(* CODESYS project HiSimulK_NF.project
   Title: BWTS
   Version: 2.0.0.1
   Company: Hyundaiwelding

Project tree, tasks and I/O mapping:
  Device : X2 control 15 - Powerfail, Beijer Electronics Products AB, order no. 
      , version 3.5.13.30
    application Application
      libraries: Util, * (System); Toolbibliothek WM, 1.0.0.6 (Weidmüller Interface GmbH & Co.KG); Standard, * (System); BWTS, 1.4.3.4 (Hyundaiwelding)
      task MainTask (cyclic, interval t#20ms, priority 1) calls MODE, MASTER_SEQUENCE_BALLASTING, MASTER_SEQUENCE_DEBALLASTING, MASTER_SEQUENCE_STRIPPING, SEQ_BAL_SP_P, SEQ_BAL_SP_S, SEQ_BAL_ST_P, SEQ_BAL_ST_S, SEQ_DEBAL_SP_P, SEQ_DEBAL_SP_S, SEQ_DEBAL_ST_P, SEQ_DEBAL_ST_S, SEQ_STRIP_SP, SEQ_STRIP_ST, MASTER_SEQUENCE_DIAGNOSIS, SEQ_DIAG_DEVICE, SEQ_DIAG_INSTRUMENT
      task Alarm (cyclic, interval 20 ms, priority 1) calls ALARM_BUZZER_1, ALARM_BUZZER_2, ALARM_COMMON, ALARM_DEVICE, ALARM_INTERLOCK_A, ALARM_INTERLOCK_D_1, ALARM_INTERLOCK_D_2, ALARM_RECTIFIER, ALARM_TRO
      task ETC (cyclic, interval 50 ms, priority 1) calls AUTO_MODE, BLOWER_TIMER, LINE_UP, MAINTENANCE_AND_DISABLE, RF_CC, SELECTION, TRC_SETTING, UTILITY, RUNNING_HOURS
      task Device (cyclic, interval t#20ms, priority 1) calls DEVICE_AIT151, DEVICE_AIT251, DEVICE_B117A, DEVICE_B117B, DEVICE_FCV1131, DEVICE_FCV2131, DEVICE_FCV1211, DEVICE_FCV2211, DEVICE_GSP01, DEVICE_GSP02, DEVICE_P132, DEVICE_P232, DEVICE_P171A, DEVICE_P171B, DEVICE_RFA, DEVICE_RFB, DEVICE_RFC, DEVICE_WBP01, DEVICE_WBP02, DEVICE_XV1151, DEVICE_XV1171A, DEVICE_XV1171B, DEVICE_XV1172A, DEVICE_XV1321, DEVICE_XV2321, DEVICE_XV1511, DEVICE_XV1512, DEVICE_XV2511, DEVICE_XV2512, DEVICE_XV1731, DEVICE_XV1732, DEVICE_XV1901, DEVICE_XV1541, DEVICE_BA35, DEVICE_BA36, DEVICE_BA37, DEVICE_BA38
      task Shutdown (cyclic, interval t#20ms, priority 1) calls ESD101, PSD10X, PSD11X, PSD12X, PSD20X, PSD21X, PSD22X, PSD30X, PSD31X, USD41X, USD42X, USD43X
      task SIMULATION (cyclic, interval t#20ms, priority 1) calls SCENARIO, SIMULATION_CAL, VIRTUAL_1, VIRTUAL_2, VIRTUAL_3, AMS
      global variables GVL_Alarm_Device
      global variables GVL_IO_DO
      global variables GVL_IO_AO
      global variables GVL_IO_AI
      Logic/
        3.SD/
          program PSD10X [CFC]
          program USD41X [CFC]
          program ESD101 [CFC]
          program PSD20X [CFC]
          program PSD21X [CFC]
          program PSD11X [CFC]
          program USD42X [CFC]
          program PSD12X [CFC]
          program PSD22X [CFC]
          program PSD30X [CFC]
          program PSD31X [CFC]
          program USD43X [CFC]
        1.Mode/
          program MODE [CFC]
        0.ETC/
          program SELECTION [CFC]
          program TRC_SETTING [CFC]
          program MAINTENANCE_AND_DISABLE [CFC]
          program RF_CC [CFC]
          program UTILITY [CFC]
          program BLOWER_TIMER [CFC]
          program AUTO_MODE [CFC]
          program LINE_UP [CFC]
          program RUNNING_HOURS [ST]
        2.Sequence/
          program SEQ_BAL_ST_S [CFC]
          program SEQ_DEBAL_SP_S [CFC]
          program SEQ_DEBAL_ST_S [CFC]
          program MASTER_SEQUENCE_BALLASTING [CFC]
          program MASTER_SEQUENCE_DEBALLASTING [CFC]
          program SEQ_BAL_SP_S [CFC]
          program MASTER_SEQUENCE_STRIPPING [CFC]
          program SEQ_BAL_ST_P [CFC]
          program SEQ_BAL_SP_P [CFC]
          program SEQ_DEBAL_ST_P [CFC]
          program SEQ_DEBAL_SP_P [CFC]
          program SEQ_STRIP_ST [CFC]
          program SEQ_STRIP_SP [CFC]
          program MASTER_SEQUENCE_DIAGNOSIS [CFC]
          program SEQ_DIAG_DEVICE [ST]
          program SEQ_DIAG_INSTRUMENT [ST]
        0.ALARM/
          program ALARM_INTERLOCK_D_1 [CFC]
          program ALARM_BUZZER_1 [ST]
          program ALARM_RECTIFIER [ST]
          program ALARM_INTERLOCK_A [CFC]
          program ALARM_TRO [CFC]
          program ALARM_DEVICE [ST]
          program ALARM_INTERLOCK_D_2 [CFC]
          program ALARM_COMMON [ST]
          program ALARM_BUZZER_2 [ST]
        4.Device/
          program DEVICE_FCV1211 [CFC]
          program DEVICE_P171A [CFC]
          program DEVICE_WBP01 [CFC]
          program DEVICE_XV1731 [CFC]
          program DEVICE_XV1171B [CFC]
          program DEVICE_AIT151 [CFC]
          program DEVICE_XV1732 [CFC]
          program DEVICE_B117B [CFC]
          program DEVICE_XV1511 [CFC]
          program DEVICE_FCV1131 [CFC]
          program DEVICE_RFA [CFC]
          program DEVICE_XV1151 [CFC]
          program DEVICE_B117A [CFC]
          program DEVICE_XV1512 [CFC]
          program DEVICE_P132 [CFC]
          program DEVICE_XV1171A [CFC]
          program DEVICE_XV1172A [CFC]
          program DEVICE_P171B [CFC]
          program DEVICE_P232 [CFC]
          program DEVICE_RFB [CFC]
          program DEVICE_WBP02 [CFC]
          program DEVICE_XV1321 [CFC]
          program DEVICE_XV1541 [CFC]
          program DEVICE_XV2321 [CFC]
          program DEVICE_XV1901 [CFC]
          program DEVICE_GSP01 [CFC]
          program DEVICE_GSP02 [CFC]
          program DEVICE_AIT251 [CFC]
          program DEVICE_XV2511 [CFC]
          program DEVICE_XV2512 [CFC]
          program DEVICE_FCV2211 [CFC]
          program DEVICE_FCV2131 [CFC]
          program DEVICE_RFC [CFC]
          program DEVICE_BA35 [CFC]
          program DEVICE_BA36 [CFC]
          program DEVICE_BA37 [CFC]
          program DEVICE_BA38 [CFC]
        0.SIMULATION/
          program AMS [CFC]
          program SCENARIO [CFC]
          program VIRTUAL_1 [CFC]
          program SIMULATION_CAL [CFC]
          program VIRTUAL_2 [CFC]
          program VIRTUAL_3 [ST]
        0.SIMULATION FBD/
          function block SM_RF_TRO1 [CFC]
          function SM_CELL_VOLT [ST]
          function SM_NA_TRO [ST]
          function SM_H2_CONC [ST]
          function SM_HEAT [ST]
          function block SM_FU_DP [ST]
          function block SM_FOT [CFC]
          function block SM_RF_TRO [ST]
      Symbols
      global variables GVL_Event_Operation
      global variables GVL_SEQ_LIB
      global variables GVL_Event_Device
      global variables GVL_Alarm_Interlock
      global variables GVL_Event_Optrack
      global variables GVL_IO_DI
      global variables GVL_Alarm_System
      global variables GVL_IO_RECTIFIER
      global variables PersistentVars
      global variables GVL_UTILITY
      global variables GVL_SIMULATION
      global variables GVL_IO_TRO
*)

// Device/Application/GVL_Alarm_Device
//{attribute 'qualified_only'}
VAR_GLOBAL
	/////////////////////////////////////// Tags that registered as an Alarm ///////////////////////////////////////
	
	//BLOWER
	B117A_STF : BOOL;
	B117A_SPF : BOOL;
	B117B_STF : BOOL;
	B117B_SPF : BOOL;
	
	XV1171A_OPF : BOOL;
	XV1171A_CLF : BOOL;
	XV1171B_OPF : BOOL;
	XV1171B_CLF : BOOL;
	
	//Sea Water Feeding Unit
	P171A_STF : BOOL;
	P171A_SPF : BOOL;
	P171B_STF : BOOL;
	P171B_SPF : BOOL;
	
	//Injection Flow Control Valves
	FCV1131_CF : BOOL;	// FCV-1131 CONTROL FAIL
	FCV2131_CF : BOOL;	// FCV-2131 CONTROL FAIL
	
	//Main Flow Control Valves
	FCV1211_CF : BOOL;	// FCV-1211 CONTROL FAIL
	FCV2211_CF : BOOL;	// FCV-2211 CONTROL FAIL

	//N.U UNIT
	P132_STF : BOOL;
	P132_SPF : BOOL;
	P232_STF : BOOL;
	P232_SPF : BOOL;
		
	//RECTIFIER
	RF142A_STF : BOOL;
	RF142A_SPF : BOOL;
	RF142B_STF : BOOL;
	RF142B_SPF : BOOL;
	RF142C_STF : BOOL;
	RF142C_SPF : BOOL;

	//W.B PUMP
	WBP01_STF : BOOL;
	WBP01_SPF : BOOL;
	WBP02_STF : BOOL;
	WBP02_SPF : BOOL;

	GSP01_STF : BOOL;
	GSP01_SPF : BOOL;
	GSP02_STF : BOOL;
	GSP02_SPF : BOOL;
	
	/////////////////////////////////////// END : Tags that registered as an Alarm ///////////////////////////////////////
	
	// BALLAST VALVES
	BA35_OPF : BOOL;
	BA35_CLF : BOOL;
	BA36_OPF : BOOL;
	BA36_CLF : BOOL;
	BA37_OPF : BOOL;
	BA37_CLF : BOOL;
	BA38_OPF : BOOL;
	BA38_CLF : BOOL;
END_VAR

// Device/Application/GVL_IO_DO
//{attribute 'qualified_only'}
VAR_GLOBAL
	// Digital Output with DC 24V
	BWTS_003 : BOOL; //Shutdown alarm Lamp
	BWTS_004 : BOOL; //Common alarm Lamp
	BWTS_007 : BOOL; //Alarm buzzer
	
	XV_1151_CMD : BOOL;
	XV_1172A_CMD : BOOL;
	XV_1731_CMD : BOOL;
	XV_1732_CMD : BOOL;
	XV_1171A_CMD : BOOL;
	XV_1171B_CMD : BOOL;
	XV_1901_CMD : BOOL; 

	XV_1321_CMD : BOOL;
	XV_2321_CMD : BOOL;
	AIT_151_ST : BOOL;
	AIT_251_ST : BOOL;

	XV_1511_CMD : BOOL;
	XV_1512_CMD : BOOL;
	XV_2511_CMD : BOOL;
	XV_2512_CMD : BOOL;

	XV_1541_CMD : BOOL;
	
	// Digital Output with free voltage
	
	BWTS_005 : BOOL;		// BWTS COMMON ALARM TO AMS	
	BWTS_006 : BOOL;		// BWTS SHUTDOWN ALARM TO AMS
	BWTS_009 : BOOL;		// BWTS RUNNING TO AMS
	B_117A_ST : BOOL;
	B_117B_ST : BOOL;
	P_171A_ST : BOOL;
	P_171B_ST : BOOL;
	
	P_132_ST : BOOL;
	P_232_ST : BOOL;
	
	RF_142A_ST : BOOL;
	RF_142A_SP : BOOL;
	RF_142B_ST : BOOL;
	RF_142B_SP : BOOL;
	RF_142C_ST : BOOL;
	RF_142C_SP : BOOL;

	GSP_01_SP : BOOL;
	GSP_02_SP : BOOL;
END_VAR

// Device/Application/GVL_IO_AO
//{attribute 'qualified_only'}
VAR_GLOBAL
	// Analog Output
	FCV_1211_CMD : REAL;
	FCV_2211_CMD : REAL;
	
	FCV_1131_CMD : REAL;
	FCV_2131_CMD : REAL;

	P_132_CMD : REAL;
	P_232_CMD : REAL;

END_VAR

// Device/Application/GVL_IO_AI
//{attribute 'qualified_only'}
VAR_GLOBAL
	// Analog Input
	CT_1111 : REAL;
	TE_1111 : REAL;
	AIT_1121 : REAL;
	AIT_1122 : REAL;
	AIT_1123 : REAL;
	PT_1121 : REAL;
	PT_1721 : REAL;
	PT_1722 : REAL;
	LIT_1311 : REAL;
	AP_LVL_01 : REAL;

	P_132_FD : REAL;
	P_232_FD : REAL;

	FCV_1211_FD : REAL;
	FCV_2211_FD : REAL;

	FIT_1211 : REAL;
	FIT_2211 : REAL;

	FCV_1131_FD : REAL;
	FCV_2131_FD : REAL;

	FIT_1131 : REAL;
	FIT_2131 : REAL;

	AIT_151 : REAL;
	AIT_251 : REAL;
	
	/////////////////////////////////////////////////////////// ANALOGUE RANGE ///////////////////////////////////////////////////////////
	
	RL_CT_1111 : REAL := 0;	
	RH_CT_1111 : REAL := 100;
	
	RL_TE_1111 : REAL := 0;
	RH_TE_1111 : REAL := 55;
	
	RL_PT_1121 : REAL := -70;
	RH_PT_1121 : REAL := 70;
	
	RL_PT_1721 : REAL := 0;
	RH_PT_1721 : REAL := 10;
	RL_PT_1722 : REAL := 0;
	RH_PT_1722 : REAL := 10;
	
	RL_AP_LVL_01 : REAL := 0;
	RH_AP_LVL_01 : REAL := 800;	
	
	RL_FIT_1211 : REAL := 0;
	RH_FIT_1211 : REAL := 10163;
	
	RL_FIT_2211 : REAL := 0;
	RH_FIT_2211 : REAL := 10163;
	
	RL_FIT_1131 : REAL := 0;
	RH_FIT_1131 : REAL := 120;
	
	RL_FIT_2131 : REAL := 0;
	RH_FIT_2131 : REAL := 120;
	
	RL_AIT_151 : REAL := 0;
	RH_AIT_151 : REAL := 16;
	
	RL_AIT_251 : REAL := 0;
	RH_AIT_251 : REAL := 16;
	
END_VAR

// Device/Application/GVL_Event_Operation
//{attribute 'qualified_only'}
VAR_GLOBAL
	//OPERATION STATUS
	BAL_ST_S, BAL_IN_STBD, BAL_SP_S, BAL_S_RDY : BOOL;			// STBD BALLASTING
	BAL_ST_P, BAL_IN_PORT, BAL_SP_P, BAL_P_RDY : BOOL;			// PORT BALLASTING  	
		    	
	DEBAL_ST_S, DEBAL_IN_STBD, DEBAL_SP_S, DEBAL_S_RDY : BOOL;				// STBD DEBALLASTING
	DEBAL_ST_P, DEBAL_IN_PORT, DEBAL_SP_P, DEBAL_P_RDY : BOOL;				// PORT DEBALLASTING
		
	STR_ST_S, STR_IN_STBD, STR_SP_S, STR_S_RDY : BOOL;						// STBD STRIPPING
		
	WBP01_ST_REQ: BOOL;
	WBP01_SP_REQ: BOOL;
	WBP02_ST_REQ: BOOL;
	WBP02_SP_REQ: BOOL;
	
	GSP01_ST_REQ: BOOL;
	GSP01_SP_REQ: BOOL;
	GSP02_ST_REQ: BOOL;
	GSP02_SP_REQ: BOOL;	
	
	DIAG_ST, DIAG_IN_SELF : BOOL;	// SELF-DIAGNOSIS --------------- ADDED BY VER.1
END_VAR

// Device/Application/GVL_SEQ_LIB
//{attribute 'qualified_only'}
VAR_GLOBAL
	MST_BST_S, MST_BST_P : BWTS.SEQ;
	MST_BSP_S, MST_BSP_P : BWTS.SEQ;
	
	BST_S_01, BST_P_01 : BWTS.SEQ;	// Blower Start
	
	BST_S_03, BST_P_03 : BWTS.SEQ;	// TRC Valve Init. Open
	BST_S_04, BST_P_04 : BWTS.SEQ;	// Inj. Valve Init. Open
	BST_S_05, BST_P_05 : BWTS.SEQ;	// H/E Valve Init. Open
	BST_S_06, BST_P_06 : BWTS.SEQ;	// S.W.F.P Start
	BST_S_07, BST_P_07 : BWTS.SEQ;	// E/U Level Check
	BST_S_08, BST_P_08 : BWTS.SEQ;	// WBP Start Request
	
	BST_S_10, BST_P_10 : BWTS.SEQ;	// Salinity Check
	
	BST_S_12, BST_P_12 : BWTS.SEQ;	// Main flow Control
	BST_S_13, BST_P_13 : BWTS.SEQ;	// Inj. Flow Control
	BST_S_14, BST_P_14 : BWTS.SEQ;	// Rectifier Start
	BST_S_15, BST_P_15 : BWTS.SEQ;	// TRO Valve Open
	BST_S_16, BST_P_16 : BWTS.SEQ;	// TRO Sensing Start
	
	BST_S_18, BST_P_18 : BWTS.SEQ;	// Ballast Valves ACtion
	                                 	
	BSP_S_01, BSP_P_01 : BWTS.SEQ;	// Rectifier Stop
	
	BSP_S_03, BSP_P_03 : BWTS.SEQ;	// WBP Stop Request
	BSP_S_04, BSP_P_04 : BWTS.SEQ;	// TRO Unit Stop
	BSP_S_05, BSP_P_05 : BWTS.SEQ;	// S.W.F.P Stop
	
	BSP_S_07, BSP_P_07 : BWTS.SEQ;	// H/E Valve Close
	BSP_S_08, BSP_P_08 : BWTS.SEQ;	// Inj. Valve Close
	BSP_S_09, BSP_P_09 : BWTS.SEQ;	// TRC Valve Close
	BSP_S_10, BSP_P_10 : BWTS.SEQ;	// Blower Stop
	
	BSP_S_12, BSP_P_12 : BWTS.SEQ;	// Ballast Valve Act.

	MST_DST_S, MST_DST_P : BWTS.SEQ;
	MST_DSP_S, MST_DSP_P : BWTS.SEQ;
	
	          
	DST_S_02, DST_P_02 : BWTS.SEQ;	// TRC Valve Init. Open        
	DST_S_03, DST_P_03 : BWTS.SEQ;	// N/U Start
	DST_S_04, DST_P_04 : BWTS.SEQ;	// WBP Start Request            
	DST_S_05, DST_P_05 : BWTS.SEQ;	// TRO Valve Open         
	DST_S_06, DST_P_06 : BWTS.SEQ;	// Main Flow Control
	DST_S_07, DST_P_07 : BWTS.SEQ;	// TRO Sensing Start          
	DST_S_08, DST_P_08 : BWTS.SEQ;	// Recirculation Mode       
	DST_S_09, DST_P_09 : BWTS.SEQ;	// Discharge Mode
		                  
	DSP_S_01, DSP_P_01 : BWTS.SEQ;	// WBP Stop Request
	DSP_S_02, DSP_P_02 : BWTS.SEQ;	// N/U Pump Stop
	DSP_S_03, DSP_P_03 : BWTS.SEQ;	// TRO Unit Stop
	
	DSP_S_05, DSP_P_05 : BWTS.SEQ;	// TRC Valve Close
	DSP_S_06, DSP_P_06 : BWTS.SEQ;	// N/U Inj. Valve Close
	DSP_S_07, DSP_P_07 : BWTS.SEQ;	// Ballast Valve Act.

	MST_SST_S, MST_SST_P : BWTS.SEQ;
	MST_SSP_S, MST_SSP_P : BWTS.SEQ;
	
	SST_S_01 : BWTS.SEQ;	// N/U Start          
	SST_S_02 : BWTS.SEQ;	// WBP Start Request       
	SST_S_03 : BWTS.SEQ;	// TRO Valve Open
	SST_S_04 : BWTS.SEQ;	// TRO Sensing Start           
	   
	SST_S_06 : BWTS.SEQ;	// TRC Valve Open         
	SST_S_07 : BWTS.SEQ;	// Ballast Valves Action          
	SST_S_08 : BWTS.SEQ;	// Eductor Valve Open       
	SST_S_09 : BWTS.SEQ;	// TRO Booster Unit Start
	        
	SSP_S_01 : BWTS.SEQ;	// WBP Stop Request
	SSP_S_02 : BWTS.SEQ;	// N/U Pump Stop 
	SSP_S_03 : BWTS.SEQ;	// TRO Unit Stop
	SSP_S_04 : BWTS.SEQ;	// N/U Inj. Valve Close
	
	SSP_S_06 : BWTS.SEQ;	// TRC Valve Close
	SSP_S_07 : BWTS.SEQ;	// Eductor Valve Close
	
	// PSD
	PSD101, PSD102, PSD103, PSD10 : BWTS.PSD;									// Ballasting Common Process Shutdown
	PSD111, PSD113, PSD114, PSD115, PSD11 : BWTS.PSD;					// Ballast STBD Process Shutdown
	PSD121, PSD123, PSD124, PSD125, PSD12 : BWTS.PSD;					// Ballast PORT Process Shutdown
		
	PSD201, PSD20: BWTS.PSD;													// Deballasting Common Process Shutdown
	PSD211, PSD212, PSD213, PSD21 : BWTS.PSD;									// Deballasting STBD Process Shutdown
	PSD221, PSD222, PSD223, PSD22 : BWTS.PSD;									// Deballasting PORT Process Shutdown
		
	PSD301, PSD30 : BWTS.PSD;													// Stripping Common Process Shutdown
	PSD311, PSD312, PSD313, PSD31 : BWTS.PSD;									// Stripping STBD Process Shutdown
		
	SEQ112, SEQ122, SEQ212, SEQ222, SEQ312 : BWTS.PSD;			// Sequence Fail
	
	PSD41, PSD42, PSD43 : BWTS.PSD;
	ESD01 : BWTS.PSD;										// Emergency Shutdown
	
		// SELF-DIAGNOSIS ---------- ADDED BY VER 1
	MST_DIAG : BWTS.SEQ;
	
	DIAG_B117A_1 : BWTS.SEQ;
	DIAG_B117A_2 : BWTS.SEQ;
	DIAG_B117A_3 : BWTS.SEQ;
	
	DIAG_B117B_1 : BWTS.SEQ;
	DIAG_B117B_2 : BWTS.SEQ;
	DIAG_B117B_3 : BWTS.SEQ;
	
	DIAG_XV1171A_1 : BWTS.SEQ;
	DIAG_XV1171A_2 : BWTS.SEQ;
	DIAG_XV1171A_3 : BWTS.SEQ;
	
	DIAG_XV1171B_1 : BWTS.SEQ;
	DIAG_XV1171B_2 : BWTS.SEQ;
	DIAG_XV1171B_3 : BWTS.SEQ;
	
	DIAG_P132_1 : BWTS.SEQ;
	DIAG_P132_2 : BWTS.SEQ;
	DIAG_P132_3 : BWTS.SEQ;
	
	DIAG_P232_1 : BWTS.SEQ;
	DIAG_P232_2 : BWTS.SEQ;
	DIAG_P232_3 : BWTS.SEQ;
	
	DIAG_FCV1211_1 : BWTS.SEQ;
	DIAG_FCV1211_2 : BWTS.SEQ;
	DIAG_FCV1211_3 : BWTS.SEQ;
	DIAG_FCV1211_4 : BWTS.SEQ;
	
	DIAG_FCV2211_1 : BWTS.SEQ;
	DIAG_FCV2211_2 : BWTS.SEQ;
	DIAG_FCV2211_3 : BWTS.SEQ;
	DIAG_FCV2211_4 : BWTS.SEQ;
	
	DIAG_FCV1131_1 : BWTS.SEQ;
	DIAG_FCV1131_2 : BWTS.SEQ;
	DIAG_FCV1131_3 : BWTS.SEQ;
	DIAG_FCV1131_4 : BWTS.SEQ;
	
	DIAG_FCV2131_1 : BWTS.SEQ;
	DIAG_FCV2131_2 : BWTS.SEQ;
	DIAG_FCV2131_3 : BWTS.SEQ;
	DIAG_FCV2131_4 : BWTS.SEQ;
		
	DIAG_BA35_1 : BWTS.SEQ;
	DIAG_BA35_2 : BWTS.SEQ;
	DIAG_BA35_3 : BWTS.SEQ;
	DIAG_BA36_1 : BWTS.SEQ;
	DIAG_BA36_2 : BWTS.SEQ;
	DIAG_BA36_3 : BWTS.SEQ;
	DIAG_BA37_1 : BWTS.SEQ;
	DIAG_BA37_2 : BWTS.SEQ;
	DIAG_BA37_3 : BWTS.SEQ;
	DIAG_BA38_1 : BWTS.SEQ;
	DIAG_BA38_2 : BWTS.SEQ;
	DIAG_BA38_3 : BWTS.SEQ;
END_VAR

// Device/Application/GVL_Event_Device
//{attribute 'qualified_only'}
VAR_GLOBAL
	
	FULL_AUTO : BOOL;
	MAINTENANCE : BOOL;	//Maintenance
	
	// BLOWER UNIT
	B117A_A : BOOL;
	B117A_M : BOOL;
	B117A_RUN : BOOL;
	B117A_SPD : BOOL;
	B117B_A : BOOL;
	B117B_M : BOOL;
	B117B_RUN : BOOL;
	B117B_SPD : BOOL;
	
	XV1171A_A : BOOL; 
	XV1171A_M : BOOL;
	XV1171A_OPD : BOOL;
	XV1171A_CLD : BOOL;
	XV1171B_A : BOOL; 
	XV1171B_M : BOOL;
	XV1171B_OPD : BOOL;
	XV1171B_CLD : BOOL;
		
	// TRC CONTROL VAVLE
	FCV1211_A : BOOL;
	FCV1211_M : BOOL;
	FCV1211_OPD : BOOL;
	FCV1211_CLD : BOOL;
	FCV1211_ON : BOOL;
	
	FCV2211_A : BOOL;
	FCV2211_M : BOOL;
	FCV2211_OPD : BOOL;
	FCV2211_CLD : BOOL;
	FCV2211_ON : BOOL;

	// INJECTION CONTROL VAVLE
	FCV1131_A : BOOL;
	FCV1131_M : BOOL;
	FCV1131_OPD : BOOL;
	FCV1131_CLD : BOOL;
	FCV1131_ON : BOOL;
	
	FCV2131_A : BOOL;
	FCV2131_M : BOOL;
	FCV2131_OPD : BOOL;
	FCV2131_CLD : BOOL;
	FCV2131_ON : BOOL;
	
	// HEATER INLET/BYPASS VAVLE
	XV1731_A : BOOL;
	XV1731_M : BOOL;
	XV1731_OPD : BOOL;
	XV1731_CLD : BOOL;
	XV1732_A : BOOL;
	XV1732_M : BOOL;
	XV1732_OPD : BOOL;
	XV1732_CLD : BOOL;
		
	// SEA WATER FEED PUMP
	P171A_RUN : BOOL;
	P171A_SPD : BOOL;
	P171A_A : BOOL;
	P171A_M : BOOL;
	P171B_RUN : BOOL;
	P171B_SPD : BOOL;
	P171B_A : BOOL;
	P171B_M : BOOL;
	
	// TRO INLET VALVE	
	XV1511_A : BOOL;
	XV1511_M : BOOL;
	XV1511_OPD : BOOL;
	XV1511_CLD : BOOL;
	
	XV1512_A : BOOL;
	XV1512_M : BOOL;
	XV1512_OPD : BOOL;
	XV1512_CLD : BOOL;
			
	XV2511_A : BOOL;
	XV2511_M : BOOL;
	XV2511_OPD : BOOL;
	XV2511_CLD : BOOL;

	XV2512_A : BOOL;
	XV2512_M : BOOL;
	XV2512_OPD : BOOL;
	XV2512_CLD : BOOL;

	XV1541_A, XV1541_M : BOOL;
	XV1541_OPD, XV1541_CLD : BOOL;
 
	// TRO SENSORS
	AIT151_A : BOOL;
	AIT151_M : BOOL;
	AIT151_RUN : BOOL;
	AIT151_SPD : BOOL;
	
	AIT251_A : BOOL;
	AIT251_M : BOOL;
	AIT251_RUN : BOOL;
	AIT251_SPD : BOOL;

	// CLOSED TANK VALVE
	XV1151_A : BOOL;
	XV1151_M : BOOL;
	XV1151_OPD : BOOL;
	XV1151_CLD : BOOL;
	
	// RECTIFIER
	RFA_A : BOOL;
	RFA_M : BOOL;
	RFA_RUN : BOOL;
	RFA_SPD : BOOL;
	
	RFB_A : BOOL;
	RFB_M : BOOL;
	RFB_RUN : BOOL;
	RFB_SPD : BOOL;
	
	RFC_A : BOOL;
	RFC_M : BOOL;
	RFC_RUN : BOOL;
	RFC_SPD : BOOL;
		
	// MAIN PUMP
	WBP01_RUN : BOOL;
	WBP01_SPD : BOOL;	
	WBP02_RUN : BOOL;
	WBP02_SPD : BOOL;
	
	GSP01_RUN : BOOL;
	GSP01_SPD : BOOL;
	GSP02_RUN : BOOL;
	GSP02_SPD : BOOL;
	
	// N.A UNIT
	P132_A : BOOL;
	P132_M : BOOL;
	P132_RUN : BOOL;
	P132_SPD : BOOL;
	
	P232_A : BOOL;
	P232_M : BOOL;
	P232_RUN : BOOL;
	P232_SPD : BOOL;
	
	XV1321_A : BOOL;
	XV1321_M : BOOL;
	XV1321_OPD : BOOL;
	XV1321_CLD : BOOL;
	
	XV2321_A : BOOL;
	XV2321_M : BOOL;
	XV2321_OPD : BOOL;
	XV2321_CLD : BOOL;

	// DRAIN UNIT
	XV1901_A : BOOL;
	XV1901_M : BOOL;
	XV1901_OPD : BOOL;
	XV1901_CLD : BOOL;		

	////////////////////////////////////////////////// SELECTION //////////////////////////////////////////////////
	B117A_SEL : BOOL;
	B117B_SEL : BOOL;
	
	P171A_SEL : BOOL;
	P171B_SEL : BOOL;
	
	TRO01_SEL: BOOL;
	TRO02_SEL : BOOL;
	TRO_CROSS : BOOL;
	
	P132_SEL : BOOL;
	P232_SEL : BOOL;
	NU_CROSS : BOOL;
	
	RFA_DISABLE : BOOL;
	RFB_DISABLE : BOOL;
	RFC_DISABLE : BOOL;
	
	GSP01_SEL : BOOL;
	GSP02_SEL : BOOL;
		
	SEA_ENABLE : BOOL;
	
	SEA_ENABLE_S : BOOL;
	SEA_ENABLE_P : BOOL;
	
	CIR_ENABLE_S : BOOL;
	CIR_ENABLE_P : BOOL;
	
	//BALLAST VALVES
	BA35_A : BOOL;
	BA35_M : BOOL;
	BA36_A : BOOL;
	BA36_M : BOOL;
	BA37_A : BOOL;
	BA37_M : BOOL;
	BA38_A : BOOL;
	BA38_M : BOOL;
END_VAR

// Device/Application/GVL_Alarm_Interlock
//{attribute 'qualified_only'}
VAR_GLOBAL
	/////////////////////////////////////// Tags that registered as an Alarm ///////////////////////////////////////
	//Feeding Sea Water salinity
	CT_1111_LO : BOOL;
	CT_1111_LL : BOOL;
	
	//Feeding Sea Water Temperature
	TE_1111_HI : BOOL;
	TE_1111_LO : BOOL;
	TE_1111_LL : BOOL;
	
	//H2 Gas Detector
	AIT_1121_HH : BOOL;
	AIT_1121_HI : BOOL;
	AIT_1122_HH : BOOL;
	AIT_1122_HI : BOOL;
	AIT_1123_HH : BOOL;
	AIT_1123_HI : BOOL;
	
	//APT Level Too Level
	AP_LVL_LO, AP_LVL_LL : BOOL;
	
	//Blower Unit
	PT_1121_HI : BOOL;
	PT_1121_LO : BOOL;
	PT_1121_LL : BOOL;
	B_117A_F : BOOL;
	B_117B_F : BOOL;
	B_117A_OFF : BOOL;
	B_117B_OFF : BOOL;
	BLR_BOTH_F : BOOL;
	
	//SEA WATER FEEDING UNIT
	PT_1721_HI : BOOL;
	PT_1721_LO : BOOL;
	PT_1721_LL : BOOL;
	PT_1722_HH : BOOL;
	PT_1722_HI : BOOL;
	PT_1722_LO : BOOL;
	
	SWFU_DP_HH : BOOL;
	SWFU_DP_HI : BOOL;
	
	P_171A_F : BOOL;
	P_171A_OFF : BOOL;
	P_171B_F : BOOL;
	P_171B_OFF : BOOL;
	
	SWFP_BOTH_F : BOOL;
	
	// LINE-UP FAIL ALARM
	BAL_VV_AL_S : BOOL;
	BAL_VV_AL_P : BOOL;
		
	DEBAL_VV_AL_S : BOOL;
	DEBAL_VV_AL_P : BOOL;
	
	STR_VV_AL_S : BOOL;
	
	//Main Flow rate
	FIT_1211_HH : BOOL;
	FIT_1211_HI : BOOL;
	FIT_1211_LO : BOOL;
	FIT_2211_HH : BOOL;
	FIT_2211_HI : BOOL;
	FIT_2211_LO : BOOL;
	
	//Injection Flow rate
	FIT_1131_LO, FIT_1131_LL : BOOL;
	FIT_2131_LO, FIT_2131_LL : BOOL;

	RFS_1131 : BOOL;
	RFS_2131 : BOOL;
	
	//TRO Sensor
	BTRO_HH_S : BOOL;
	BTRO_HI_S : BOOL;
	BTRO_LO_S : BOOL;
	BTRO_LL_S : BOOL;
	DTRO_HH_S : BOOL;
	DTRO_HI_S : BOOL;
	
	BTRO_HH_P : BOOL;
	BTRO_HI_P : BOOL;
	BTRO_LO_P : BOOL;
	BTRO_LL_P : BOOL;
	DTRO_HH_P : BOOL;
	DTRO_HI_P : BOOL;
	
	STRO_HH : BOOL;
	STRO_HI : BOOL;
	
	AIT_151_E : BOOL;
	AIT_151_F : BOOL;
	AIT_151_L : BOOL; // FOR HiQ-TRO
	AIT_151_BYPASS : BOOL; // FOR HiQ-TRO (* 2023.06.01, JSY - Change from event to alarm*) 
	AIT_151_PF : BOOL; // FOR HiQ-TRO (* 2023.06.01, JSY - Power source supply statue Purge Controller to the TRO sensor*) 
	
	AIT_251_E : BOOL;
	AIT_251_F : BOOL;
	AIT_251_L : BOOL; // FOR HiQ-TRO
	AIT_251_BYPASS : BOOL; // FOR HiQ-TRO (* 2023.06.01, JSY - Change from event to alarm*)
	AIT_251_PF : BOOL; // FOR HiQ-TRO (* 2023.06.01, JSY - Power source supply statue Purge Controller to the TRO sensor*)

	//TRO DRAIN UNIT
	LS_1901_HH : BOOL;
	
	//E.U Level Switch
	LS_1111_LL : BOOL;
	LS_1141_HI : BOOL;
	
	//N.A UNIT
	LIT_1311_HI : BOOL;
	LIT_1311_LO : BOOL;
	LIT_1311_LL : BOOL;
	
	P_132_TRIP : BOOL;
	P_232_TRIP : BOOL;
	
	DPS_1321 : BOOL;
	DPS_2321 : BOOL;
	
	//RECTIFIER
	//ALARM
	REC1001, REC2001, REC3001 : BOOL;	// RECTIFIER ERROR
	REC1002, REC2002, REC3002 : BOOL;	// RECTIFIER E-STOP BY INTERNAL SAFETY INTERLOCK
	REC1003, REC2003, REC3003 : BOOL;	// RECTIFIER MODULE1 INPUT OVER CURRENT
	REC1004, REC2004, REC3004 : BOOL;	// RECTIFIER MODULE2 INPUT OVER CURRENT
	REC1005, REC2005, REC3005 : BOOL;	// RECTIFIER MODULE3 INPUT OVER CURRENT
	REC1006, REC2006, REC3006 : BOOL;	// RECTIFIER MODULE1 OUTPUT OVER CURRENT
	REC1007, REC2007, REC3007 : BOOL;	// RECTIFIER MODULE2 OUTPUT OVER CURRENT
	REC1008, REC2008, REC3008 : BOOL;	// RECTIFIER MODULE3 OUTPUT OVER CURRENT
	REC1009, REC2009, REC3009 : BOOL;	// RECTIFIER OUTPUT OVER VOLTAGE
	REC1010, REC2010, REC3010 : BOOL;	// RECTIFIER MODULE1 OVER TEMPERATURE
	REC1011, REC2011, REC3011 : BOOL;	// RECTIFIER MODULE2 OVER TEMPERATURE
	REC1012, REC2012, REC3012 : BOOL;	// RECTIFIER MODULE3 OVER TEMPERATURE
	REC1013, REC2013, REC3013 : BOOL;	// RECTIFIER UNBALANCE CURRENT
	REC1014, REC2014, REC3014 : BOOL;	// RECTIFIER LOCAL MODE
	REC1015, REC2015, REC3015 : BOOL;	// RECTIFIER LOCAL-REMOTE MODE
	REC1022, REC2022, REC3022 : BOOL;	// RECTIFIER MODULE1 FUSE ALARM
	REC1023, REC2023, REC3023 : BOOL; 	// RECTIFIER MODULE2 FUSE ALARM
	REC1024, REC2024, REC3024 : BOOL;	// RECTIFIER MODULE3 FUSE ALARM
	REC1025, REC2025, REC3025 : BOOL; 	// RECTIFIER EMERGENCY OPERATION
	REC1026, REC2026, REC3026 : BOOL; 	// RECTIFIER FAN ALARM
	REC1032, REC2032, REC3032 : BOOL; 	// RECTIFIER E-STOP BY EXTERNAL COMMAND
	REC1033, REC2033, REC3033 : BOOL; 	// RECTIFIER INTERNAL OVER TEMPERATURE
	
	REC1017_HH, REC1017_HI, REC1018_HH, REC1018_HI, REC1019_HH, REC1019_HI, REC1020_HH,	REC1020_HI,	REC1021_HH,	REC1021_HI,	REC1027_HH,	REC1027_HI : BOOL;
	RF_142A_E : BOOL;
	
	REC2017_HH,	REC2017_HI, REC2018_HH, REC2018_HI, REC2019_HH, REC2019_HI,	REC2020_HH,	REC2020_HI, REC2021_HH, REC2021_HI, REC2027_HH,	REC2027_HI : BOOL;
	RF_142B_E : BOOL;
	
	REC3017_HH,	REC3017_HI, REC3018_HH, REC3018_HI, REC3019_HH, REC3019_HI,	REC3020_HH,	REC3020_HI, REC3021_HH, REC3021_HI, REC3027_HH,	REC3027_HI : BOOL;
	RF_142C_E : BOOL;
	
	RF_ALL_SPD : BOOL;
	
	//FAN Alarm
	PR_FAN_OFF : BOOL;
	ER_FAN_OFF : BOOL;
	
	// MCC-100 BREAKER OFF
	MCC_100_OFF : BOOL;
	
	//E.U Outlet Alarm
	ZS_1112A_CL : BOOL;
	ZS_1112A_OP : BOOL;
	ZS_1113A_CL : BOOL;
	ZS_1113A_OP : BOOL;
	ZS_1114A_CL : BOOL;
	ZS_1114A_OP : BOOL;
	
	// MAIN PUMP ALARM
	WBP_01_AL : BOOL;
	WBP_01_FAULT : BOOL;
	WBP_02_AL : BOOL;
	WBP_02_FAULT : BOOL;
	
	GSP_01_AL : BOOL;
	GSP_02_AL : BOOL;
	GSP_01_FAULT : BOOL;
	GSP_02_FAULT : BOOL;	
	
	// BYPASS ALARM
	SYS_BYPASS_1 : BOOL;
	SYS_BYPASS_2 : BOOL;
	SYS_BYPASS_3 : BOOL;
	SYS_BYPASS_4 : BOOL;
	
	//BALLAST SYSTEM
	GAS_LEAK_AL : BOOL;			// GAS DETECT FROM PUMP ROOM OR TK
		
END_VAR

// Device/Application/GVL_Event_Optrack
//{attribute 'qualified_only'}
VAR_GLOBAL
	//Operation
	MP_BAL_ST_S, MP_BAL_ST_P: BOOL;		// Ballasting start command (Event)
	MP_BAL_SP_S, MP_BAL_SP_P: BOOL;		// Ballasting stop command (Event)
	MP_BAL_ST_A : BOOL;
	MP_BAL_SP_A : BOOL;	
	
	MP_DEBAL_ST_S, MP_DEBAL_ST_P: BOOL;	// Deballasting start command (Event)
	MP_DEBAL_SP_S, MP_DEBAL_SP_P: BOOL;	// Deballasting stop command (Event)
	MP_DEBAL_ST_A : BOOL;
	MP_DEBAL_SP_A : BOOL;
	
	MP_STRIP_ST_S, MP_STRIP_ST_P: BOOL;
	MP_STRIP_SP_S, MP_STRIP_SP_P: BOOL;
		
	//BLOWER
	MF_B117_BP : BOOL;
	MP_B117A_SEL, MP_B117A_A, MP_B117A_M, MP_B117A_ST, MP_B117A_SP : BOOL;
	MP_B117B_SEL, MP_B117B_A, MP_B117B_M, MP_B117B_ST, MP_B117B_SP : BOOL;
	
	MP_XV1171A_A, MP_XV1171A_M, MP_XV1171A_OP, MP_XV1171A_CL : BOOL;
	MP_XV1171B_A, MP_XV1171B_M, MP_XV1171B_OP, MP_XV1171B_CL : BOOL;
			
	//SEA WATER FEED PUMP
	MP_P171A_SEL, MP_P171A_A, MP_P171A_M, MP_P171A_ST, MP_P171A_SP : BOOL;
    MP_P171B_SEL, MP_P171B_A, MP_P171B_M, MP_P171B_ST, MP_P171B_SP : BOOL;
	
	//MAIN TRC VALVES
	MP_FCV1211_A, MP_FCV1211_M,	MP_FCV1211_SET : BOOL;
	MP_FCV2211_A, MP_FCV2211_M,	MP_FCV2211_SET : BOOL;
		
	MP_TRC_SET_MAIN : BOOL;
	
	//INJECTION VALVES
	MP_FCV1131_A, MP_FCV1131_M,	MP_FCV1131_SET : BOOL;
	MP_FCV2131_A, MP_FCV2131_M,	MP_FCV2131_SET : BOOL;
	
 	//HEATER INLET/BYPSS VALVES
	MP_XV1731_A, MP_XV1731_M, MP_XV1731_OP, MP_XV1731_CL : BOOL;
	MP_XV1732_A, MP_XV1732_M, MP_XV1732_OP, MP_XV1732_CL : BOOL;
	
	//DISABLE
	MF_PT1721, MF_TE1111, MF_CT1111, MF_LIT1311 : BOOL;
	
	//MAINTENANCE
	MP_AIT1121_ST, MP_AIT1121_SP : BOOL;
	MP_AIT1122_ST, MP_AIT1122_SP : BOOL;
	MP_AIT1123_ST, MP_AIT1123_SP : BOOL;
	MP_REPAIR_ST, MP_REPAIR_SP : BOOL;
	
	//TRO INLET VALVE
	MP_XV1511_A, MP_XV1511_M, MP_XV1511_OP, MP_XV1511_CL : BOOL;
	MP_XV1512_A, MP_XV1512_M, MP_XV1512_OP, MP_XV1512_CL : BOOL;
	
	MP_XV2511_A, MP_XV2511_M, MP_XV2511_OP, MP_XV2511_CL : BOOL;
	MP_XV2512_A, MP_XV2512_M, MP_XV2512_OP, MP_XV2512_CL : BOOL;

	//TRO SAMPLING UNIT
	MP_XV1541_A, MP_XV1541_M, MP_XV1541_OP, MP_XV1541_CL : BOOL;
	
	//CLOSED TANK VALVE
	MP_XV1151_A, MP_XV1151_M, MP_XV1151_OP, MP_XV1151_CL : BOOL;
	
	//AIR DILUTION VALVE
	MP_XV1172A_OP, MP_XV1172A_CL : BOOL;
	
	//TRO SENSOR
	MP_TRO01_SEL : BOOL;
	MP_TRO02_SEL : BOOL;
	
	MP_TRO_CROSS : BOOL;
	MP_TRO_NORMAL : BOOL;
	
	
	MP_AIT151_A, MP_AIT151_M, MP_AIT151_ST, MP_AIT151_SP : BOOL;
	MP_AIT251_A, MP_AIT251_M, MP_AIT251_ST, MP_AIT251_SP : BOOL;
	
	//DRAIN UNIT
	MP_XV1901_A, MP_XV1901_M, MP_XV1901_OP, MP_XV1901_CL : BOOL;  
 	
	//RECTIFIER
	MP_RFA_EN, MP_RFA_DIS, MP_RFA_A, MP_RFA_M, MP_RFA_ST, MP_RFA_SP, MP_RFA_SET : BOOL;
	MP_RFB_EN, MP_RFB_DIS, MP_RFB_A, MP_RFB_M, MP_RFB_ST, MP_RFB_SP, MP_RFB_SET : BOOL;
	MP_RFC_EN, MP_RFC_DIS, MP_RFC_A, MP_RFC_M, MP_RFC_ST, MP_RFC_SP, MP_RFC_SET : BOOL; 
	
	//G.S PUMP
	MP_GSP01_SEL, MP_GSP02_SEL : BOOL;
		
	//N.A UNIT
	MF_NA_PRE_SET : BOOL;		// NA PRE-SET FUNCTION ACTIVATE ------------ ADDED BY VER 1
	MP_NU_CROSS, MP_NU_NORMAL : BOOL;
	MP_P132_SEL, MP_P232_SEL : BOOL;
		
	MP_P132_A, MP_P132_M, MP_P132_ST, MP_P132_SP, MP_P132_SET : BOOL;
	MP_P232_A, MP_P232_M, MP_P232_ST, MP_P232_SP, MP_P232_SET : BOOL;
			
	MP_XV1321_A, MP_XV1321_M, MP_XV1321_OP, MP_XV1321_CL : BOOL;
	MP_XV2321_A, MP_XV2321_M, MP_XV2321_OP, MP_XV2321_CL : BOOL;
	
	// APT LEVEL
	MF_APT : BOOL;
	
	//BALLAST VALVE(YARD)
	
	//E-STOP
	MP_ESTOP : BOOL;
	//RESET
	MP_RESET : BOOL;
	//ACK
	MP_SOUNDOFF : BOOL;

	
	
	
	MP_SEA_EN_S : BOOL;
	MP_SEA_DIS_S : BOOL;
	MP_SEA_EN_P : BOOL;
	MP_SEA_DIS_P : BOOL;
	MP_CIR_EN_S : BOOL;
	MP_CIR_DIS_S : BOOL;
	MP_CIR_EN_P : BOOL;
	MP_CIR_DIS_P : BOOL;
	
	// BALLAST VALVE CONTROL
	MP_BA35_A : BOOL;
	MP_BA35_M : BOOL;
	MP_BA35_OP : BOOL;
	MP_BA35_CL : BOOL;
	MP_BA35_RESET : BOOL;
	
	MP_BA36_A : BOOL;
	MP_BA36_M : BOOL;
	MP_BA36_OP : BOOL;
	MP_BA36_CL : BOOL;
	MP_BA36_RESET : BOOL;
	
	MP_BA37_A : BOOL;
	MP_BA37_M : BOOL;
	MP_BA37_OP : BOOL;
	MP_BA37_CL : BOOL;
	MP_BA37_RESET : BOOL;
	
	MP_BA38_A : BOOL;
	MP_BA38_M : BOOL;
	MP_BA38_OP : BOOL;
	MP_BA38_CL : BOOL;
	MP_BA38_RESET : BOOL;
	
	// SELF-DIAGNOSIS
	MP_DIAG_ST : BOOL;
	
	// RUNNING HOUR
	MP_RH_EM_TOTAL_RESET, MP_RH_EM_PARTIAL_RESET : BOOL;
	
	MP_RH_AIT1121_RESET, MP_RH_AIT1122_RESET, MP_RH_AIT1123_RESET : BOOL;
	
	MP_RH_P171A_RESET, MP_RH_P171B_RESET : BOOL;
	
	MP_RH_P132_RESET, MP_RH_P232_RESET : BOOL;
	
	MP_RH_AIT151_RESET, MP_RH_AIT251_RESET : BOOL;	
	
	MP_RH_BAL_M_RESET : BOOL;
	MP_RH_DEBAL_M_RESET : BOOL;
	MP_RH_STRIP_RESET : BOOL;
END_VAR

// Device/Application/GVL_IO_DI
//{attribute 'qualified_only'} // Digital Input
VAR_GLOBAL
	// Tags that do not require registration as an event.
	BWTS_002 : BOOL; //Sound off cc-100 
	
	B_117A_RUN : BOOL;
	B_117B_RUN : BOOL;
	P_171A_RUN : BOOL;
	P_171B_RUN : BOOL;

	XV_1171A_OPD : BOOL;
	XV_1171A_CLD : BOOL;
	XV_1171B_OPD : BOOL;
	XV_1171B_CLD : BOOL;
	
	P_132_RUN : BOOL;	
	P_232_RUN : BOOL;
		
	WBP_01_RUN : BOOL;
	WBP_02_RUN : BOOL;
	GSP_01_RUN : BOOL;
	GSP_02_RUN : BOOL;
		
	// Tags that registered as an Event
	LS_1111 : BOOL;
	LS_1141 : BOOL;
		
	P_132_RMT : BOOL := TRUE;
	P_232_RMT : BOOL := TRUE;
		
	LS_1901_HI : BOOL;
	LS_1901_LO : BOOL;
		
	BWTS_MODE : BOOL;
	
	ZS_1112A_OPD : BOOL;
	ZS_1113A_OPD : BOOL;
	
	ER_01_FAN : BOOL;
	ER_02_FAN : BOOL;
	ER_03_FAN : BOOL;
	ER_04_FAN : BOOL;
	PR_01_FAN : BOOL;
	PR_02_FAN : BOOL;
	
	/////////////////////// END : Tags that registered as an Event 
	BWTS_008 : BOOL;
	
	///////////////////// FOR SIMULATION
	ZS_1114A_OPD : BOOL;
END_VAR

// Device/Application/GVL_Alarm_System
//{attribute 'qualified_only'}
VAR_GLOBAL
	//Emergency STOP
	CC100_TEMP_HI : BOOL;	//CC-100 TEMPERATURE HIGH
	ESTOP_HMI: BOOL;		//E-STOP FROM HMI
	ESTOP_CC: BOOL;			//E-STOP FROM CC-100
	ESTOP_RF: BOOL;			//E-STOP FROM RECTIFIER
	
	//BLOWER BYPASS
	BLR_BYPASS : BOOL;
	
	//SIGNAL FAILURE

	
	//DISABLE
	DISABLE1 : BOOL;	//STRAINER PRESSURE SENSOR DISABLE
	DISABLE2 : BOOL;	//SEA WATER TEMPERATURE SENSOR DISABLE
	DISABLE3 : BOOL;	//SEA WATER SALINITY SENSOR DISABLE
	DISABLE4 : BOOL;	//N.A TANK LEVEL SENSOR DISABLE
	
	//MAINTENANCE
	MM_AIT1121 : BOOL;	//AIT-1121 MAINTENANCE MODE
	MM_AIT1122 : BOOL;	//AIT-1122 MAINTENANCE MODE
	MM_AIT1123 : BOOL;	//AIT-1123 MAINTENANCE MODE
	MM_REPAIR : BOOL;	//REPAIR MODE
	
	//SHUTDOWN
	ESD : BOOL;	//EMERGENCY ACTIVATION
	
	PSD_11 : BOOL; //STBD Ballasting Process Shutdown Activation
	PSD_12 : BOOL; //PORT Ballasting Process Shutdown Activation
	
 	PSD_21 : BOOL; //STBD DeBallasting Process Shutdown Activation
	PSD_22 : BOOL; //PORT DeBallasting Process Shutdown Activation
	
	PSD_31 : BOOL; //Stripping Process Shutdown Activation
	
	PSD_41 : BOOL; //NO.1 RECTIFIER SHUTDOWN ACTIVATION
	PSD_42 : BOOL; //NO.2 RECTIFIER SHUTDOWN ACTIVATION
	PSD_43 : BOOL; //NO.3 RECTIFIER SHUTDOWN ACTIVATION
	
	//RUNNING HOUR
	RH_EU_AL : BOOL;
	
	RH_AIT1121_AL : BOOL;
	RH_AIT1122_AL : BOOL;
	RH_AIT1123_AL : BOOL;
	
	RH_P171A_AL : BOOL;
	RH_P171B_AL : BOOL;
	
	RH_P132_AL : BOOL;
	RH_P232_AL : BOOL;
	
	RH_AIT151_AL : BOOL;
	RH_AIT251_AL : BOOL;
	
	// LOW SALINITY AREA ALARM
	GPS_ALARM : BOOL;
	
END_VAR

// Device/Application/GVL_IO_RECTIFIER
//{attribute 'qualified_only'}
VAR_GLOBAL
	//STATUS RECTIFIER->CC
	REC1000, REC2000, REC3000 : BOOL;	// RECTIFIER RUNNING
	REC1016, REC2016, REC3016 : BOOL;	// RECTIFIER REMOTE MODE
	REC1017, REC2017, REC3017 : REAL;	// RECTIFIER TOTAL OUTPUT CURRENT
	REC1018, REC2018, REC3018 : REAL;	// RECTIFIER TOTAL OUTPUT VOLTAGE
	REC1019, REC2019, REC3019 : REAL;	// RECTIFIER MODULE1 TEMPERATURE
	REC1020, REC2020, REC3020 : REAL;	// RECTIFIER MODULE2 TEMPERATURE
	REC1021, REC2021, REC3021 : REAL;	// RECTIFIER MODULE3 TEMPERATURE
	REC1027, REC2027, REC3027 : REAL;	// RECTIFIER INTERNAL TEMPERATURE
	REC1028, REC2028, REC3028 : REAL;	// RECTIFIER SHUNT#1 CURRENT
	REC1029, REC2029, REC3029 : REAL;	// RECTIFIER SHUNT#2 CURRENT
	REC1030, REC2030, REC3030 : REAL;	// RECTIFIER SHUNT#3 CURRENT
	REC1031, REC2031, REC3031 : REAL;	// RECTIFIER SHUNT#4 CURRENT
		
	//ORDER CC->RECTIFIER
	REC1041, REC2041, REC3041 : BOOL;	// RECTIFIER START/STOP
	REC1043, REC2043, REC3043 : REAL;	// RECTIFIER CURRENT SET
		
	//BUFFER
	
	RF142A, RF142B, RF142C	: ARRAY[1..34] OF WORD; (* Buffer for registers (receive or send)  *)
			
	/////////////////////////////////////////////////////////// ANALOGUE RANGE ///////////////////////////////////////////////////////////
	
	RL_REC1017, RL_REC2017, RL_REC3017 : REAL := 0;
	RH_REC1017, RH_REC2017, RH_REC3017 : REAL := 1000;
	RL_REC1018, RL_REC2018, RL_REC3018 : REAL := 0;
	RH_REC1018, RH_REC2018, RH_REC3018 : REAL := 200;
	RL_REC1043, RL_REC2043, RL_REC3043 : REAL := 0;
	RH_REC1043, RH_REC2043, RH_REC3043 : REAL := 1000;
	
	
END_VAR

// Device/Application/PersistentVars
//{attribute 'qualified_only'}
VAR_GLOBAL PERSISTENT RETAIN
	
	/////////////////////////////////////// Tags that registered as an Alarm ///////////////////////////////////////
	/////////////////////////////////////// Alarm Parameter ///////////////////////////////////////

			
	// FLOW RATE
	MS_FIT1211_HH : REAL := 115;
	MS_FIT1211_HI : REAL := 110;
	MS_FIT1211_LO : REAL := 20;
	TD_FIT1211_HH : TIME := T#300S;
	TD_FIT1211_HI : TIME := T#180S;
	TD_FIT1211_LO : TIME := T#180S;
	
	MS_FIT2211_HH : REAL := 115;
	MS_FIT2211_HI : REAL := 110;
	MS_FIT2211_LO : REAL := 20;
	TD_FIT2211_HH : TIME := T#300S;
	TD_FIT2211_HI : TIME := T#180S;
	TD_FIT2211_LO : TIME := T#180S;

	
	// SEA WATER FEEDING UNIT
	MS_PT1721_HI : REAL := 6.5;   
	MS_PT1721_LO : REAL := 2.5;   
	MS_PT1721_LL : REAL := 2;    
	TD_PT1721_HI : TIME := T#10S;
	TD_PT1721_LO : TIME := T#10S;
	TD_PT1721_LL : TIME := T#10S;

	MS_PT1722_HH : REAL := 7;   
	MS_PT1722_HI : REAL := 6.5;   
	MS_PT1722_LO : REAL := 2;    
	TD_PT1722_HH : TIME := T#10S;
	TD_PT1722_HI : TIME := T#10S;
	TD_PT1722_LO : TIME := T#10S;

	MS_DP171_HH : REAL := 1;
	MS_DP171_HI : REAL := 0.7;	
	TD_DP171_HH : TIME := T#60S;
	TD_DP171_HI : TIME := T#30S;

	// BLOWER PRESSURE
	MS_PT1121_HI : REAL := 30;
	MS_PT1121_LO : REAL := 5;
	MS_PT1121_LL : REAL := 1;
	TD_PT1121_HI : TIME := T#30S;
	TD_PT1121_LO : TIME := T#30S;
	TD_PT1121_LL : TIME := T#5S;
	
	// H2 GAS DETECTOR
	MS_AIT1121_HH : REAL := 50;
	MS_AIT1121_HI : REAL := 25;
	TD_AIT1121_HH : TIME := T#5S;
	TD_AIT1121_HI : TIME := T#30S;
	
	MS_AIT1122_HH : REAL := 50;
	MS_AIT1122_HI : REAL := 25;
	TD_AIT1122_HH : TIME := T#1S;
	TD_AIT1122_HI : TIME := T#30S;
	
	MS_AIT1123_HH : REAL := 50;
	MS_AIT1123_HI : REAL := 25;
	TD_AIT1123_HH : TIME := T#1S;
	TD_AIT1123_HI : TIME := T#30S;
	
	// SEA WATER TEMPERATURE	
	MS_TE1111_HI : REAL := 38;
	MS_TE1111_LO : REAL := 10;
	MS_TE1111_LL : REAL := 4;
	TD_TE1111_HI : TIME := T#60S;
	TD_TE1111_LO : TIME := T#60S;
	TD_TE1111_LL : TIME := T#60S;
	
	// SEA WATER SALINITY
	MS_CT1111_LO : REAL := 15;
	MS_CT1111_LL : REAL := 10;
	TD_CT1111_LO : TIME := T#30S;
	TD_CT1111_LL : TIME := T#180S;
	
	// INJECTION FLOW RATE
	MS_FIT1131_LO : REAL := 50;   
	MS_FIT1131_LL : REAL := 30;   
	TD_FIT1131_LO : TIME := T#180S;   
	TD_FIT1131_LL : TIME := T#30S;
	
	MS_FIT2131_LO : REAL := 50;   
	MS_FIT2131_LL : REAL := 30;   
	TD_FIT2131_LO : TIME := T#180S;   
	TD_FIT2131_LL : TIME := T#30S;
	
	// TRO
	MS_BTRO_HH : REAL := 10.5;
	MS_BTRO_HI : REAL := 10;
	MS_BTRO_LO : REAL := 5.5;
	MS_BTRO_LL : REAL := 5;
	TD_BTRO_HH : TIME := T#600S;
	TD_BTRO_HI : TIME := T#300S;
	TD_BTRO_LO : TIME := T#300S;
	TD_BTRO_LL : TIME := T#600S;

	MS_DTRO_HH : REAL := 0.1;
	MS_DTRO_HI : REAL := 0.08;
	TD_DTRO_HH : TIME := T#1S;
	TD_DTRO_HI : TIME := T#1S;
	
	// NU
	MS_LIT1311_HI : REAL := 100;
	MS_LIT1311_LO : REAL := 50;
	MS_LIT1311_LL : REAL := 15;
	TD_LIT1311_HI : TIME := T#30S;
	TD_LIT1311_LO : TIME := T#30S;
	TD_LIT1311_LL : TIME := T#60S;
		
	//RECTIFIER
	MS_100D_A_HH : REAL := 830; 
	MS_100D_A_HI : REAL := 825; 
	TD_100D_A_HH : TIME := T#1S;
	TD_100D_A_HI : TIME := T#1S;
	MS_100D_V_HH : REAL := 134; 
	MS_100D_V_HI : REAL := 127; 
	TD_100D_V_HH : TIME := T#1S;
	TD_100D_V_HI : TIME := T#1S;
	
	MS_MD_TEMP_HH : REAL := 97;
	MS_MD_TEMP_HI : REAL := 95;
	TD_MD_TEMP_HH : TIME := T#30S;
	TD_MD_TEMP_HI : TIME := T#30S;
	
	MS_RF_TEMP_HH : REAL := 73;
	MS_RF_TEMP_HI : REAL := 70;
	TD_RF_TEMP_HH : TIME := T#30S;
	TD_RF_TEMP_HI : TIME := T#30S;

	// AP TANK LEVEL
	MS_AP_LO : REAL := 310;
	MS_AP_LL : REAL := 242;
	TD_AP_LO : TIME := T#30S;
	TD_AP_LL : TIME := T#60S;
	
	/////////////////////////////////////// System Parameter ///////////////////////////////////////
	
	// BLOWER TIMER
	MS_BLR_PRE : TIME := T#120S;				// BLOWER PRE-RUN TIME
	MS_BLR_GAS : TIME := T#300S;				// BLOWER GAS OPERATING TIME
	MS_BLR_SP : TIME := T#600S;					// BLOWER SAFETY OPERATING TIME
	
	// TRO SENSOR TIMER
	MS_TRO_WAIT : TIME := T#30S;				// TRO START WAITING TIME
	MS_TRO_SAMPLING : TIME := T#10S;			// TRO SAMPLING LINE FILLING TIME 
	MS_TRO_STABLE : TIME := T#600S;				// TRO INITIAL STABLE TIME FOR BALLASTING
	MS_DTRO_STABLE : TIME := T#180S;			// TRO INITIAL STABLE TIME FOR DEBALLASTING
	
	// YARD VALVE
	MS_RECIRCULATION_ST : TIME := T#180S;		// RECIRCULATION TIME DURING DE-BALLASTING START-UP
	MS_YARD_AL : TIME := T#120S;				// YARD ALARM DELAY TIME
		
	// MAIN FCV VALVE
	MS_FCV1211_BAL : REAL := 35;				// MAIN FCV VALVES INITIAL OPEN SET VALUE FOR BALLASTING
	MS_FCV1211_DEBAL : REAL := 35;				// MAIN FCV VALVES INITIAL OPEN SET VALUE FOR DE-BALLASTING
	MS_FCV1211_BF : REAL := 5;					// MAIN FCV VALVES CLOSING SET VALUE ON BACK-FLUSHING 
	MS_FCV1211_DB : REAL := 5;					// DEADBAND OF TRC CONTROL
	MS_FCV1211_STEP : REAL := 1;				// STEP SIZE OF TRC CONTROL
	MS_FCV1211_SAMPLE : TIME := T#10S;			// STEP INTERVAL TIME OF TRC CONTROL
	MS_FCV1211_MIN : REAL := 15;				// MAIN FCV VALVES LIMIT (MIN)
	MS_FCV1211_MAX : REAL := 65;				// MAIN FCV VALVES LIMIT (MAX)
	MS_FCV1211_ASDB : REAL := 10;				// MAIN FCV VALVES OPEN&CLOSE RECOGNITION SET VALUE
	MS_FCV1211_CFDB : REAL := 10;				// MAIN FCV VALVES CONTROL FAILURE RECOGNITION SET VALUE
	MS_FCV1211_TRC : REAL:= 3000;				// TARGET TRC SET VALUE (S.V)
	
	MS_FCV2211_BAL : REAL := 15;				// MAIN FCV VALVES INITIAL OPEN SET VALUE FOR BALLASTING
	MS_FCV2211_DEBAL : REAL := 15;				// MAIN FCV VALVES INITIAL OPEN SET VALUE FOR DE-BALLASTING
	MS_FCV2211_BF : REAL := 5;					// MAIN FCV VALVES CLOSING SET VALUE ON BACK-FLUSHING 
	MS_FCV2211_DB : REAL := 5;					// DEADBAND OF TRC CONTROL
	MS_FCV2211_STEP : REAL := 1;				// STEP SIZE OF TRC CONTROL
	MS_FCV2211_SAMPLE : TIME := T#10S;			// STEP INTERVAL TIME OF TRC CONTROL
	MS_FCV2211_MIN : REAL := 15;				// MAIN FCV VALVES LIMIT (MIN)
	MS_FCV2211_MAX : REAL := 65;				// MAIN FCV VALVES LIMIT (MAX)
	MS_FCV2211_ASDB : REAL := 10;				// MAIN FCV VALVES OPEN&CLOSE RECOGNITION SET VALUE
	MS_FCV2211_CFDB : REAL := 10;				// MAIN FCV VALVES CONTROL FAILURE RECOGNITION SET VALUE
	MS_FCV2211_TRC : REAL:= 3000;				// TARGET TRC SET VALUE (S.V)

	// INJECTION VALVE
	MS_INJECTION_TG : REAL := 60; 
	
	MS_FCV1131_INIT : REAL := 30;				// INJECTION FCV VALVES INITIAL OPEN SET VALUE
	MS_FCV1131_KP : REAL := 0.005;				// PID PROPORTIONAL CONSTANT
	MS_FCV1131_KI : REAL := 0.02;				// PID RESET TIME
	MS_FCV1131_KD : REAL := 0.02;				// PID DERIVATIVE TIME
	MS_FCV1131_MIN : REAL := 30;				// INJECTION FCV VALVES LIMIT (MIN)
	MS_FCV1131_MAX : REAL := 65;				// INJECTION FCV VALVES LIMIT (MAX)
	MS_FCV1131_ASDB : REAL	:= 10;				// INJECTION FCV VALVES OPEN&CLOSE RECOGNITION SET VALUE     
	MS_FCV1131_CFDB : REAL := 10;               // INJECTION FCV VALVES CONTROL FAILURE RECOGNITION SET VALUE
	
	MS_FCV2131_INIT : REAL := 60;				// INJECTION FCV VALVES INITIAL OPEN SET VALUE
	MS_FCV2131_KP : REAL := 0.005;				// PID PROPORTIONAL CONSTANT
	MS_FCV2131_KI : REAL := 0.02;				// PID RESET TIME
	MS_FCV2131_KD : REAL := 0.02;				// PID DERIVATIVE TIME
	MS_FCV2131_MIN : REAL := 30;				// INJECTION FCV VALVES LIMIT (MIN)
	MS_FCV2131_MAX : REAL := 65;				// INJECTION FCV VALVES LIMIT (MAX)
	MS_FCV2131_ASDB : REAL	:= 10;				// INJECTION FCV VALVES OPEN&CLOSE RECOGNITION SET VALUE     
	MS_FCV2131_CFDB : REAL := 10;               // INJECTION FCV VALVES CONTROL FAILURE RECOGNITION SET VALUE
	
	// N.A UNIT
	MS_NU_PRE : TIME := T#60S;					// N.A PUMP PRE-RUN TIME
	MS_NU_DB : REAL := 0.01;				// TRO DEADBAND FOR N.A CONTROL
	MS_NU_TRG : REAL := 0.06;				// TARGET TRO FOR N.A CONTROL

	MS_P132_INIT : REAL := 75;					// NEUTRALIZATION P/P INITIAL SET VALUE
	MS_P132_UP : REAL := 6;						// NEUTRALIZATION P/P STEP SET VALUE (UP)
	MS_P132_DOWN : REAL := 4;					// NEUTRALIZATION P/P STEP SET VALUE (DOWN)
	MS_P132_SAMPLE : TIME := T#60S;				// NEUTRALIZATION P/P STEP INTERVAL TIME OF N.A CONTROL
	MS_P132_MIN : REAL := 10;					// NEUTRALIZATION P/P STROKE LIMIT (MIN)
	MS_P132_MAX : REAL := 100;					// NEUTRALIZATION P/P STROKE LIMIT (MAX)
		
	MS_P232_INIT : REAL := 75;					// NEUTRALIZATION P/P INITIAL SET VALUE
	MS_P232_UP : REAL := 6;						// NEUTRALIZATION P/P STEP SET VALUE (UP)
	MS_P232_DOWN : REAL := 4;					// NEUTRALIZATION P/P STEP SET VALUE (DOWN)	
	MS_P232_SAMPLE : TIME := T#60S;				// NEUTRALIZATION P/P STEP INTERVAL TIME OF N.A CONTROL
	MS_P232_MIN : REAL := 10;       			// NEUTRALIZATION P/P STROKE LIMIT (MIN)
	MS_P232_MAX : REAL := 100;      			// NEUTRALIZATION P/P STROKE LIMIT (MAX)

	//HEAT EXCHANGER
	MS_TE_NOR : REAL := 10;						// HEAT EXCHANGER VALVE CHANGE TRIGGER VALUE
	
	//SALINITY RECOVERY
	MS_CIT_NOR : REAL := 15;					// SALINITY RECOVERY TRIGGER VALUE
	
	//WAITING TIME FOR WBP
	MS_WBP_SP : TIME := T#10S;					
	
	// SEA WATER FEED UNIT
	MS_SWP_ST : TIME := T#10S;					// SWFP START WAITING TIME
	MS_SWP_SP : TIME := T#60S;					// SWFP STOP WAITING TIME
	
	//RECTIFIER
	MS_RF_TRG : REAL := 8;						// TARGET TRO FOR RECTIFIER CONTROL
	MS_RF_DB : REAL := 0.4;						// TRO DEADBAND FOR RECTIFIER CONTROL 
	MS_RF_CCSS_MAX : REAL := 5;					// RECTIFIER CCSS LIMIT (MAX)
	MS_RF_HOLD : TIME := T#300S;				// RECTIFIER INITIAL HOLDING TIME
	MS_RF_SAMPLE : TIME := T#60S;				// RECTIFIER STEP INTERVAL TIME
	
	MS_RFA_INIT : REAL := 375;					// RECTIFIER INITIAL CURRENT SET VALUE
	MS_RFA_MIN : REAL := 50;					// RECTIFIER LIMIT (MIN)
	MS_RFA_MAX : REAL := 820;					// RECTIFIER LIMIT (MAX)
		
	MS_RFB_INIT : REAL := 375;					// RECTIFIER INITIAL CURRENT SET VALUE	
	MS_RFB_MIN : REAL := 50;					// RECTIFIER LIMIT (MIN)
	MS_RFB_MAX : REAL := 820;					// RECTIFIER LIMIT (MAX)
	
	MS_RFC_INIT : REAL := 375;					// RECTIFIER INITIAL CURRENT SET VALUE	
	MS_RFC_MIN : REAL := 50;					// RECTIFIER LIMIT (MIN)
	MS_RFC_MAX : REAL := 820;					// RECTIFIER LIMIT (MAX)
                                 			
	//CONTROL RIGHT
	ControlRight : INT;
	ControlRightFlagLOS : INT;
	ControlRightFlagROS : INT;
	
	//SELF-DIAGNOSIS
	MS_DIAG_TIME : TIME :=T#5M;
	
	// RUNNING HOUR
	TIME_RH_EM_TOTAL, TIME_RH_EM_PARTIAL : UDINT;
	     
	TIME_RH_AIT1121, TIME_RH_AIT1122, TIME_RH_AIT1123 : UDINT;
	     
	TIME_RH_P171A, TIME_RH_P171B : UDINT;
	     
	TIME_RH_P132, TIME_RH_P232 : UDINT;
	     
	TIME_RH_AIT151, TIME_RH_AIT251 : UDINT;	
		 
	TIME_RH_BAL_M : UDINT;	
	TIME_RH_DEBAL_M : UDINT;
	TIME_RH_STRIP : UDINT;
	
END_VAR

// Device/Application/GVL_UTILITY
//{attribute 'qualified_only'}
VAR_GLOBAL
	TRO_STBD : REAL;
	TRO_PORT : REAL;
	TRO_STR : REAL;
	
	INJECTION_TG_S : REAL;
	INJECTION_TG_P : REAL;
		
	DP_P171 : REAL;
	
	MS_P132_SET : REAL;
	MS_P232_SET : REAL;
		
	SET_TOTAL_TRC : REAL;
	
	SET_FCV1211_TRC : REAL;	
	SET_FCV2211_TRC : REAL;	
	
	MS_FCV1211_SET : REAL;
	MS_FCV2211_SET : REAL;
	
	MS_FCV1131_SET : REAL;
	MS_FCV2131_SET : REAL;
	
	RFA_CCSS : REAL;
	MS_RFA_SET : REAL;
	RFB_CCSS : REAL;
	MS_RFB_SET : REAL;
	RFC_CCSS : REAL;
	MS_RFC_SET : REAL;
	
	ROS_HART_BIT : INT;
	LOS_HART_BIT : INT;
	
	// VAVLE LINE-UP FLAG
	BAV_BAL_S : BOOL;
	BAV_BAL_P : BOOL;

	BAV_DEBAL_S : BOOL;
	BAV_DEBAL_P : BOOL;

	BAV_STR_S : BOOL;

	// OPERATION FLAG
	ON_IN_OP : BOOL;
	ON_IN_BAL : BOOL;
	ON_IN_DEBAL : BOOL;
	ON_IN_STR : BOOL;
	
	//GPS
	LAT_DEG : UINT;
	LAT_MIN : REAL;
	LAT_DIR : STRING;
	LON_DEG : UINT;
	LON_MIN : REAL;
	LON_DIR : STRING;
	
	//SIMULATION
	H2_GAS : REAL;
	CELL_VOLT : REAL;
	SW_TEMP : REAL;

	TRO_RF_S : REAL;
	TRO_RF_P : REAL;
	TRO_NA_S : REAL;
	TRO_NA_P : REAL;
	
	// NA PRE-SET ---------- ADDED BY VER 1
	NA_PRE_INIT_P132 : REAL;
	NA_PRE_MAX_P132 : REAL;
	NA_PRE_MIN_P132 : REAL;
	
	NA_PRE_INIT_P232 : REAL;
	NA_PRE_MAX_P232 : REAL;
	NA_PRE_MIN_P232 : REAL;

	
	MS_TRO_HOLD_P132 : REAL;					// NA PRE-SET TARTGET HOLDING TIME
	MS_TRO_HOLD_P232 : REAL;					// NA PRE-SET TARTGET HOLDING TIME
		
	// SELF-DIAGNOSIS  ---------------- ADDED BY VER.1
	DIAG_ELAPSE_TIME : TIME ;
	DIAG_COMPLETE : BOOL;
	
	B117A_PASS   : BOOL;
	B117B_PASS   : BOOL;
	
	XV1171A_PASS   : BOOL;
	XV1171B_PASS   : BOOL;
	
	FCV1211_PASS   : BOOL;
	FCV2211_PASS   : BOOL;
		
	FCV1131_PASS   : BOOL;
	FCV2131_PASS   : BOOL;
		 
	P132_PASS   : BOOL;
	P232_PASS   : BOOL;
				
	RF142A_PASS : BOOL;
	RF142B_PASS : BOOL;
	RF142C_PASS : BOOL;
	
	AIT151_PASS : BOOL;
	AIT251_PASS : BOOL;
		
	TE1111_PASS : BOOL;
	CT1111_PASS : BOOL;
	
	PT1721_PASS : BOOL;
	PT1722_PASS : BOOL;
	
	AIT1121_PASS : BOOL;
	AIT1122_PASS : BOOL;
	AIT1123_PASS : BOOL;
	
	PT1121_PASS : BOOL;
	
	FIT1211_PASS : BOOL;
	FIT2211_PASS : BOOL;
		 
	FIT1131_PASS : BOOL;
	FIT2131_PASS : BOOL;
		
	LIT1311_PASS : BOOL;
	
	BA035_PASS : BOOL;
	BA036_PASS : BOOL;
	BA037_PASS : BOOL;
	BA038_PASS : BOOL;
	
	RF_INTERLOCK: BOOL;
	
	// RUNNING HOUR DISPLAY VARIABLE
	TIME_TOTAL_HOUR_EM_TOTAL : UDINT;	
	TIME_TOTAL_HOUR_EM_PARTIAL : UDINT;
	
	TIME_TOTAL_DAY_AIT1121,	TIME_TOTAL_DAY_AIT1122,	TIME_TOTAL_DAY_AIT1123 : UDINT;
	
	TIME_TOTAL_DAY_P171A, TIME_TOTAL_DAY_P171B : UDINT;
	
	TIME_TOTAL_HOUR_P132, TIME_TOTAL_HOUR_P232 : UDINT;
		
	TIME_TOTAL_DAY_AIT151, TIME_TOTAL_DAY_AIT251 : UDINT;
	
	TIME_DAY_RH_BAL_M, TIME_HOUR_RH_BAL_M, TIME_MIN_RH_BAL_M : UDINT;
	
	TIME_DAY_RH_DEBAL_M, TIME_HOUR_RH_DEBAL_M, TIME_MIN_RH_DEBAL_M : UDINT;
		
	TIME_DAY_RH_STRIP, TIME_HOUR_RH_STRIP, TIME_MIN_RH_STRIP : UDINT;
	
	// REPORT FLAG
	REPORT_BAL_ST_M, REPORT_BAL_SP_M, SD_BAL_M : BOOL;
	
	REPORT_DEBAL_ST_M, REPORT_DEBAL_SP_M, SD_DEBAL_M : BOOL;

	REPORT_STRIP_ST, REPORT_STRIP_SP, SD_STRIP : BOOL;
	
	REPORT_RFA_ST, REPORT_RFA_SP, SD_RFA : BOOL;
	REPORT_RFB_ST, REPORT_RFB_SP, SD_RFB : BOOL;
	REPORT_RFC_ST, REPORT_RFC_SP, SD_RFC : BOOL;
END_VAR

// Device/Application/GVL_SIMULATION
//{attribute 'qualified_only'}
VAR_GLOBAL
	// BALLAST VALVES
	BA30_OPD : BOOL;
	BA30_CLD : BOOL;
	BA31_OPD : BOOL;
	BA31_CLD : BOOL;
	BA32_OPD : BOOL;
	BA32_CLD : BOOL;
	BA33_OPD : BOOL;
	BA33_CLD : BOOL;
	BA34_OPD : BOOL;
	BA34_CLD : BOOL;
	BA35_OPD : BOOL;
	BA35_CLD : BOOL;
	BA36_OPD : BOOL;
	BA36_CLD : BOOL;
	BA37_OPD : BOOL;
	BA37_CLD : BOOL;
	BA38_OPD : BOOL;
	BA38_CLD : BOOL;
	BA39_OPD : BOOL;
	BA39_CLD : BOOL;
	
	MP_BA30_V_OP : BOOL;
	MP_BA30_V_CL : BOOL;
	MP_BA31_V_OP : BOOL;
	MP_BA31_V_CL : BOOL;
	MP_BA32_V_OP : BOOL;
	MP_BA32_V_CL : BOOL;
	MP_BA33_V_OP : BOOL;
	MP_BA33_V_CL : BOOL;
	MP_BA34_V_OP : BOOL;
	MP_BA34_V_CL : BOOL;
	MP_BA35_V_OP : BOOL;
	MP_BA35_V_CL : BOOL;
	MP_BA36_V_OP : BOOL;
	MP_BA36_V_CL : BOOL;
	MP_BA37_V_OP : BOOL;
	MP_BA37_V_CL : BOOL;
	MP_BA38_V_OP : BOOL;
	MP_BA38_V_CL : BOOL;
	MP_BA39_V_OP : BOOL;
	MP_BA39_V_CL : BOOL;
	
	//SCENARIO
	SCENARIO1 : BOOL;
	SCENARIO2_1 : BOOL;
	SCENARIO2_2 : BOOL;
	SCENARIO3_1 : BOOL;
	SCENARIO3_2 : BOOL;
	SCENARIO4_1 : BOOL;
	SCENARIO4_2 : BOOL;
	SCENARIO5 : BOOL;
	SCENARIO6 : BOOL;
	SCENARIO7 : BOOL;
	SCENARIO8_1 : BOOL;
	SCENARIO8_2 : BOOL;
	SCENARIO9_1 : BOOL;
	SCENARIO9_2 : BOOL;
	SCENARIO10_1 : BOOL;
	SCENARIO10_2 : BOOL;
	
		// SCENARIO
	MP_SCEN1_ST : BOOL;
	MP_SCEN1_SP : BOOL;
	MP_SCEN2_1_ST : BOOL;
	MP_SCEN2_1_SP : BOOL;
	MP_SCEN2_2_ST : BOOL;
	MP_SCEN2_2_SP : BOOL;
	MP_SCEN3_1_ST : BOOL;
	MP_SCEN3_1_SP : BOOL;
	MP_SCEN3_2_ST : BOOL;
	MP_SCEN3_2_SP : BOOL;
	MP_SCEN4_1_ST : BOOL;
	MP_SCEN4_1_SP : BOOL;
	MP_SCEN4_2_ST : BOOL;
	MP_SCEN4_2_SP : BOOL;
	MP_SCEN5_ST : BOOL;
	MP_SCEN5_SP : BOOL;
	MP_SCEN6_ST : BOOL;
	MP_SCEN6_SP : BOOL;
	MP_SCEN7_ST : BOOL;
	MP_SCEN7_SP : BOOL;
	MP_SCEN8_1_ST : BOOL;
	MP_SCEN8_1_SP : BOOL;
	MP_SCEN8_2_ST : BOOL;
	MP_SCEN8_2_SP : BOOL;
	MP_SCEN9_1_ST : BOOL;
	MP_SCEN9_1_SP : BOOL;
	MP_SCEN9_2_ST : BOOL;
	MP_SCEN9_2_SP : BOOL;
	MP_SCEN10_1_ST : BOOL;
	MP_SCEN10_1_SP : BOOL;
	MP_SCEN10_2_ST : BOOL;
	MP_SCEN10_2_SP : BOOL;
	
	// Simulation Manual Set (Analogue)
	MS_CT1111 : REAL;
	MF_CT1111_MAN : BOOL;
	
	MS_TE1111 : REAL;
	MF_TE1111_MAN : BOOL;
	
	MS_PT1121 : REAL;
	MF_PT1121_MAN : BOOL;
	
	MS_AIT1121 : REAL;
	MF_AIT1121_MAN : BOOL;
	MS_AIT1122 : REAL;
	MF_AIT1122_MAN : BOOL;
	MS_AIT1123 : REAL;
	MF_AIT1123_MAN : BOOL;
	
	MS_PT1721 : REAL;
	MF_PT1721_MAN : BOOL;
	MS_PT1722 : REAL;
	MF_PT1722_MAN : BOOL;
	
	MS_PIT1211 : REAL;
	MF_PIT1211_MAN : BOOL;
	MS_PIT1212 : REAL;
	MF_PIT1212_MAN : BOOL;
	MS_PIT2211 : REAL;
	MF_PIT2211_MAN : BOOL;
	MS_PIT2212 : REAL;
	MF_PIT2212_MAN : BOOL;
	
	MS_LIT1311 : REAL;
	MF_LIT1311_MAN : BOOL;
	
	MS_FIT1131 : REAL;
	MF_FIT1131_MAN : BOOL;
	MS_FIT2131 : REAL;
	MF_FIT2131_MAN : BOOL;
	
	MS_FIT1211 : REAL;
	MF_FIT1211_MAN : BOOL;
	MS_FIT2211 : REAL;
	MF_FIT2211_MAN : BOOL;
	
	MS_AIT151 : REAL;
	MF_AIT151_MAN : BOOL;
	MS_AIT251 : REAL;
	MF_AIT251_MAN : BOOL;
	
	MS_APLVL01 : REAL;
	MF_APLVL01_MAN : BOOL;
	
	// Simulation Manual Set (Digital)
	
	MF_BWTS008 : BOOL;
	MF_BWTS008_MAN : BOOL;
	
	MF_LS1111 : BOOL;
	MF_LS1111_MAN : BOOL;
	
	MF_LS1141 : BOOL;
	MF_LS1141_MAN : BOOL;
	
	MF_B117ARUN : BOOL;
	MF_B117ARUN_MAN : BOOL;
	MF_B117BRUN : BOOL;
	MF_B117BRUN_MAN : BOOL;
	
	MF_P171ARUN : BOOL;
	MF_P171ARUN_MAN : BOOL;
	MF_P171BRUN : BOOL;
	MF_P171BRUN_MAN : BOOL;
	
	MF_P132RUN : BOOL;
	MF_P132RUN_MAN : BOOL;
	MF_P232RUN : BOOL;
	MF_P232RUN_MAN : BOOL;	
	
	MF_LS1901HI : BOOL;
	MF_LS1901HI_MAN : BOOL;
	MF_LS1901LO : BOOL;
	MF_LS1901LO_MAN : BOOL;	
	
	MF_F121F : BOOL;
	MF_F121F_MAN : BOOL;
	MF_F221F : BOOL;
	MF_F221F_MAN : BOOL;

	MF_ZS1112AOPD : BOOL;
	MF_ZS1112AOPD_MAN : BOOL;
	MF_ZS1113AOPD : BOOL;
	MF_ZS1113AOPD_MAN : BOOL;
	MF_ZS1114AOPD : BOOL;
	MF_ZS1114AOPD_MAN : BOOL;	
	
	///////////////////////////////////////////////////////////// SIMULATION PARAMETER
	MS_SCEN2_1 : REAL := 14;				// Salinity Low
	MS_SCEN2_2 : REAL := 9;					// Salinity Too Low
	MS_SCEN3_1 : REAL := 9;					// Temperature Low
	MS_SCEN3_2 : REAL := 3;					// Temperature Too Low
	MS_SCEN4_1 : REAL := 0.75;				// Filter DP High
	MS_SCEN4_2 : REAL := 1.1;				// Filter DP Too High
	MS_SCEN8_1_1 : REAL := 10.1;			// TRO HIGH BAL
	MS_SCEN8_1_2 : REAL := 0.09;			// TRO HIGH DEBAL
	MS_SCEN8_2_1 : REAL := 10.6;			// TRO TOO HIGH BAL
	MS_SCEN8_2_2 : REAL := 0.11;			// TRO TOO HIGH DEBAL
	MS_SCEN9_1 : REAL := 5.4;				// TRO Low Bal
	MS_SCEN9_2 : REAL := 4.9;				// TRO Too Low Bal
	MS_SCEN10_1 : REAL := 49;				// NA Tank Level Low 
	MS_SCEN10_2 : REAL := 14;				// NA Tank Level Too Low
	
	MS_BLR_CAPA : REAL := 2750;				// Blower Capacity
	MS_SW_IN : REAL := 25;					// Source Water Temperature
	MS_HEAT_CAPA : REAL := 60;				// Heat Exchanger Capacity
	MS_SLOPE_FACT : REAL := -1158.8;		// Heat Exchanger Slope factor
	MS_CONTROL_FACT : REAL := 0.25;			// Heat Exchanger Control factor
	MS_SW_QA : REAL := 100;					// Sea Water Quality for filter DP.
	MS_FU_AREA : REAL := 18.07;				// Filtration Area for filter DP.
	MS_TAU_TRO : REAL := 60;				// Time constant for TRO first order time  
	MS_TAU_TRC : REAL := 0.5;				// Time constant for TRC first order time
	MS_NA_CAPA : REAL := 122.4;				// N.A Pump Capacity
	MS_RESIDUAL_TRO : REAL := 2;			// Residual TRO Value in Ballast Tank
END_VAR

// Device/Application/GVL_IO_TRO
//{attribute 'qualified_only'}
VAR_GLOBAL
	TRO1000 : REAL;		// TRO Value
	TRO1001 : REAL;		// Remaining Reagent
	TRO1002 : BOOL;		// Common Alarm
	TRO1003 : BOOL;		// Visible lamp blown fail
	TRO1004 : BOOL;		// Intake solenoid fail
	TRO1005 : BOOL;		// Drain solenoid fail
	TRO1006 : BOOL;		// Bypass solenoid fail
	TRO1007 : BOOL;		// Reagent solenoid (indicator)
	TRO1008 : BOOL;		// Reagent solenoid (buffer) fail
	TRO1009 : BOOL;		// Reagent motor (indicator) fail
	TRO1010 : BOOL;		// Reagent motor (buffer) fail
	TRO1011 : BOOL;		// No water
	TRO1012 : BOOL;		// Water slow
	TRO1013 : BOOL;		// Water fast
	
	TRO1101 : BOOL;		// SENSING START
	TRO1102 : BOOL;		// ALL CHECK
		
	TRO151	: ARRAY[1..5] OF WORD; (* Buffer for registers (receive or send) *)
	
	TRO2000 : REAL;		// TRO Value
	TRO2001 : REAL;		// Remaining Reagent
	TRO2002 : BOOL;		// Common Alarm
	TRO2003 : BOOL;		// Visible lamp blown fail
	TRO2004 : BOOL;		// Intake solenoid fail
	TRO2005 : BOOL;		// Drain solenoid fail
	TRO2006 : BOOL;		// Bypass solenoid fail
	TRO2007 : BOOL;		// Reagent solenoid (indicator)
	TRO2008 : BOOL;		// Reagent solenoid (buffer) fail
	TRO2009 : BOOL;		// Reagent motor (indicator) fail
	TRO2010 : BOOL;		// Reagent motor (buffer) fail
	TRO2011 : BOOL;		// No water
	TRO2012 : BOOL;		// Water slow
	TRO2013 : BOOL;		// Water fast
	
	TRO2101 : BOOL;		// SENSING START
	TRO2102 : BOOL;		// ALL CHECK
		
	TRO251	: ARRAY[1..5] OF WORD; (* Buffer for registers (receive or send) *)
END_VAR

// Device/Application/Logic/1.Mode/MODE
PROGRAM MODE
VAR	
	MODE_BAL_S: BWTS.MODE;
	MODE_BAL_P: BWTS.MODE;
			
	MODE_DEBAL_S: BWTS.MODE;
	MODE_DEBAL_P: BWTS.MODE;
		
	MODE_STRIP_S: BWTS.MODE;
	MODE_STRIP_P: BWTS.MODE;
		
	BAL_S_RESET: BOOL;
	BAL_P_RESET: BOOL;
		
	SEQ111_FAIL: BOOL;
	SEQ121_FAIL: BOOL;
		
	DEBAL_S_RESET: BOOL;
	DEBAL_P_RESET: BOOL;
		
	SEQ211_FAIL: BOOL;
	SEQ221_FAIL: BOOL;
				
	STRIP_S_RESET: BOOL;
			
	SEQ311_FAIL: BOOL;
		
	DIAG_RDY : BOOL;
	DIAG_RESET : BOOL;
	MODE_DIAG : BWTS.MODE;		
END_VAR
VAR // added by the converter: edge detectors and wires of the graphical bodies
    _w1, _w2, _w6, _w7, _w11, _w12, _w15, _w16 : ANY;
    _w3, _w4, _w5, _w8, _w9, _w10, _w13, _w14, _w17, _w18 : BOOL;
END_VAR

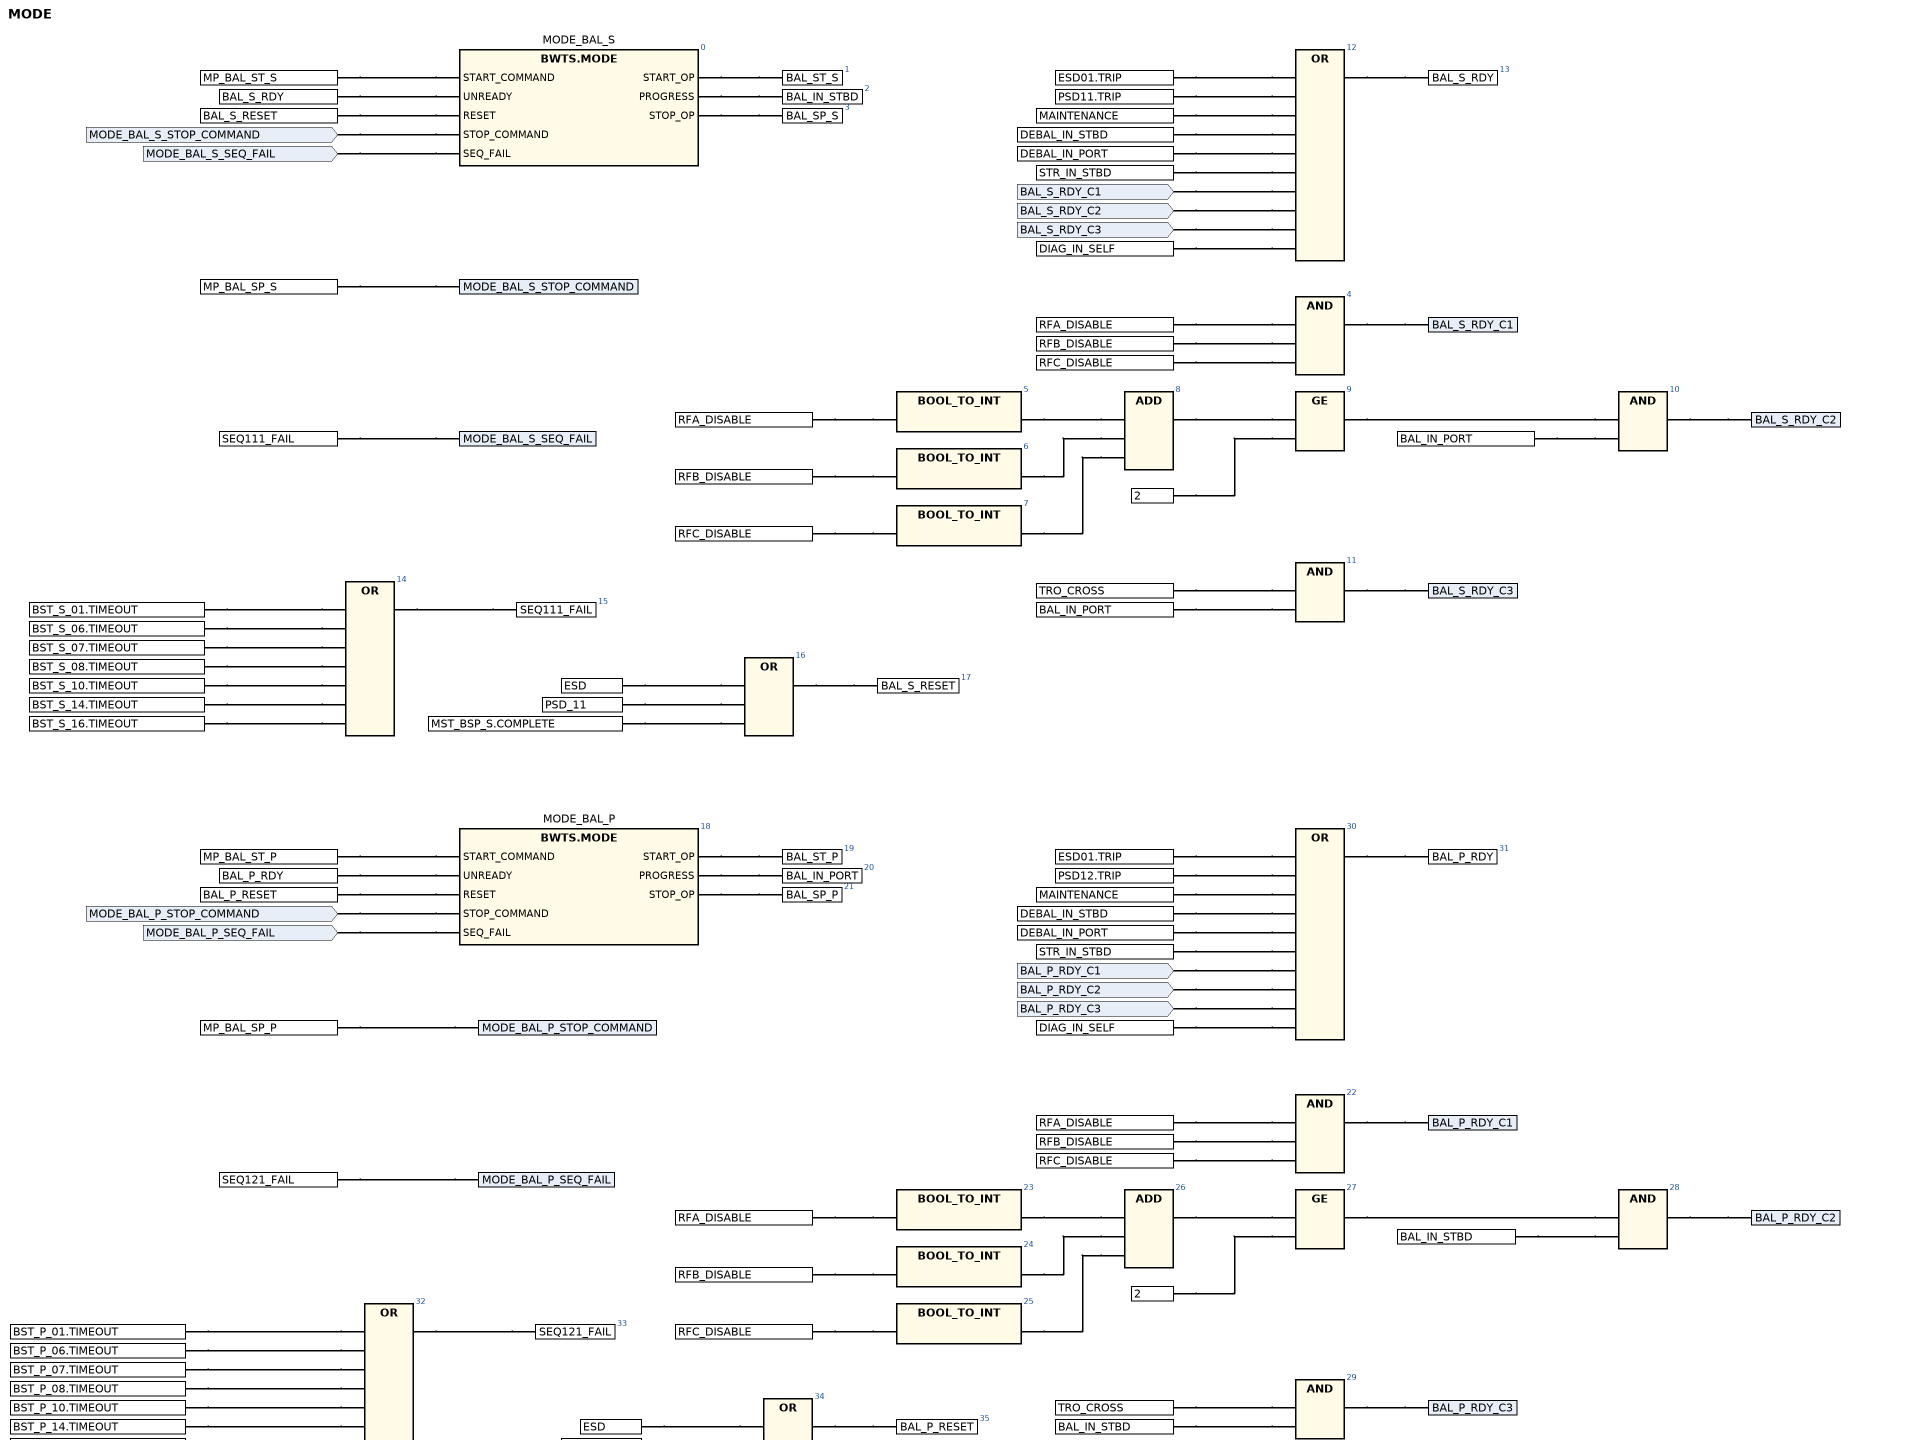
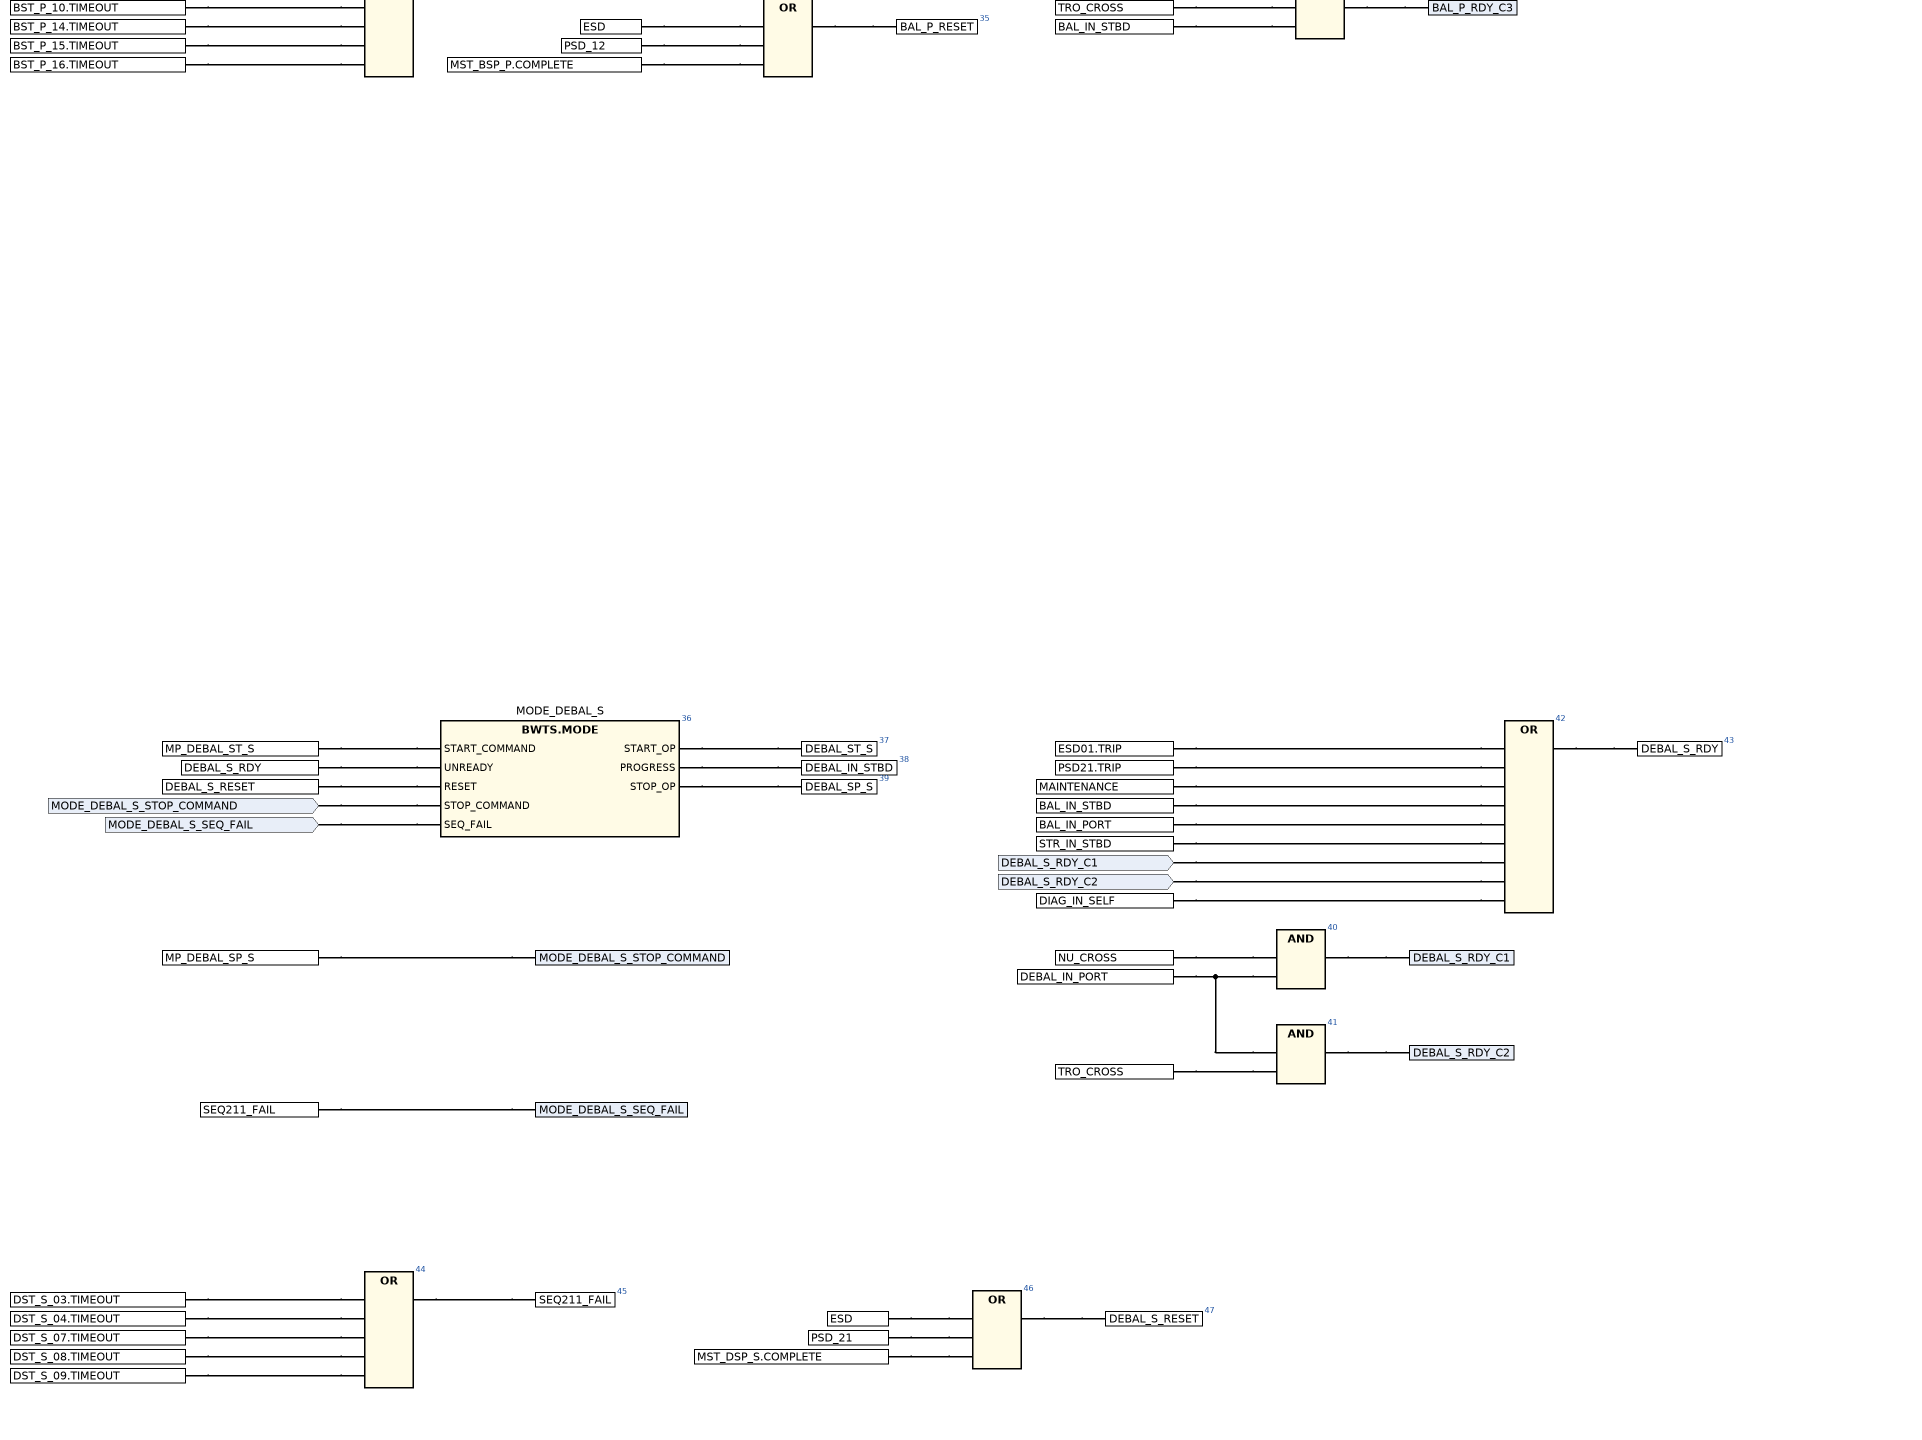
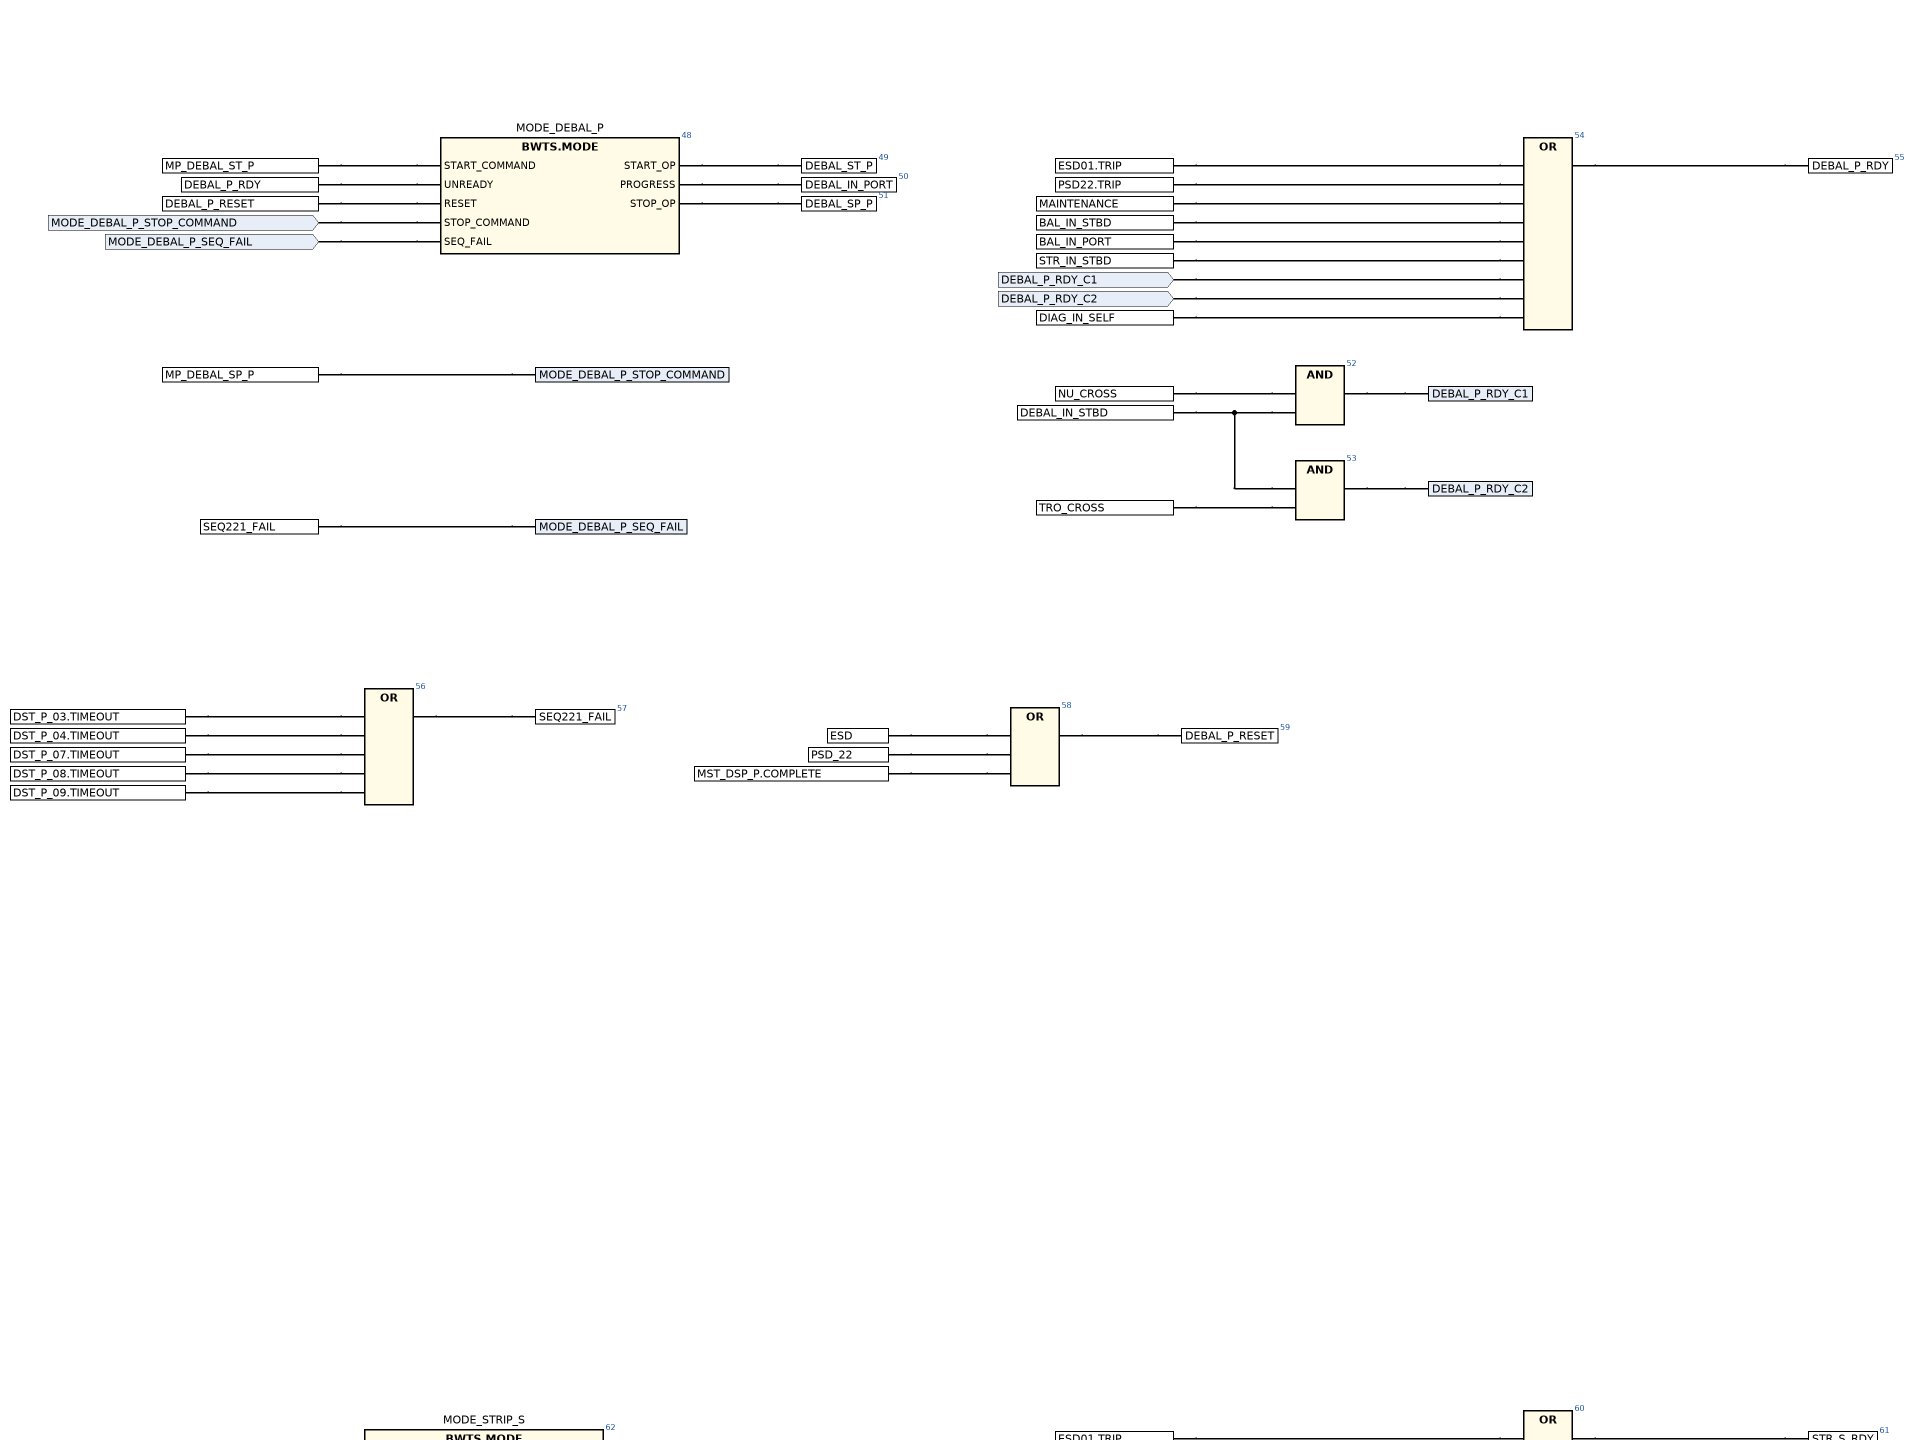
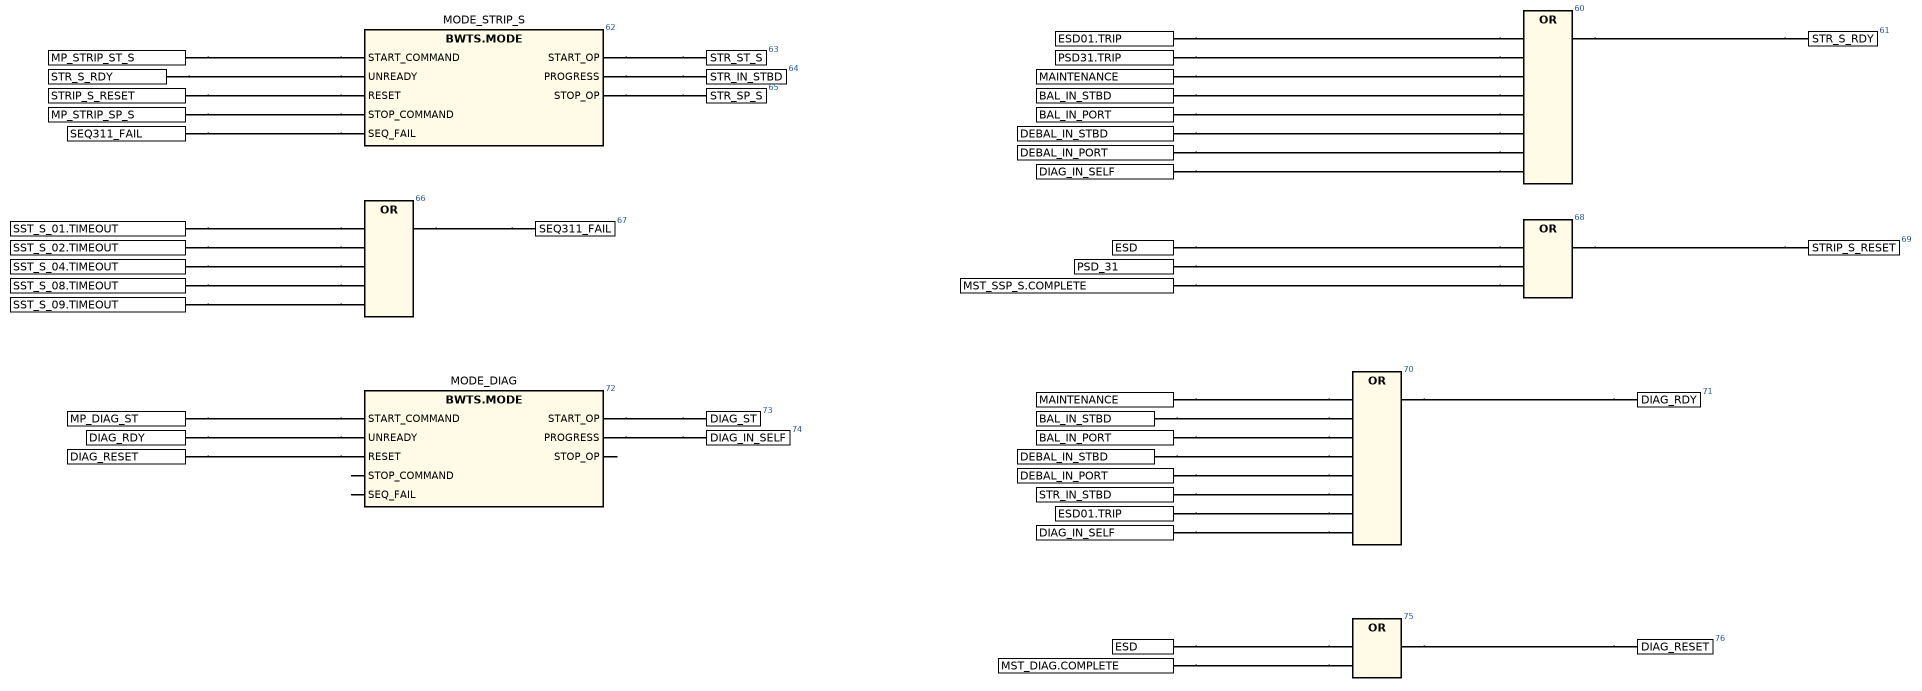
MODE_BAL_S(
    START_COMMAND := MP_BAL_ST_S,
    UNREADY := BAL_S_RDY,
    RESET := BAL_S_RESET,
    STOP_COMMAND := _w1,
    SEQ_FAIL := _w2); // BWTS.MODE
BAL_ST_S := MODE_BAL_S.START_OP;
BAL_IN_STBD := MODE_BAL_S.PROGRESS;
BAL_SP_S := MODE_BAL_S.STOP_OP;
(* RFA_DISABLE AND RFB_DISABLE AND RFC_DISABLE; result not used *)
(* BOOL_TO_INT(RFA_DISABLE) + BOOL_TO_INT(RFB_DISABLE) + BOOL_TO_INT(RFC_DISABLE) >= 2 AND BAL_IN_PORT; result not used *)
(* TRO_CROSS AND BAL_IN_PORT; result not used *)
BAL_S_RDY := ESD01.TRIP OR PSD11.TRIP OR MAINTENANCE OR DEBAL_IN_STBD OR DEBAL_IN_PORT OR STR_IN_STBD OR _w3 OR _w4 OR _w5 OR DIAG_IN_SELF;
SEQ111_FAIL := BST_S_01.TIMEOUT OR BST_S_06.TIMEOUT OR BST_S_07.TIMEOUT OR BST_S_08.TIMEOUT OR BST_S_10.TIMEOUT OR BST_S_14.TIMEOUT OR BST_S_16.TIMEOUT;
BAL_S_RESET := ESD OR PSD_11 OR MST_BSP_S.COMPLETE;
MODE_BAL_P(
    START_COMMAND := MP_BAL_ST_P,
    UNREADY := BAL_P_RDY,
    RESET := BAL_P_RESET,
    STOP_COMMAND := _w6,
    SEQ_FAIL := _w7); // BWTS.MODE
BAL_ST_P := MODE_BAL_P.START_OP;
BAL_IN_PORT := MODE_BAL_P.PROGRESS;
BAL_SP_P := MODE_BAL_P.STOP_OP;
(* RFA_DISABLE AND RFB_DISABLE AND RFC_DISABLE; result not used *)
(* BOOL_TO_INT(RFA_DISABLE) + BOOL_TO_INT(RFB_DISABLE) + BOOL_TO_INT(RFC_DISABLE) >= 2 AND BAL_IN_STBD; result not used *)
(* TRO_CROSS AND BAL_IN_STBD; result not used *)
BAL_P_RDY := ESD01.TRIP OR PSD12.TRIP OR MAINTENANCE OR DEBAL_IN_STBD OR DEBAL_IN_PORT OR STR_IN_STBD OR _w8 OR _w9 OR _w10 OR DIAG_IN_SELF;
SEQ121_FAIL := BST_P_01.TIMEOUT OR BST_P_06.TIMEOUT OR BST_P_07.TIMEOUT OR BST_P_08.TIMEOUT OR BST_P_10.TIMEOUT OR BST_P_14.TIMEOUT OR BST_P_15.TIMEOUT OR BST_P_16.TIMEOUT;
BAL_P_RESET := ESD OR PSD_12 OR MST_BSP_P.COMPLETE;
MODE_DEBAL_S(
    START_COMMAND := MP_DEBAL_ST_S,
    UNREADY := DEBAL_S_RDY,
    RESET := DEBAL_S_RESET,
    STOP_COMMAND := _w11,
    SEQ_FAIL := _w12); // BWTS.MODE
DEBAL_ST_S := MODE_DEBAL_S.START_OP;
DEBAL_IN_STBD := MODE_DEBAL_S.PROGRESS;
DEBAL_SP_S := MODE_DEBAL_S.STOP_OP;
(* NU_CROSS AND DEBAL_IN_PORT; result not used *)
(* DEBAL_IN_PORT AND TRO_CROSS; result not used *)
DEBAL_S_RDY := ESD01.TRIP OR PSD21.TRIP OR MAINTENANCE OR BAL_IN_STBD OR BAL_IN_PORT OR STR_IN_STBD OR _w13 OR _w14 OR DIAG_IN_SELF;
SEQ211_FAIL := DST_S_03.TIMEOUT OR DST_S_04.TIMEOUT OR DST_S_07.TIMEOUT OR DST_S_08.TIMEOUT OR DST_S_09.TIMEOUT;
DEBAL_S_RESET := ESD OR PSD_21 OR MST_DSP_S.COMPLETE;
MODE_DEBAL_P(
    START_COMMAND := MP_DEBAL_ST_P,
    UNREADY := DEBAL_P_RDY,
    RESET := DEBAL_P_RESET,
    STOP_COMMAND := _w15,
    SEQ_FAIL := _w16); // BWTS.MODE
DEBAL_ST_P := MODE_DEBAL_P.START_OP;
DEBAL_IN_PORT := MODE_DEBAL_P.PROGRESS;
DEBAL_SP_P := MODE_DEBAL_P.STOP_OP;
(* NU_CROSS AND DEBAL_IN_STBD; result not used *)
(* DEBAL_IN_STBD AND TRO_CROSS; result not used *)
DEBAL_P_RDY := ESD01.TRIP OR PSD22.TRIP OR MAINTENANCE OR BAL_IN_STBD OR BAL_IN_PORT OR STR_IN_STBD OR _w17 OR _w18 OR DIAG_IN_SELF;
SEQ221_FAIL := DST_P_03.TIMEOUT OR DST_P_04.TIMEOUT OR DST_P_07.TIMEOUT OR DST_P_08.TIMEOUT OR DST_P_09.TIMEOUT;
DEBAL_P_RESET := ESD OR PSD_22 OR MST_DSP_P.COMPLETE;
STR_S_RDY := ESD01.TRIP OR PSD31.TRIP OR MAINTENANCE OR BAL_IN_STBD OR BAL_IN_PORT OR DEBAL_IN_STBD OR DEBAL_IN_PORT OR DIAG_IN_SELF;
MODE_STRIP_S(
    START_COMMAND := MP_STRIP_ST_S,
    UNREADY := STR_S_RDY,
    RESET := STRIP_S_RESET,
    STOP_COMMAND := MP_STRIP_SP_S,
    SEQ_FAIL := SEQ311_FAIL); // BWTS.MODE
STR_ST_S := MODE_STRIP_S.START_OP;
STR_IN_STBD := MODE_STRIP_S.PROGRESS;
STR_SP_S := MODE_STRIP_S.STOP_OP;
SEQ311_FAIL := SST_S_01.TIMEOUT OR SST_S_02.TIMEOUT OR SST_S_04.TIMEOUT OR SST_S_08.TIMEOUT OR SST_S_09.TIMEOUT;
STRIP_S_RESET := ESD OR PSD_31 OR MST_SSP_S.COMPLETE;
DIAG_RDY := MAINTENANCE OR BAL_IN_STBD OR BAL_IN_PORT OR DEBAL_IN_STBD OR DEBAL_IN_PORT OR STR_IN_STBD OR ESD01.TRIP OR DIAG_IN_SELF;
MODE_DIAG(START_COMMAND := MP_DIAG_ST, UNREADY := DIAG_RDY, RESET := DIAG_RESET); // BWTS.MODE
DIAG_ST := MODE_DIAG.START_OP;
DIAG_IN_SELF := MODE_DIAG.PROGRESS;
DIAG_RESET := ESD OR MST_DIAG.COMPLETE;

END_PROGRAM

// Device/Application/Logic/2.Sequence/MASTER_SEQUENCE_BALLASTING
PROGRAM MASTER_SEQUENCE_BALLASTING
VAR
	TF_BST_RESET_S : TOF;
	TF_BST_RESET_P : TOF;

	TF_BSP_RESET_S : TOF;
	TF_BSP_RESET_P : TOF;

	TO_BSP_RESET_S : TON;
	TO_BSP_RESET_P : TON;

END_VAR
VAR // added by the converter: edge detectors and wires of the graphical bodies
    _w1, _w2 : ANY;
END_VAR

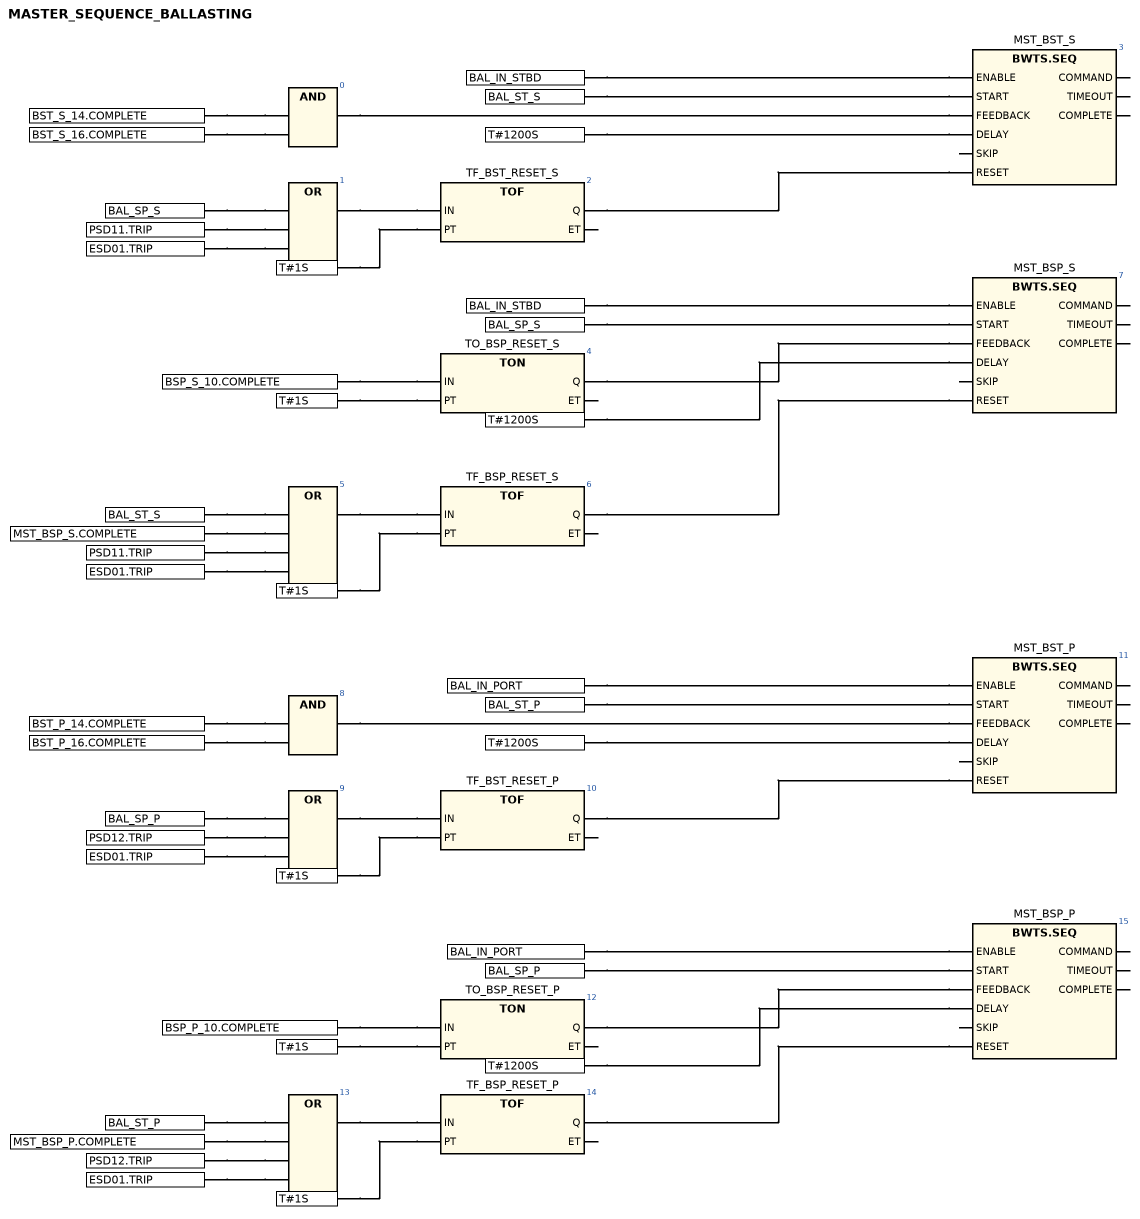
_w1 := BST_S_14.COMPLETE AND BST_S_16.COMPLETE;
TF_BST_RESET_S(IN := BAL_SP_S OR PSD11.TRIP OR ESD01.TRIP, PT := T#1S); // TOF
MST_BST_S(
    ENABLE := BAL_IN_STBD,
    START := BAL_ST_S,
    FEEDBACK := _w1,
    DELAY := T#1200S,
    RESET := TF_BST_RESET_S.Q); // BWTS.SEQ
TO_BSP_RESET_S(IN := BSP_S_10.COMPLETE, PT := T#1S); // TON
TF_BSP_RESET_S(IN := BAL_ST_S OR MST_BSP_S.COMPLETE OR PSD11.TRIP OR ESD01.TRIP, PT := T#1S); // TOF
MST_BSP_S(
    ENABLE := BAL_IN_STBD,
    START := BAL_SP_S,
    FEEDBACK := TO_BSP_RESET_S.Q,
    DELAY := T#1200S,
    RESET := TF_BSP_RESET_S.Q); // BWTS.SEQ
_w2 := BST_P_14.COMPLETE AND BST_P_16.COMPLETE;
TF_BST_RESET_P(IN := BAL_SP_P OR PSD12.TRIP OR ESD01.TRIP, PT := T#1S); // TOF
MST_BST_P(
    ENABLE := BAL_IN_PORT,
    START := BAL_ST_P,
    FEEDBACK := _w2,
    DELAY := T#1200S,
    RESET := TF_BST_RESET_P.Q); // BWTS.SEQ
TO_BSP_RESET_P(IN := BSP_P_10.COMPLETE, PT := T#1S); // TON
TF_BSP_RESET_P(IN := BAL_ST_P OR MST_BSP_P.COMPLETE OR PSD12.TRIP OR ESD01.TRIP, PT := T#1S); // TOF
MST_BSP_P(
    ENABLE := BAL_IN_PORT,
    START := BAL_SP_P,
    FEEDBACK := TO_BSP_RESET_P.Q,
    DELAY := T#1200S,
    RESET := TF_BSP_RESET_P.Q); // BWTS.SEQ

END_PROGRAM

// Device/Application/Logic/2.Sequence/MASTER_SEQUENCE_DEBALLASTING
PROGRAM MASTER_SEQUENCE_DEBALLASTING
VAR
	TF_DST_RESET_S: TOF;
	TF_DSP_RESET_S: TOF;
	TF_DST_RESET_P: TOF;
	TF_DSP_RESET_P: TOF;
	
	TO_DSP_RESET_S: TON;
	TO_DSP_RESET_P: TON;
	
END_VAR
VAR // added by the converter: edge detectors and wires of the graphical bodies
    _w1 : ANY;
END_VAR

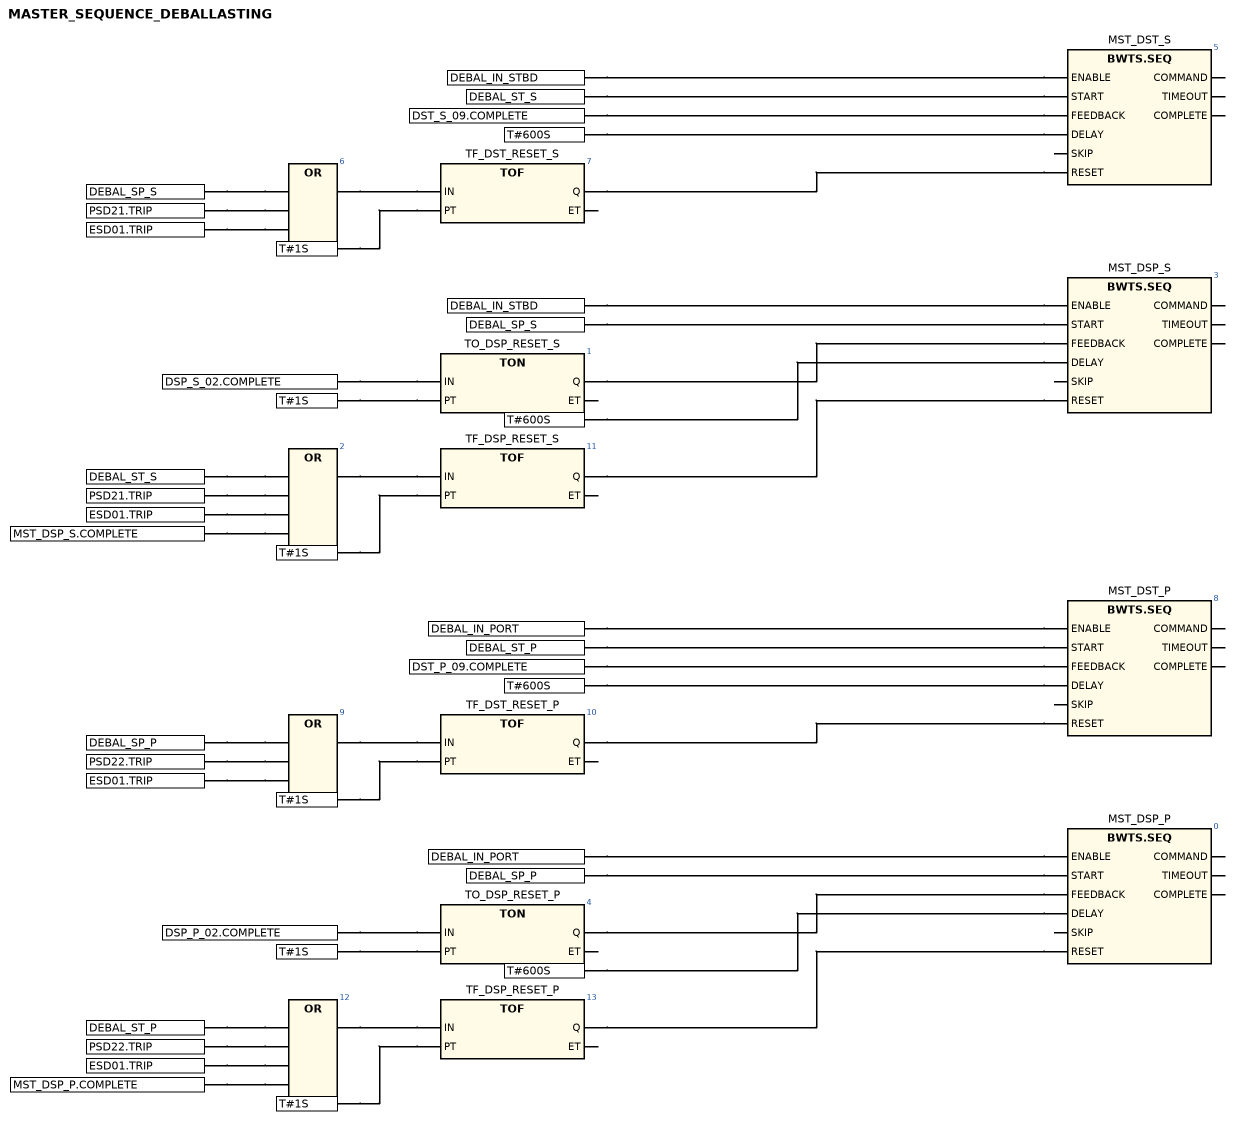
MST_DSP_P(
    ENABLE := DEBAL_IN_PORT,
    START := DEBAL_SP_P,
    FEEDBACK := TO_DSP_RESET_P.Q,
    DELAY := T#600S,
    RESET := TF_DSP_RESET_P.Q); // BWTS.SEQ
TO_DSP_RESET_S(IN := DSP_S_02.COMPLETE, PT := T#1S); // TON
_w1 := DEBAL_ST_S OR PSD21.TRIP OR ESD01.TRIP OR MST_DSP_S.COMPLETE;
MST_DSP_S(
    ENABLE := DEBAL_IN_STBD,
    START := DEBAL_SP_S,
    FEEDBACK := TO_DSP_RESET_S.Q,
    DELAY := T#600S,
    RESET := TF_DSP_RESET_S.Q); // BWTS.SEQ
TO_DSP_RESET_P(IN := DSP_P_02.COMPLETE, PT := T#1S); // TON
MST_DST_S(
    ENABLE := DEBAL_IN_STBD,
    START := DEBAL_ST_S,
    FEEDBACK := DST_S_09.COMPLETE,
    DELAY := T#600S,
    RESET := TF_DST_RESET_S.Q); // BWTS.SEQ
TF_DST_RESET_S(IN := DEBAL_SP_S OR PSD21.TRIP OR ESD01.TRIP, PT := T#1S); // TOF
MST_DST_P(
    ENABLE := DEBAL_IN_PORT,
    START := DEBAL_ST_P,
    FEEDBACK := DST_P_09.COMPLETE,
    DELAY := T#600S,
    RESET := TF_DST_RESET_P.Q); // BWTS.SEQ
TF_DST_RESET_P(IN := DEBAL_SP_P OR PSD22.TRIP OR ESD01.TRIP, PT := T#1S); // TOF
TF_DSP_RESET_S(IN := _w1, PT := T#1S); // TOF
TF_DSP_RESET_P(IN := DEBAL_ST_P OR PSD22.TRIP OR ESD01.TRIP OR MST_DSP_P.COMPLETE, PT := T#1S); // TOF

END_PROGRAM

// Device/Application/Logic/2.Sequence/MASTER_SEQUENCE_STRIPPING
PROGRAM MASTER_SEQUENCE_STRIPPING
VAR
	
	TF_SST_RESET_S: TOF;
	TF_SSP_RESET_S: TOF;
	TO_SSP_RESET_S: TON;
END_VAR
VAR // added by the converter: edge detectors and wires of the graphical bodies
    _w1 : ANY;
END_VAR

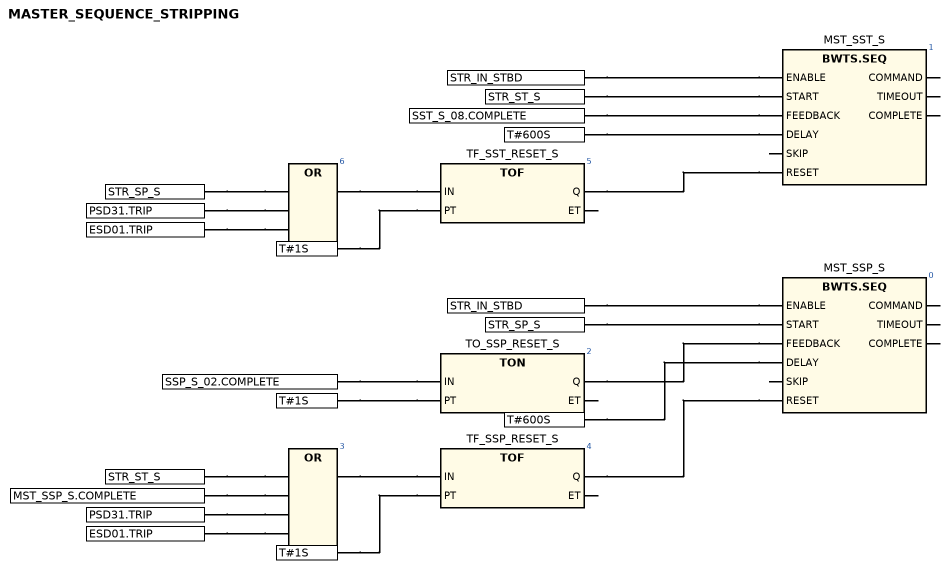
MST_SSP_S(
    ENABLE := STR_IN_STBD,
    START := STR_SP_S,
    FEEDBACK := TO_SSP_RESET_S.Q,
    DELAY := T#600S,
    RESET := TF_SSP_RESET_S.Q); // BWTS.SEQ
MST_SST_S(
    ENABLE := STR_IN_STBD,
    START := STR_ST_S,
    FEEDBACK := SST_S_08.COMPLETE,
    DELAY := T#600S,
    RESET := TF_SST_RESET_S.Q); // BWTS.SEQ
TO_SSP_RESET_S(IN := SSP_S_02.COMPLETE, PT := T#1S); // TON
TF_SSP_RESET_S(IN := STR_ST_S OR MST_SSP_S.COMPLETE OR PSD31.TRIP OR ESD01.TRIP, PT := T#1S); // TOF
TF_SST_RESET_S(IN := _w1, PT := T#1S); // TOF
_w1 := STR_SP_S OR PSD31.TRIP OR ESD01.TRIP;

END_PROGRAM

// Device/Application/Logic/2.Sequence/SEQ_BAL_SP_P
PROGRAM SEQ_BAL_SP_P
VAR
	TON_1: TON; // FLITER V/V CLOSING TIME
	TON_2: TON; // SEA WATER REPLACEMENT TIME
	TON_3: TON; // BLOWER SAFETY STOP TIME
	BST_S_ON: BOOL;;
END_VAR
VAR // added by the converter: edge detectors and wires of the graphical bodies
    _w1, _w2, _w3, _w4, _w5, _w6, _w7, _w8 : ANY;
END_VAR

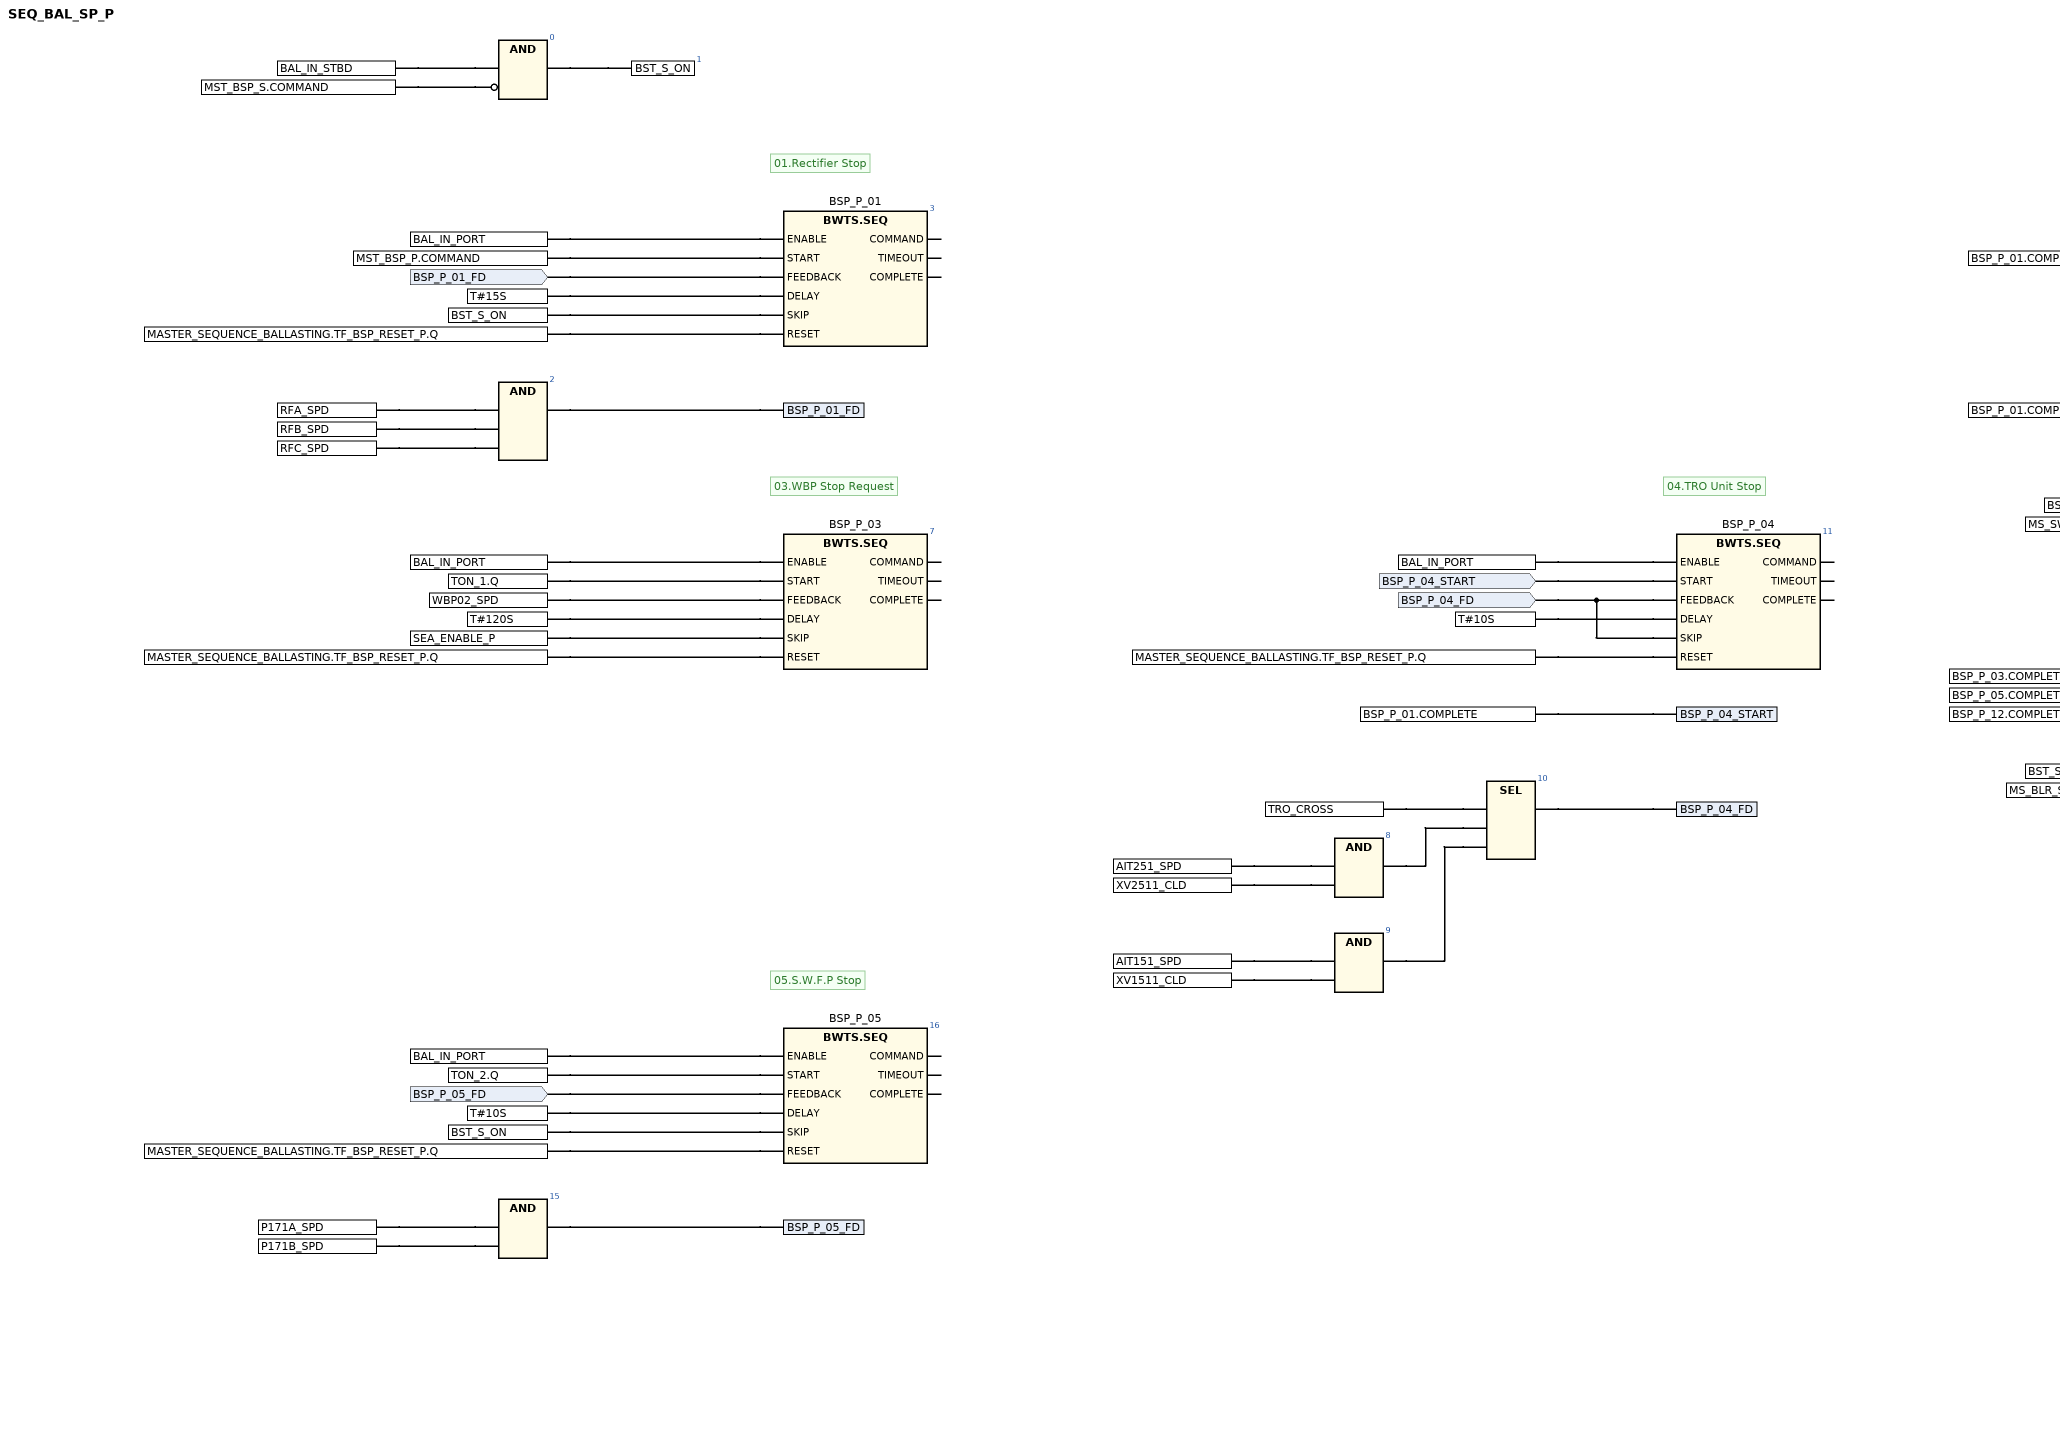
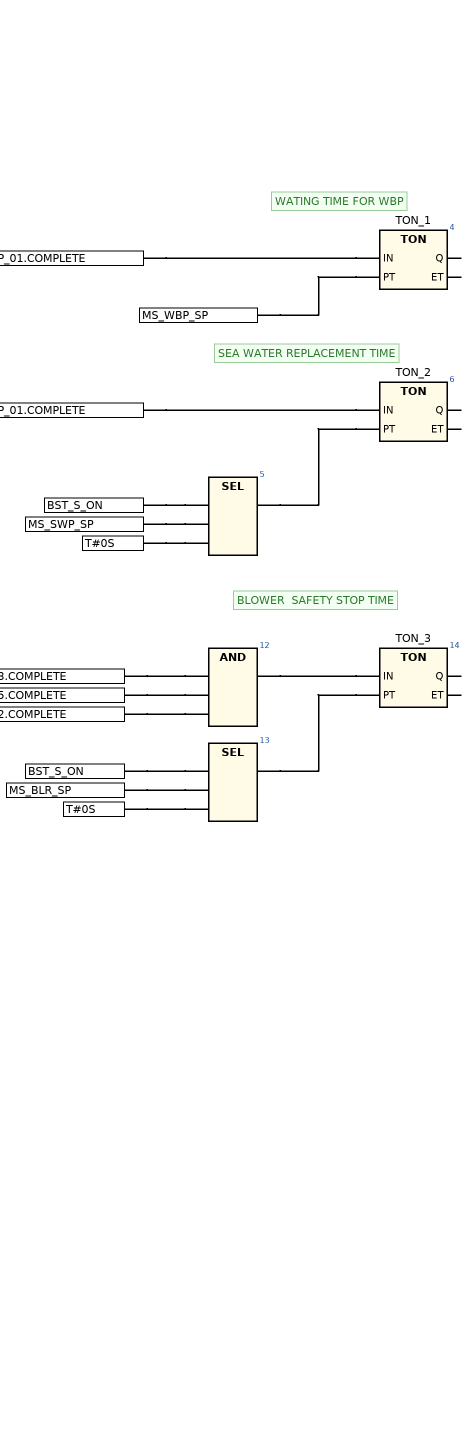
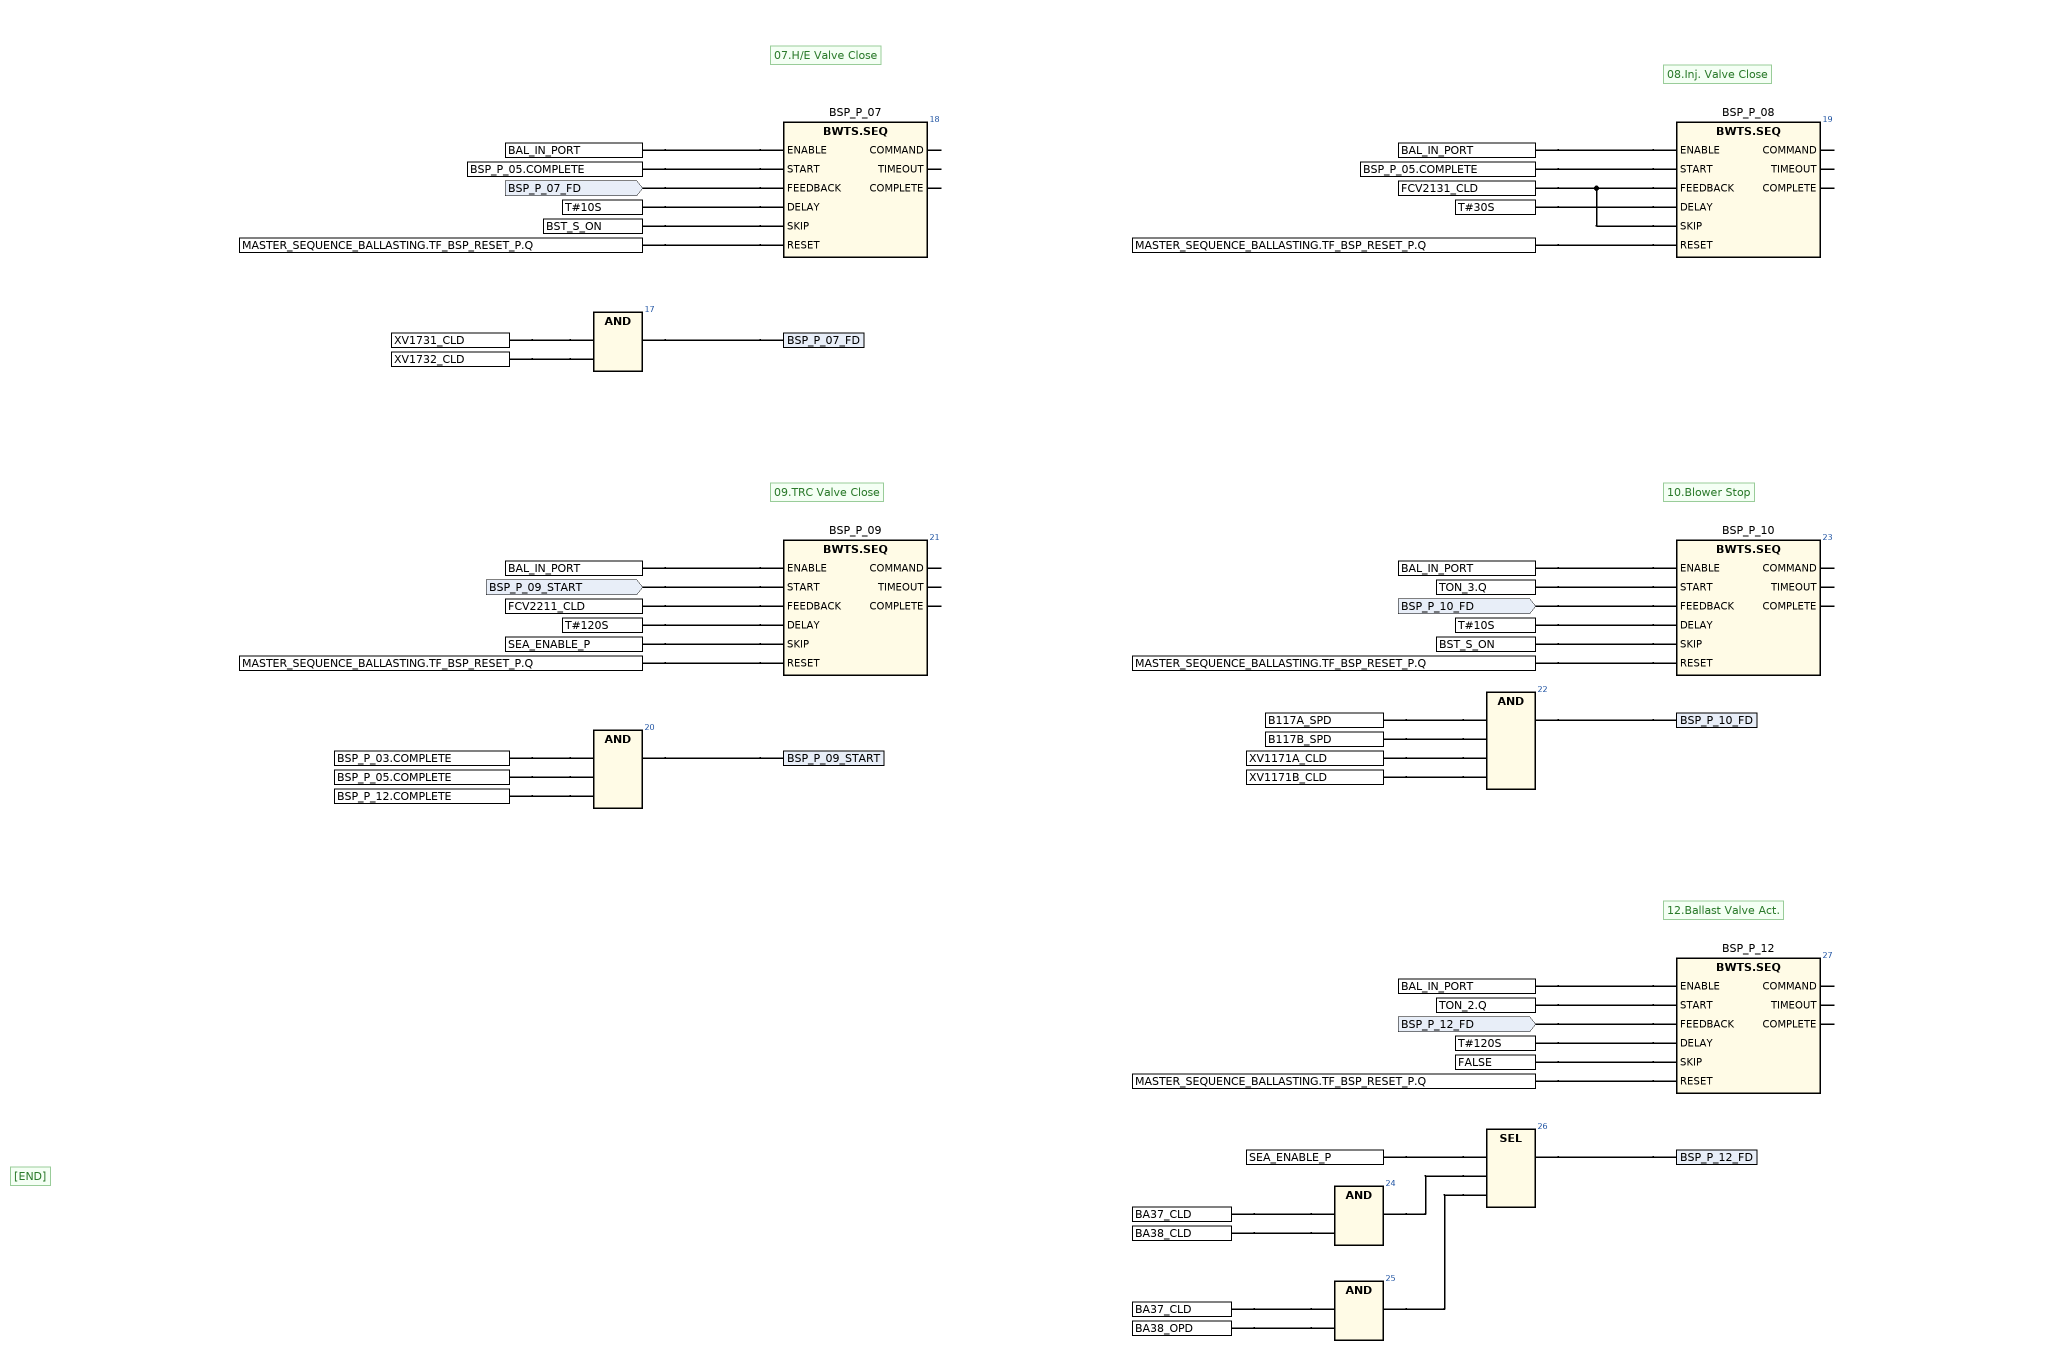
BST_S_ON := BAL_IN_STBD AND NOT MST_BSP_S.COMMAND;
(* RFA_SPD AND RFB_SPD AND RFC_SPD; result not used *)
// 01.Rectifier Stop
BSP_P_01(
    ENABLE := BAL_IN_PORT,
    START := MST_BSP_P.COMMAND,
    FEEDBACK := _w1,
    DELAY := T#15S,
    SKIP := BST_S_ON,
    RESET := MASTER_SEQUENCE_BALLASTING.TF_BSP_RESET_P.Q); // BWTS.SEQ
// WATING TIME FOR WBP
TON_1(IN := BSP_P_01.COMPLETE, PT := MS_WBP_SP); // TON
// SEA WATER REPLACEMENT TIME
TON_2(IN := BSP_P_01.COMPLETE, PT := SEL(BST_S_ON, MS_SWP_SP, T#0S)); // TON
// 03.WBP Stop Request
BSP_P_03(
    ENABLE := BAL_IN_PORT,
    START := TON_1.Q,
    FEEDBACK := WBP02_SPD,
    DELAY := T#120S,
    SKIP := SEA_ENABLE_P,
    RESET := MASTER_SEQUENCE_BALLASTING.TF_BSP_RESET_P.Q); // BWTS.SEQ
(* SEL(TRO_CROSS, AIT251_SPD AND XV2511_CLD, AIT151_SPD AND XV1511_CLD); result not used *)
// 04.TRO Unit Stop
BSP_P_04(
    ENABLE := BAL_IN_PORT,
    START := _w2,
    FEEDBACK := _w3,
    DELAY := T#10S,
    SKIP := _w3,
    RESET := MASTER_SEQUENCE_BALLASTING.TF_BSP_RESET_P.Q); // BWTS.SEQ
// BLOWER  SAFETY STOP TIME
TON_3(IN := BSP_P_03.COMPLETE AND BSP_P_05.COMPLETE AND BSP_P_12.COMPLETE, PT := SEL(BST_S_ON, MS_BLR_SP, T#0S)); // TON
(* P171A_SPD AND P171B_SPD; result not used *)
// 05.S.W.F.P Stop
BSP_P_05(
    ENABLE := BAL_IN_PORT,
    START := TON_2.Q,
    FEEDBACK := _w4,
    DELAY := T#10S,
    SKIP := BST_S_ON,
    RESET := MASTER_SEQUENCE_BALLASTING.TF_BSP_RESET_P.Q); // BWTS.SEQ
(* XV1731_CLD AND XV1732_CLD; result not used *)
// 07.H/E Valve Close
BSP_P_07(
    ENABLE := BAL_IN_PORT,
    START := BSP_P_05.COMPLETE,
    FEEDBACK := _w5,
    DELAY := T#10S,
    SKIP := BST_S_ON,
    RESET := MASTER_SEQUENCE_BALLASTING.TF_BSP_RESET_P.Q); // BWTS.SEQ
// 08.Inj. Valve Close
BSP_P_08(
    ENABLE := BAL_IN_PORT,
    START := BSP_P_05.COMPLETE,
    FEEDBACK := FCV2131_CLD,
    DELAY := T#30S,
    SKIP := FCV2131_CLD,
    RESET := MASTER_SEQUENCE_BALLASTING.TF_BSP_RESET_P.Q); // BWTS.SEQ
(* BSP_P_03.COMPLETE AND BSP_P_05.COMPLETE AND BSP_P_12.COMPLETE; result not used *)
// 09.TRC Valve Close
BSP_P_09(
    ENABLE := BAL_IN_PORT,
    START := _w6,
    FEEDBACK := FCV2211_CLD,
    DELAY := T#120S,
    SKIP := SEA_ENABLE_P,
    RESET := MASTER_SEQUENCE_BALLASTING.TF_BSP_RESET_P.Q); // BWTS.SEQ
(* B117A_SPD AND B117B_SPD AND XV1171A_CLD AND XV1171B_CLD; result not used *)
// 10.Blower Stop
BSP_P_10(
    ENABLE := BAL_IN_PORT,
    START := TON_3.Q,
    FEEDBACK := _w7,
    DELAY := T#10S,
    SKIP := BST_S_ON,
    RESET := MASTER_SEQUENCE_BALLASTING.TF_BSP_RESET_P.Q); // BWTS.SEQ
// [END]
(* SEL(SEA_ENABLE_P, BA37_CLD AND BA38_CLD, BA37_CLD AND BA38_OPD); result not used *)
// 12.Ballast Valve Act.
BSP_P_12(
    ENABLE := BAL_IN_PORT,
    START := TON_2.Q,
    FEEDBACK := _w8,
    DELAY := T#120S,
    SKIP := FALSE,
    RESET := MASTER_SEQUENCE_BALLASTING.TF_BSP_RESET_P.Q); // BWTS.SEQ

END_PROGRAM

// Device/Application/Logic/2.Sequence/SEQ_BAL_SP_S
PROGRAM SEQ_BAL_SP_S
VAR
	TON_1: TON; // FLITER V/V CLOSING TIME
	TON_2: TON; // SEA WATER REPLACEMENT TIME
	TON_3: TON; // BLOWER SAFETY STOP TIME
	BST_P_ON: BOOL;;
END_VAR
VAR // added by the converter: edge detectors and wires of the graphical bodies
    _w1, _w2, _w3, _w4, _w5, _w6, _w7, _w8 : ANY;
END_VAR

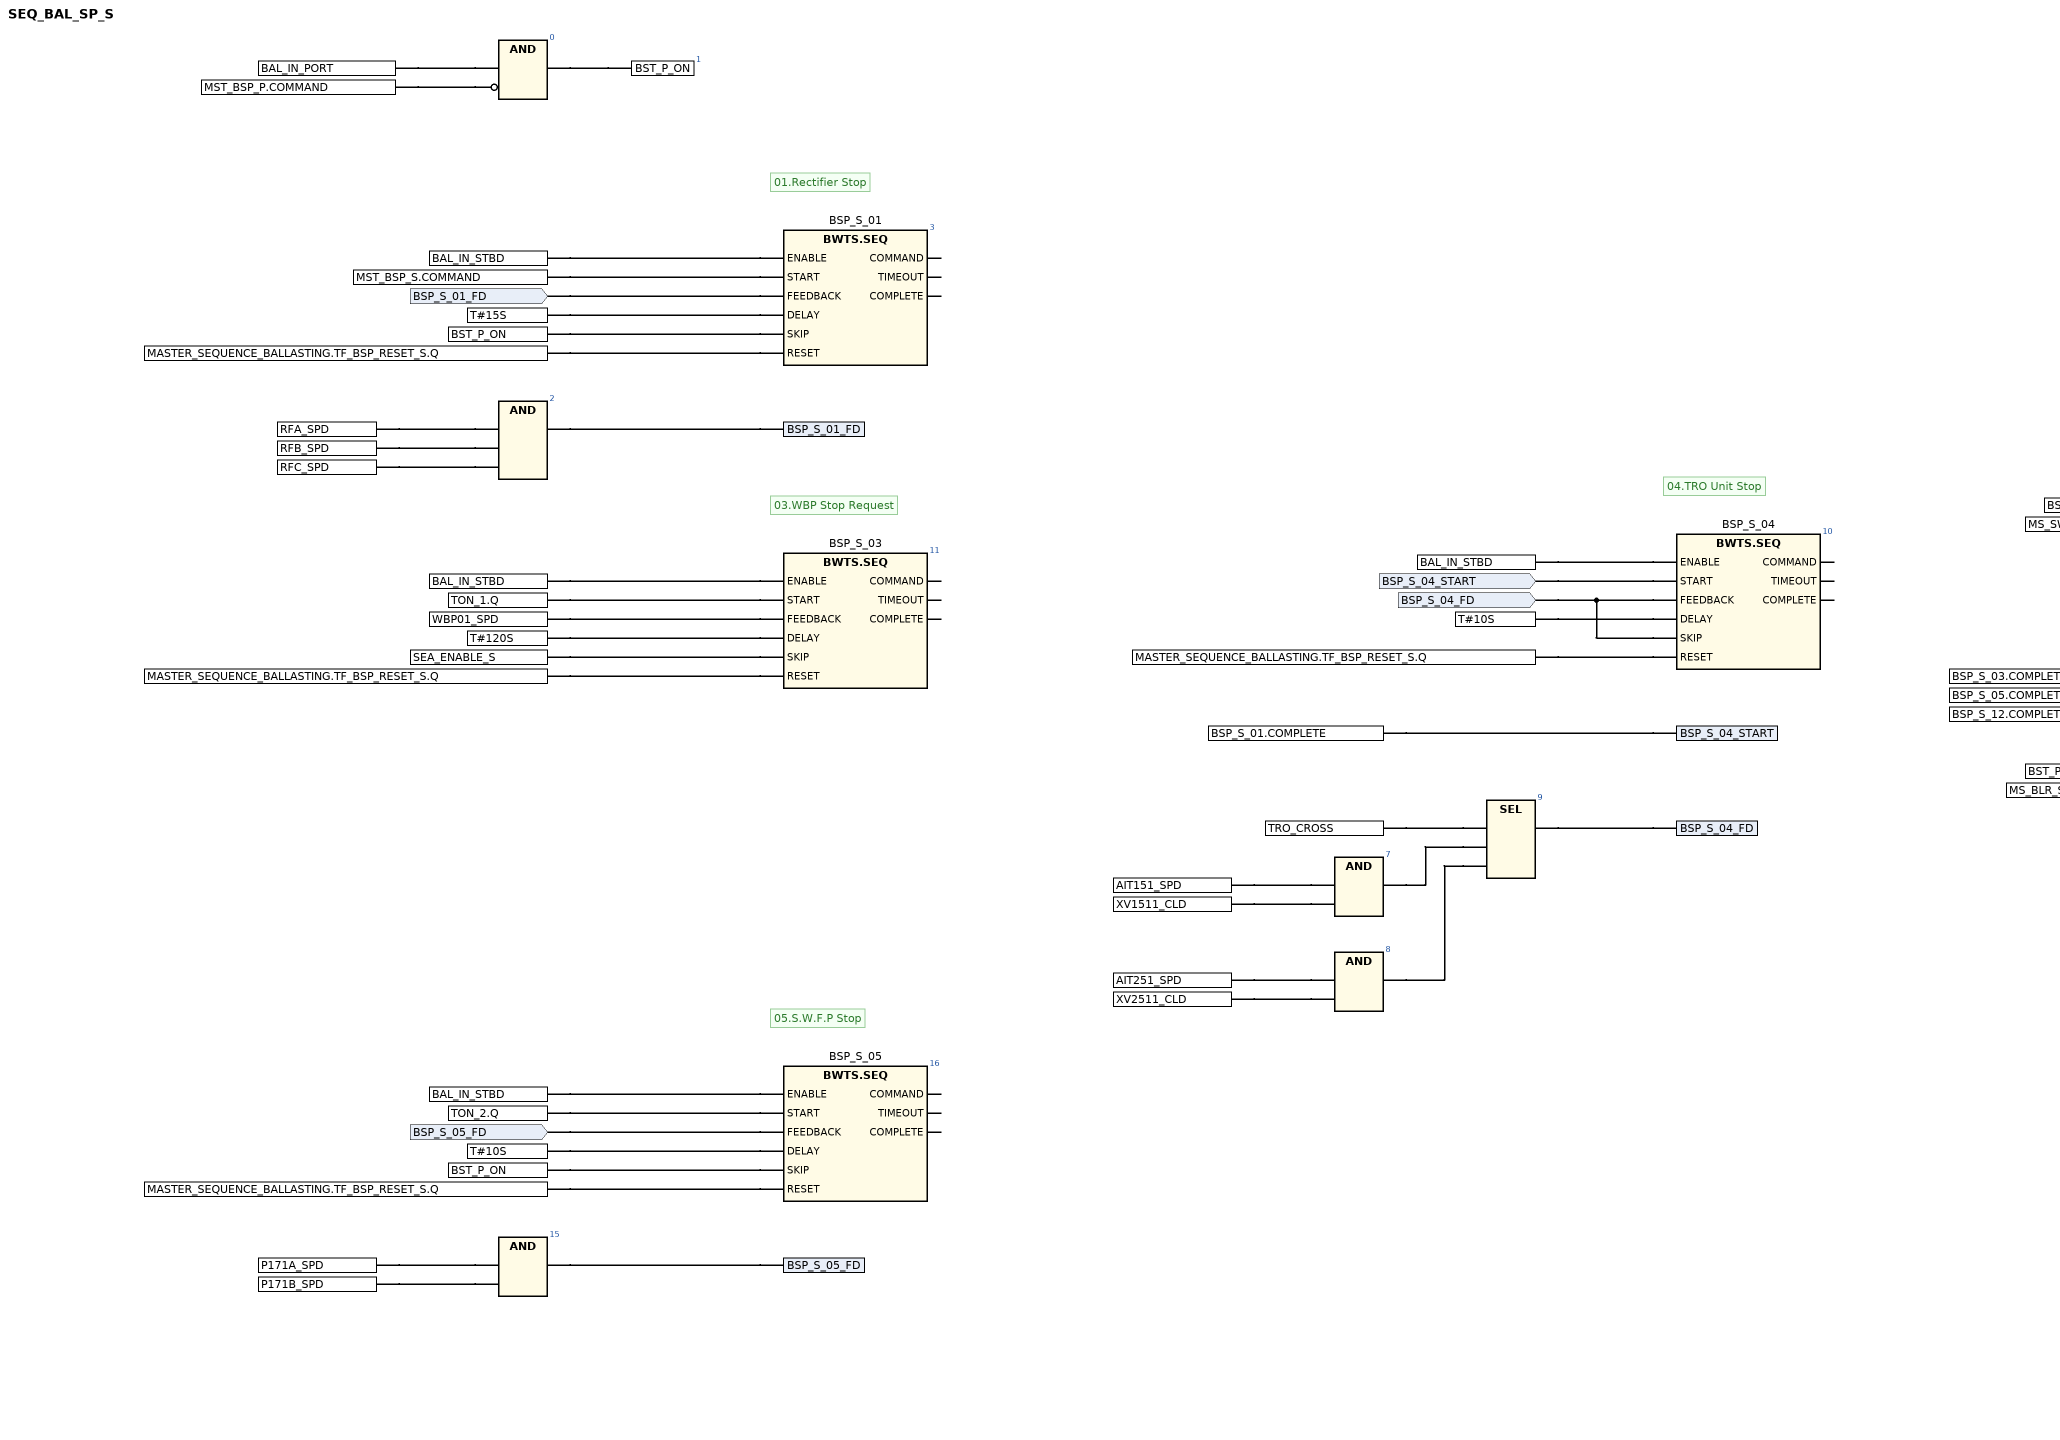
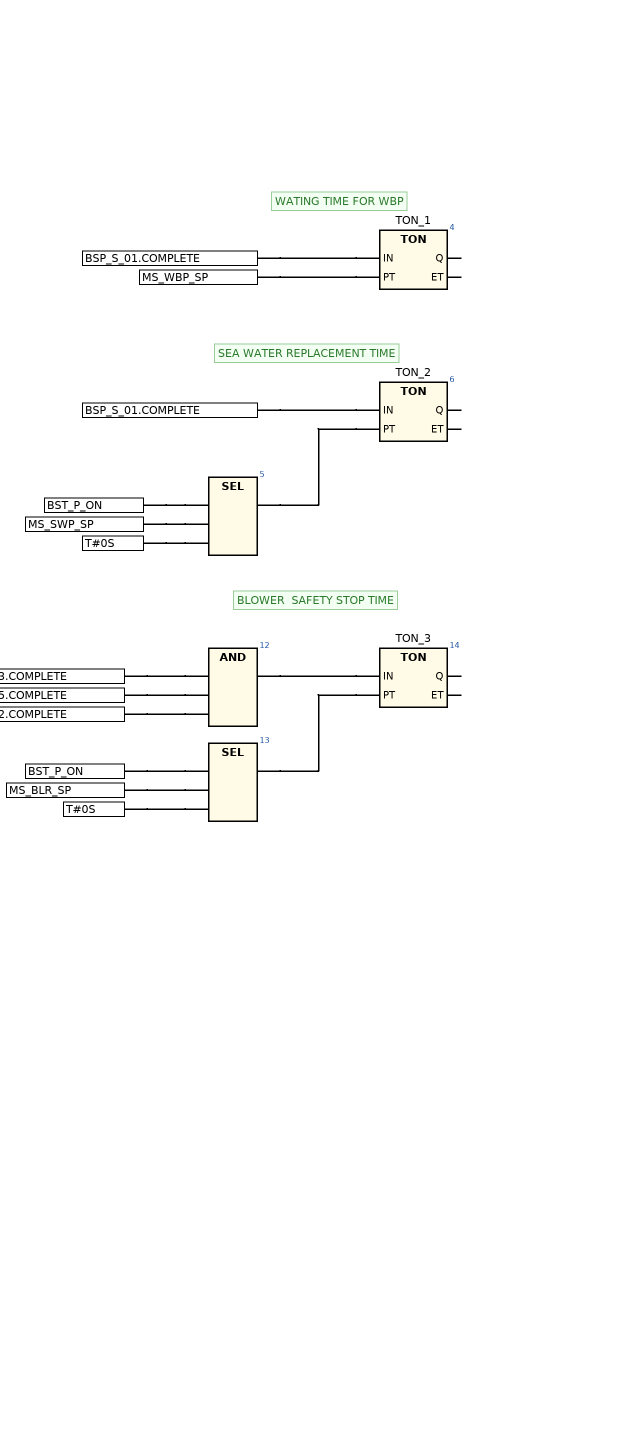
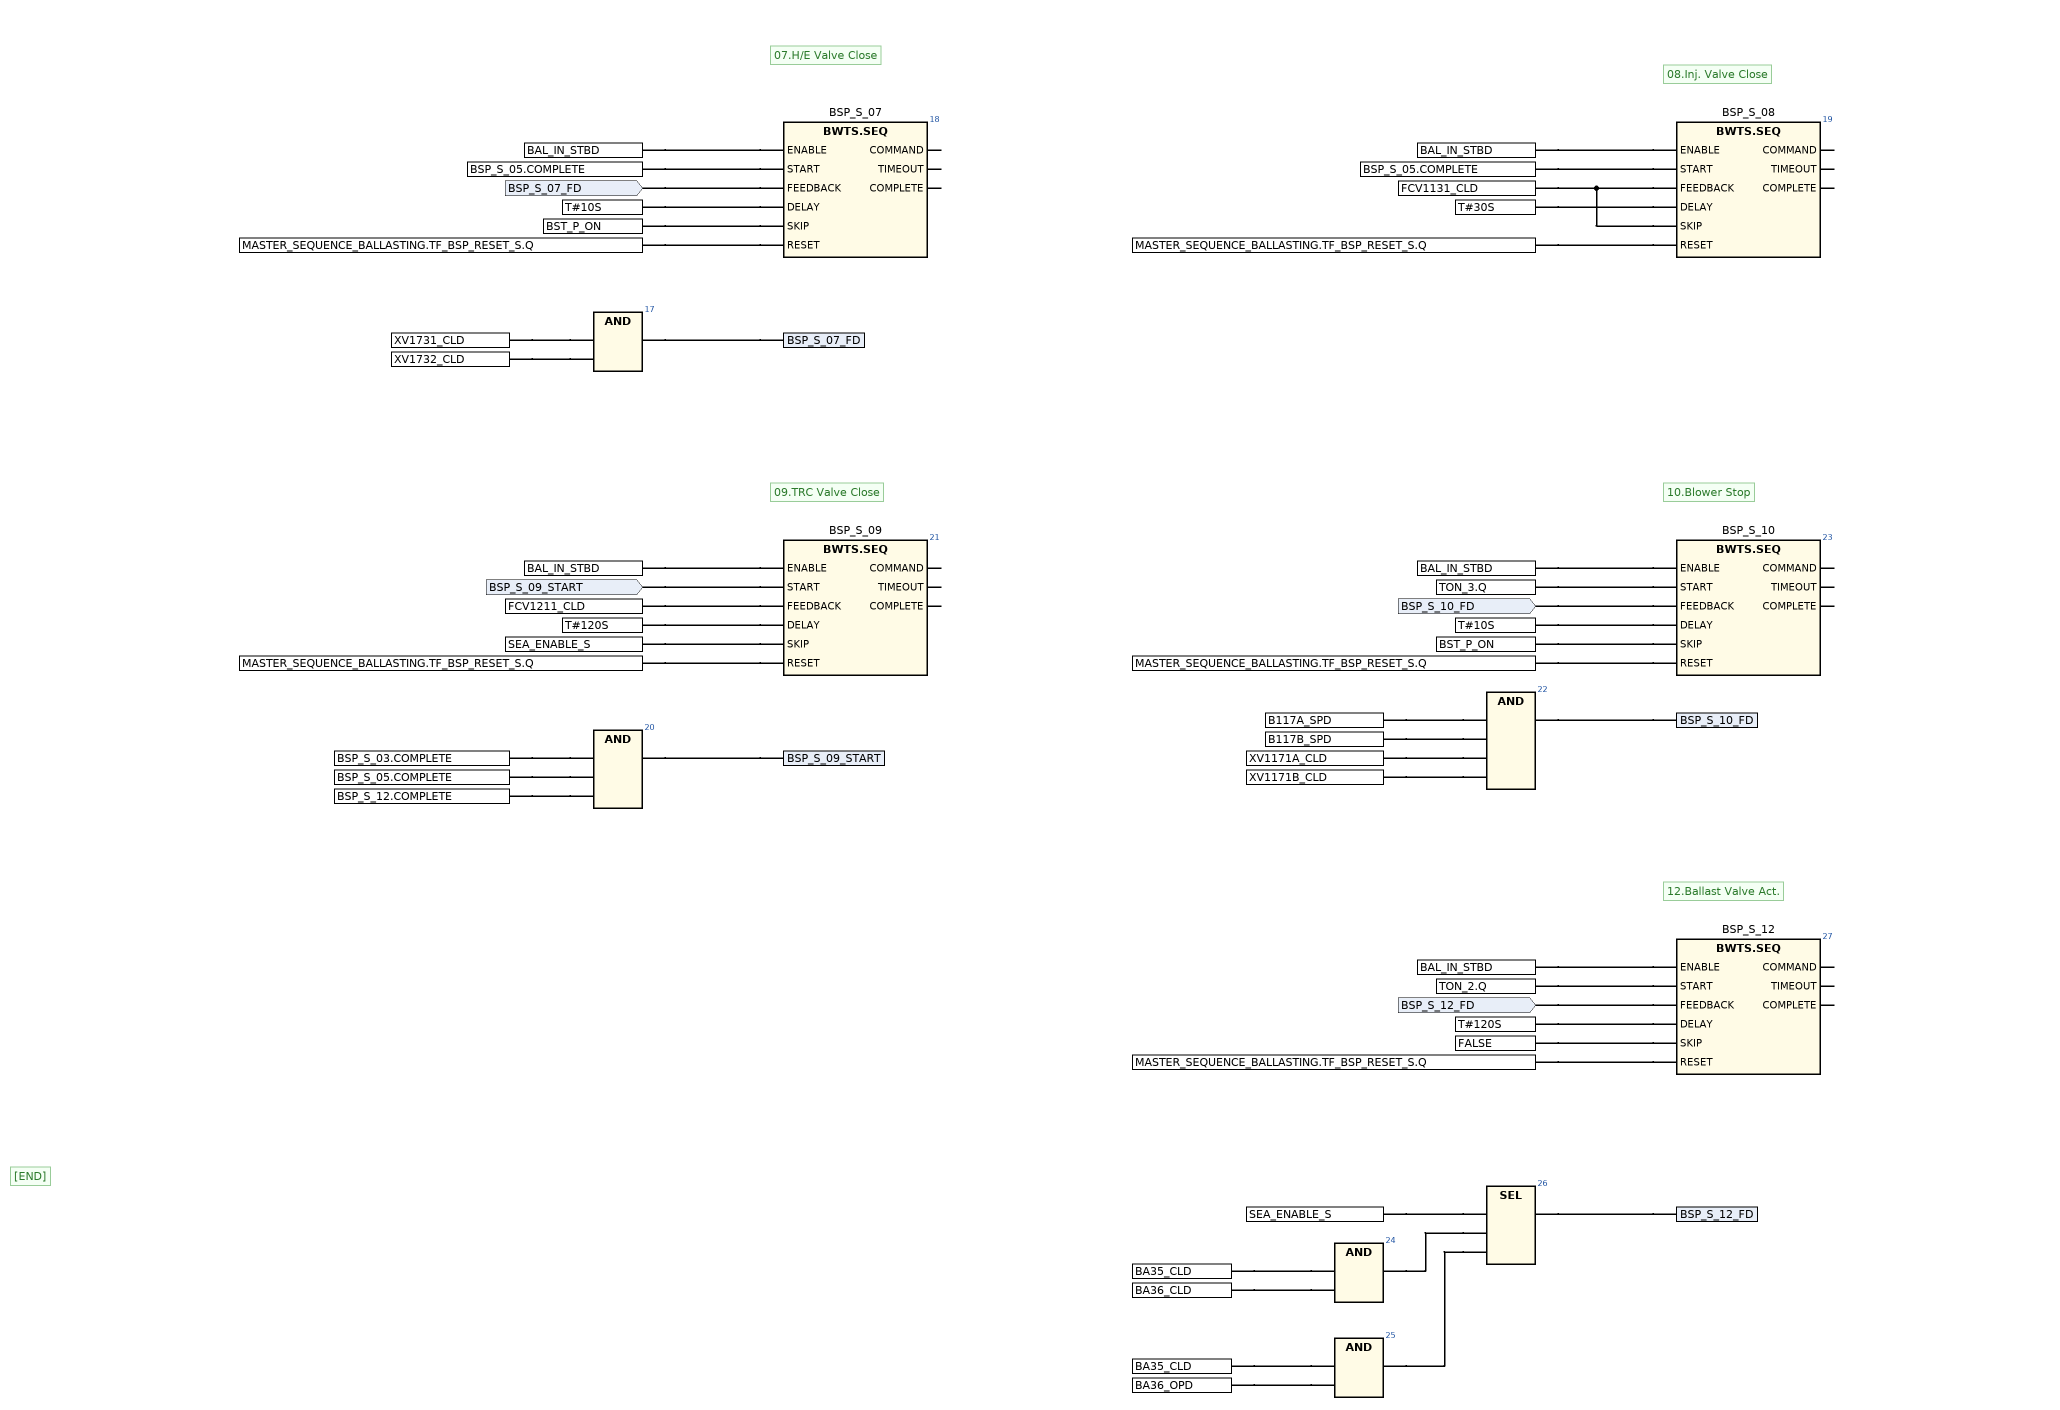
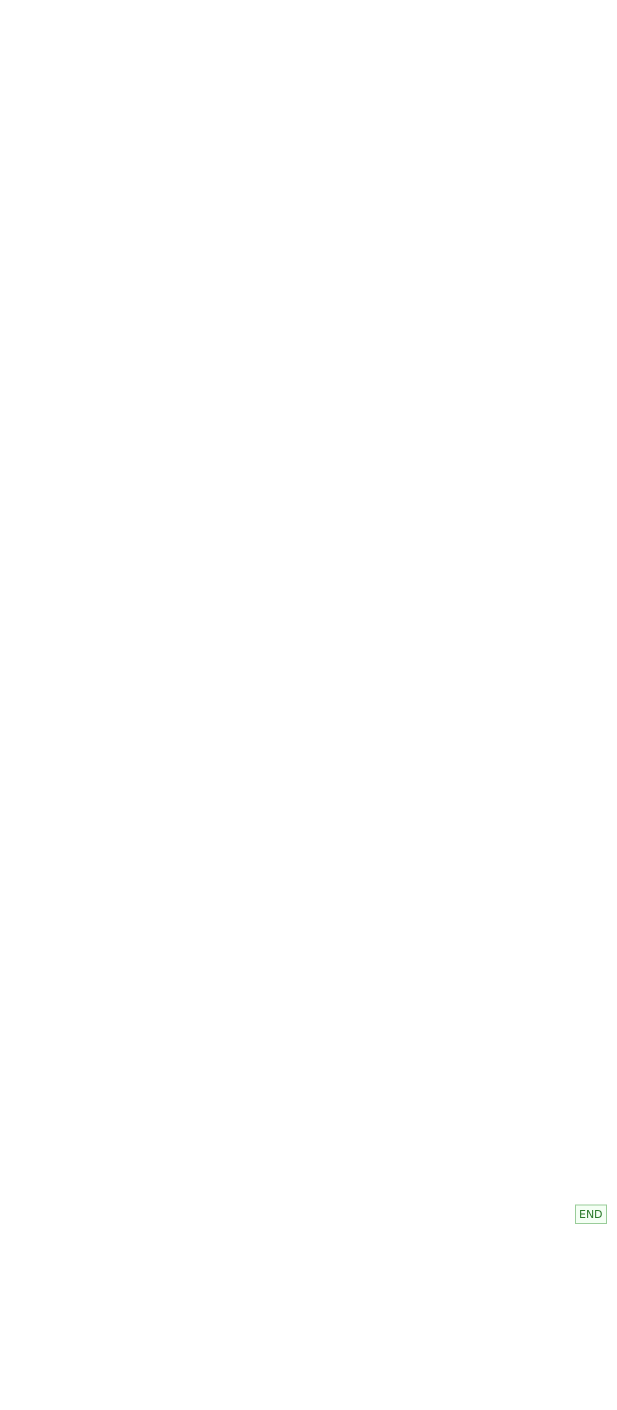
BST_P_ON := BAL_IN_PORT AND NOT MST_BSP_P.COMMAND;
(* RFA_SPD AND RFB_SPD AND RFC_SPD; result not used *)
// 01.Rectifier Stop
BSP_S_01(
    ENABLE := BAL_IN_STBD,
    START := MST_BSP_S.COMMAND,
    FEEDBACK := _w1,
    DELAY := T#15S,
    SKIP := BST_P_ON,
    RESET := MASTER_SEQUENCE_BALLASTING.TF_BSP_RESET_S.Q); // BWTS.SEQ
// WATING TIME FOR WBP
TON_1(IN := BSP_S_01.COMPLETE, PT := MS_WBP_SP); // TON
// SEA WATER REPLACEMENT TIME
TON_2(IN := BSP_S_01.COMPLETE, PT := SEL(BST_P_ON, MS_SWP_SP, T#0S)); // TON
(* SEL(TRO_CROSS, AIT151_SPD AND XV1511_CLD, AIT251_SPD AND XV2511_CLD); result not used *)
// 04.TRO Unit Stop
BSP_S_04(
    ENABLE := BAL_IN_STBD,
    START := _w2,
    FEEDBACK := _w3,
    DELAY := T#10S,
    SKIP := _w3,
    RESET := MASTER_SEQUENCE_BALLASTING.TF_BSP_RESET_S.Q); // BWTS.SEQ
// 03.WBP Stop Request
BSP_S_03(
    ENABLE := BAL_IN_STBD,
    START := TON_1.Q,
    FEEDBACK := WBP01_SPD,
    DELAY := T#120S,
    SKIP := SEA_ENABLE_S,
    RESET := MASTER_SEQUENCE_BALLASTING.TF_BSP_RESET_S.Q); // BWTS.SEQ
// BLOWER  SAFETY STOP TIME
TON_3(IN := BSP_S_03.COMPLETE AND BSP_S_05.COMPLETE AND BSP_S_12.COMPLETE, PT := SEL(BST_P_ON, MS_BLR_SP, T#0S)); // TON
(* P171A_SPD AND P171B_SPD; result not used *)
// 05.S.W.F.P Stop
BSP_S_05(
    ENABLE := BAL_IN_STBD,
    START := TON_2.Q,
    FEEDBACK := _w4,
    DELAY := T#10S,
    SKIP := BST_P_ON,
    RESET := MASTER_SEQUENCE_BALLASTING.TF_BSP_RESET_S.Q); // BWTS.SEQ
(* XV1731_CLD AND XV1732_CLD; result not used *)
// 07.H/E Valve Close
BSP_S_07(
    ENABLE := BAL_IN_STBD,
    START := BSP_S_05.COMPLETE,
    FEEDBACK := _w5,
    DELAY := T#10S,
    SKIP := BST_P_ON,
    RESET := MASTER_SEQUENCE_BALLASTING.TF_BSP_RESET_S.Q); // BWTS.SEQ
// 08.Inj. Valve Close
BSP_S_08(
    ENABLE := BAL_IN_STBD,
    START := BSP_S_05.COMPLETE,
    FEEDBACK := FCV1131_CLD,
    DELAY := T#30S,
    SKIP := FCV1131_CLD,
    RESET := MASTER_SEQUENCE_BALLASTING.TF_BSP_RESET_S.Q); // BWTS.SEQ
(* BSP_S_03.COMPLETE AND BSP_S_05.COMPLETE AND BSP_S_12.COMPLETE; result not used *)
// 09.TRC Valve Close
BSP_S_09(
    ENABLE := BAL_IN_STBD,
    START := _w6,
    FEEDBACK := FCV1211_CLD,
    DELAY := T#120S,
    SKIP := SEA_ENABLE_S,
    RESET := MASTER_SEQUENCE_BALLASTING.TF_BSP_RESET_S.Q); // BWTS.SEQ
(* B117A_SPD AND B117B_SPD AND XV1171A_CLD AND XV1171B_CLD; result not used *)
// 10.Blower Stop
BSP_S_10(
    ENABLE := BAL_IN_STBD,
    START := TON_3.Q,
    FEEDBACK := _w7,
    DELAY := T#10S,
    SKIP := BST_P_ON,
    RESET := MASTER_SEQUENCE_BALLASTING.TF_BSP_RESET_S.Q); // BWTS.SEQ
// [END]
// END
(* SEL(SEA_ENABLE_S, BA35_CLD AND BA36_CLD, BA35_CLD AND BA36_OPD); result not used *)
// 12.Ballast Valve Act.
BSP_S_12(
    ENABLE := BAL_IN_STBD,
    START := TON_2.Q,
    FEEDBACK := _w8,
    DELAY := T#120S,
    SKIP := FALSE,
    RESET := MASTER_SEQUENCE_BALLASTING.TF_BSP_RESET_S.Q); // BWTS.SEQ

END_PROGRAM

// Device/Application/Logic/2.Sequence/SEQ_BAL_ST_P
PROGRAM SEQ_BAL_ST_P
VAR
	TON_1 : TON;		// BLOWER PRE RUNNING TIME
	TON_2 : TON;		// SWFP RUNNING WAITING TIME
	TON_3 : TON;		// TRO RUNNING WAITING TIME
END_VAR
VAR // added by the converter: edge detectors and wires of the graphical bodies
    _w1, _w2, _w3, _w4, _w5, _w6, _w7, _w8 : ANY;
END_VAR

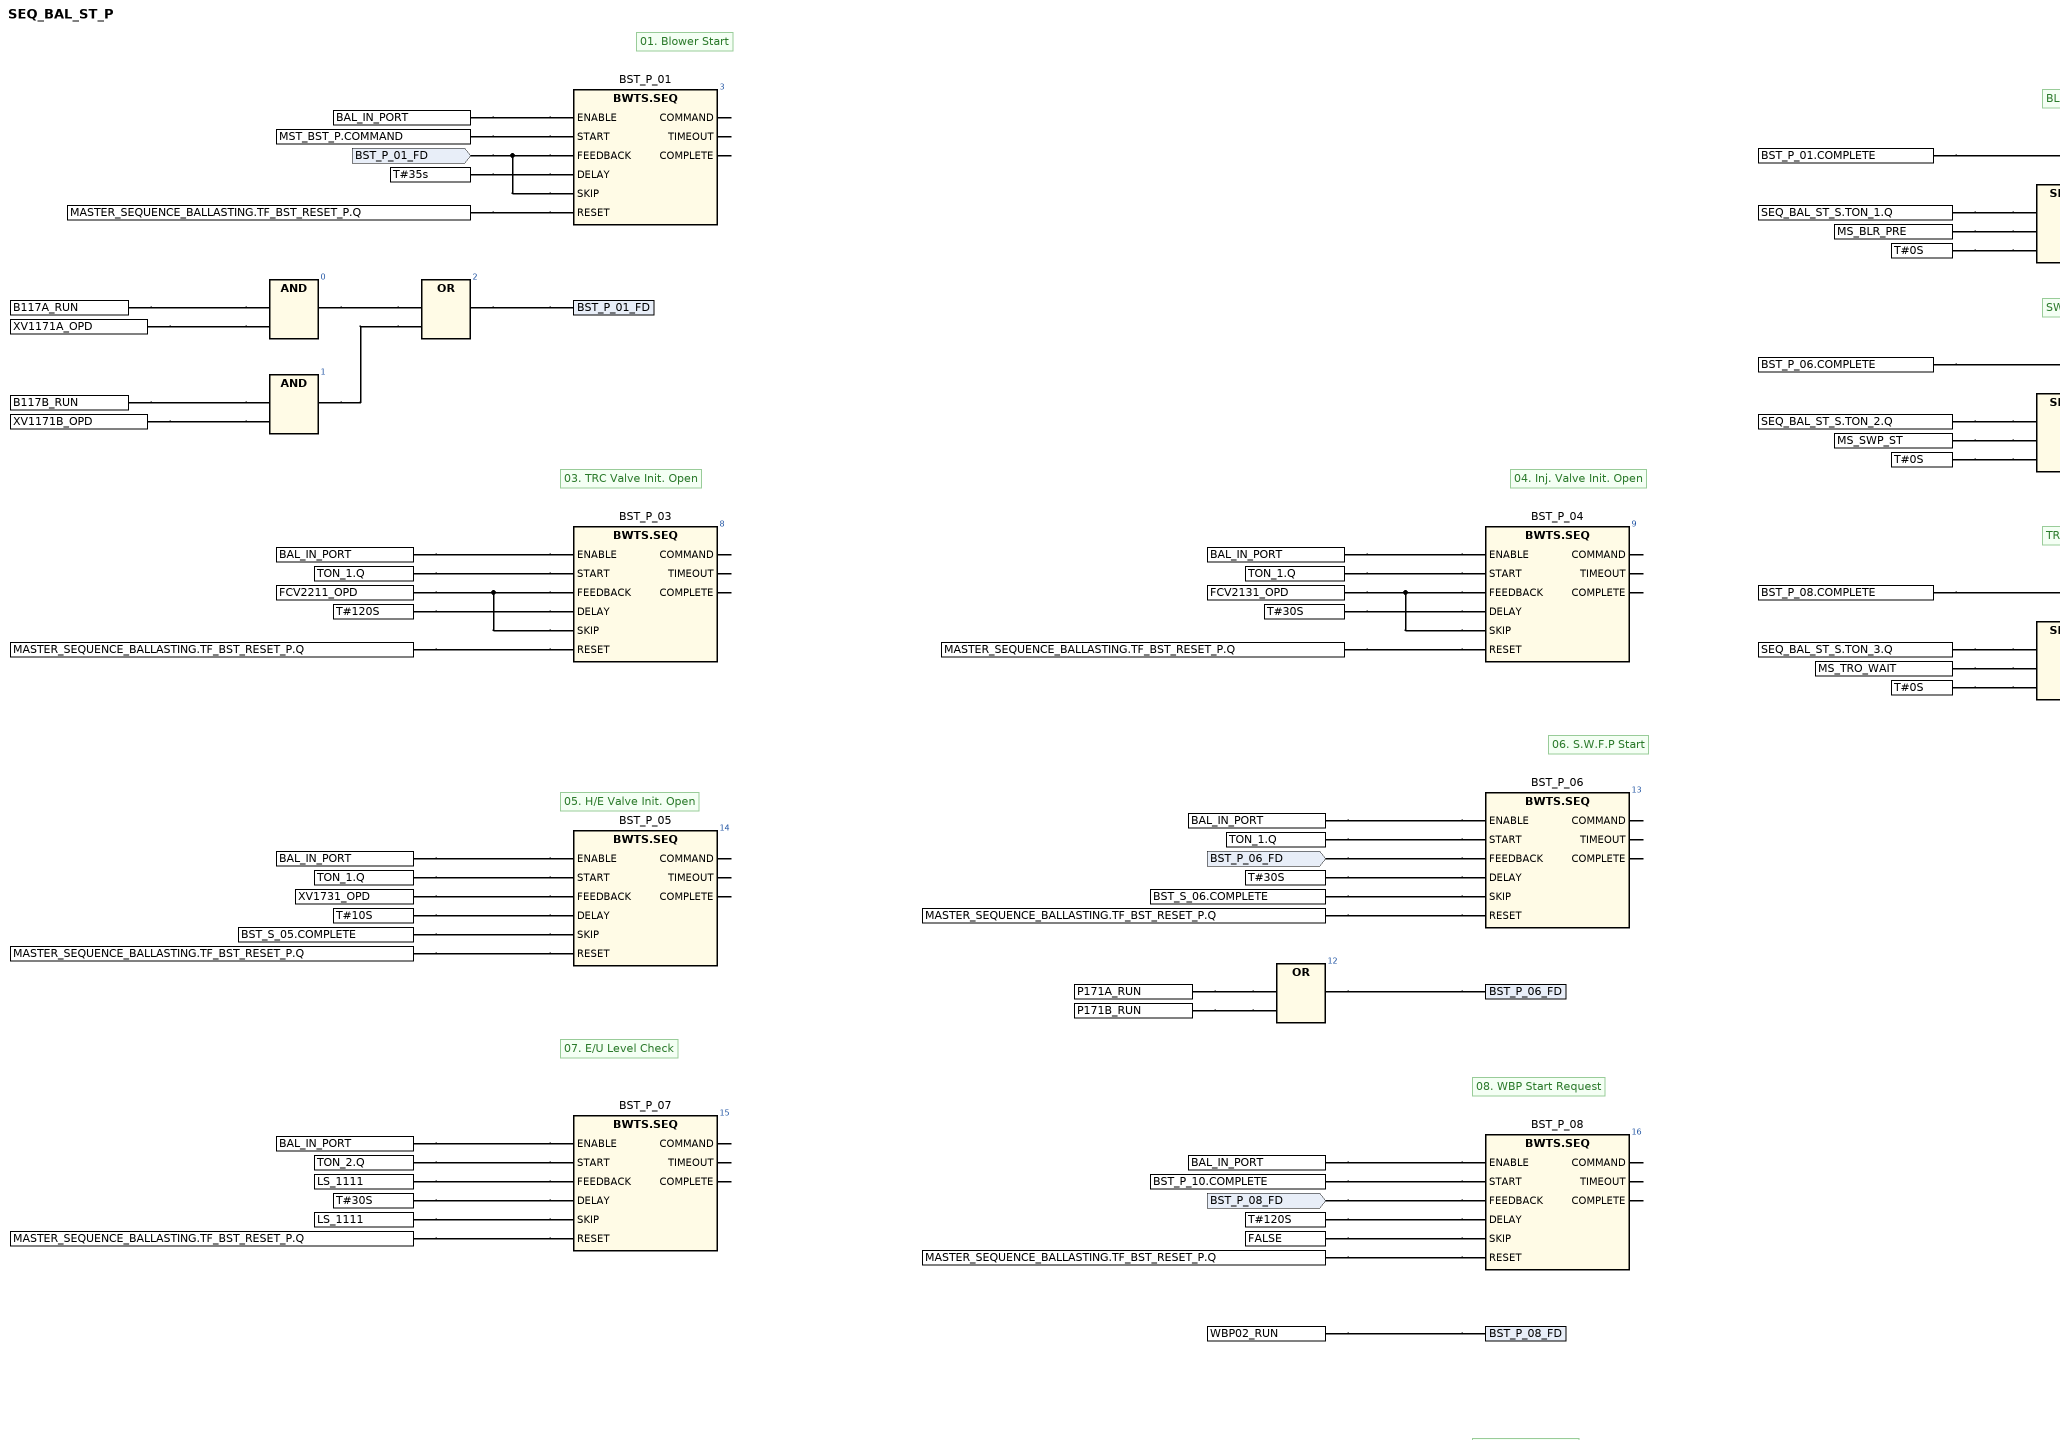
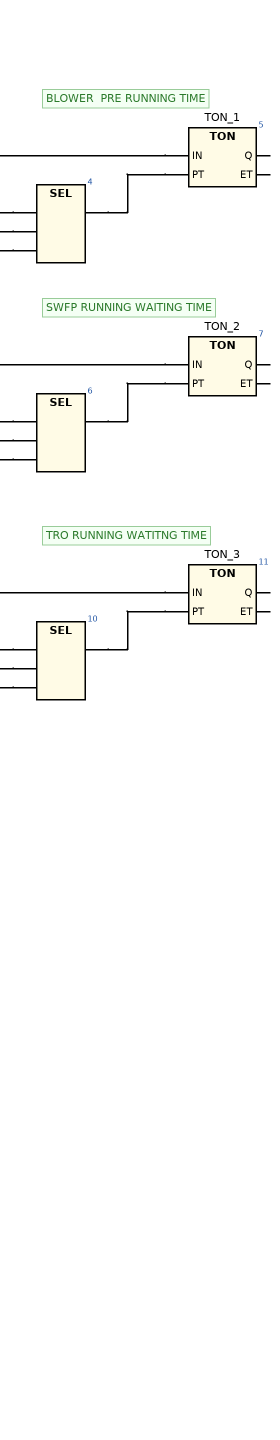
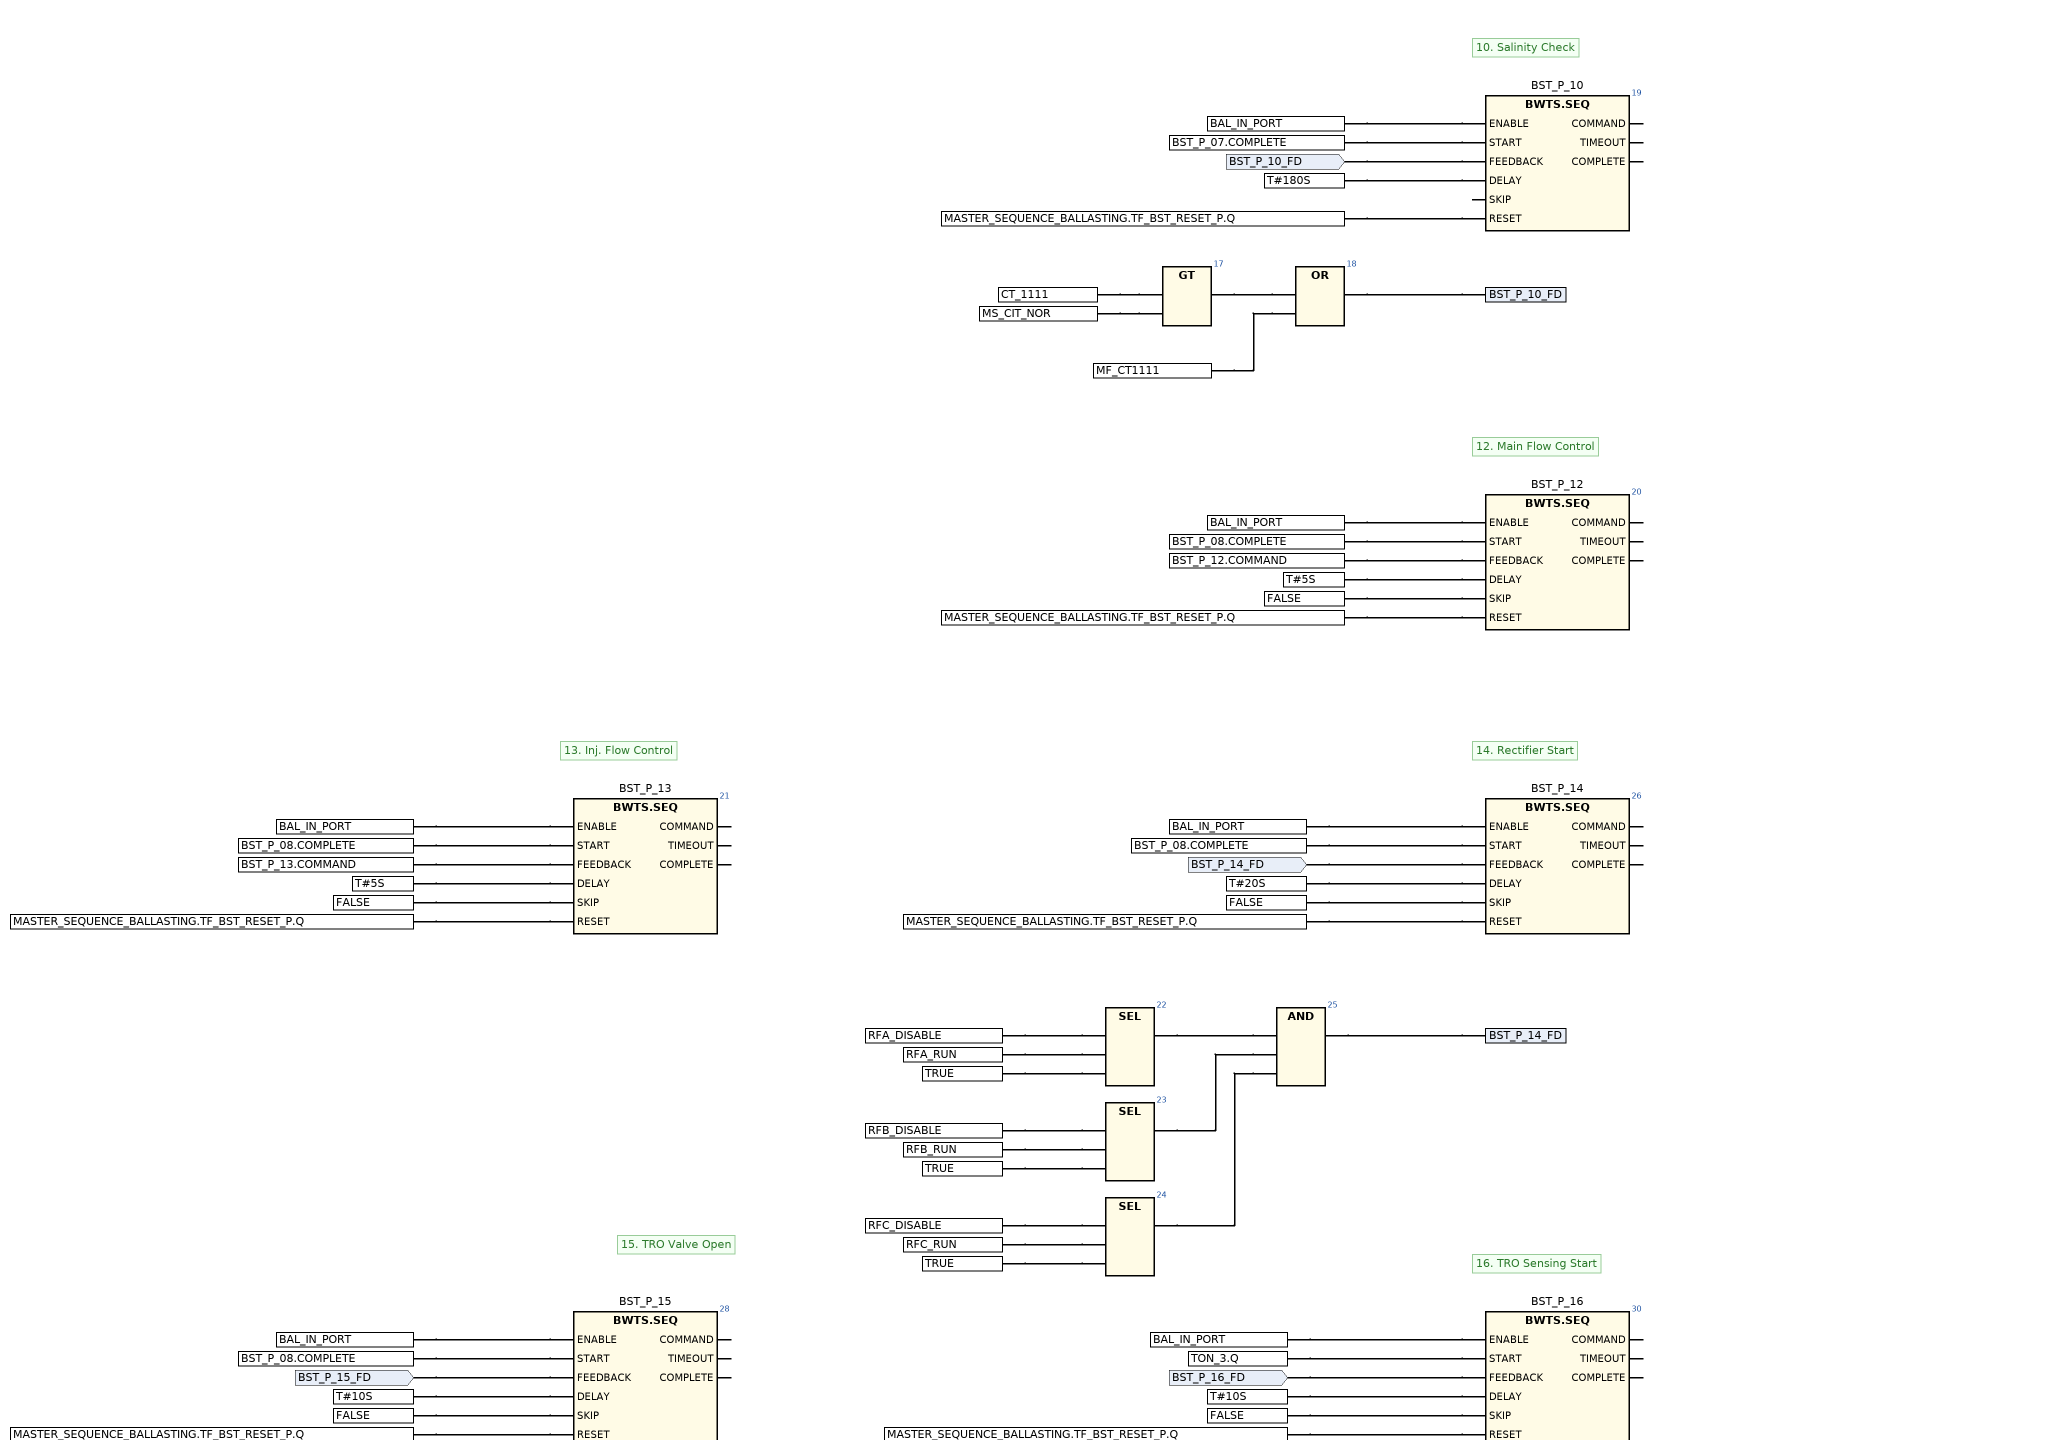
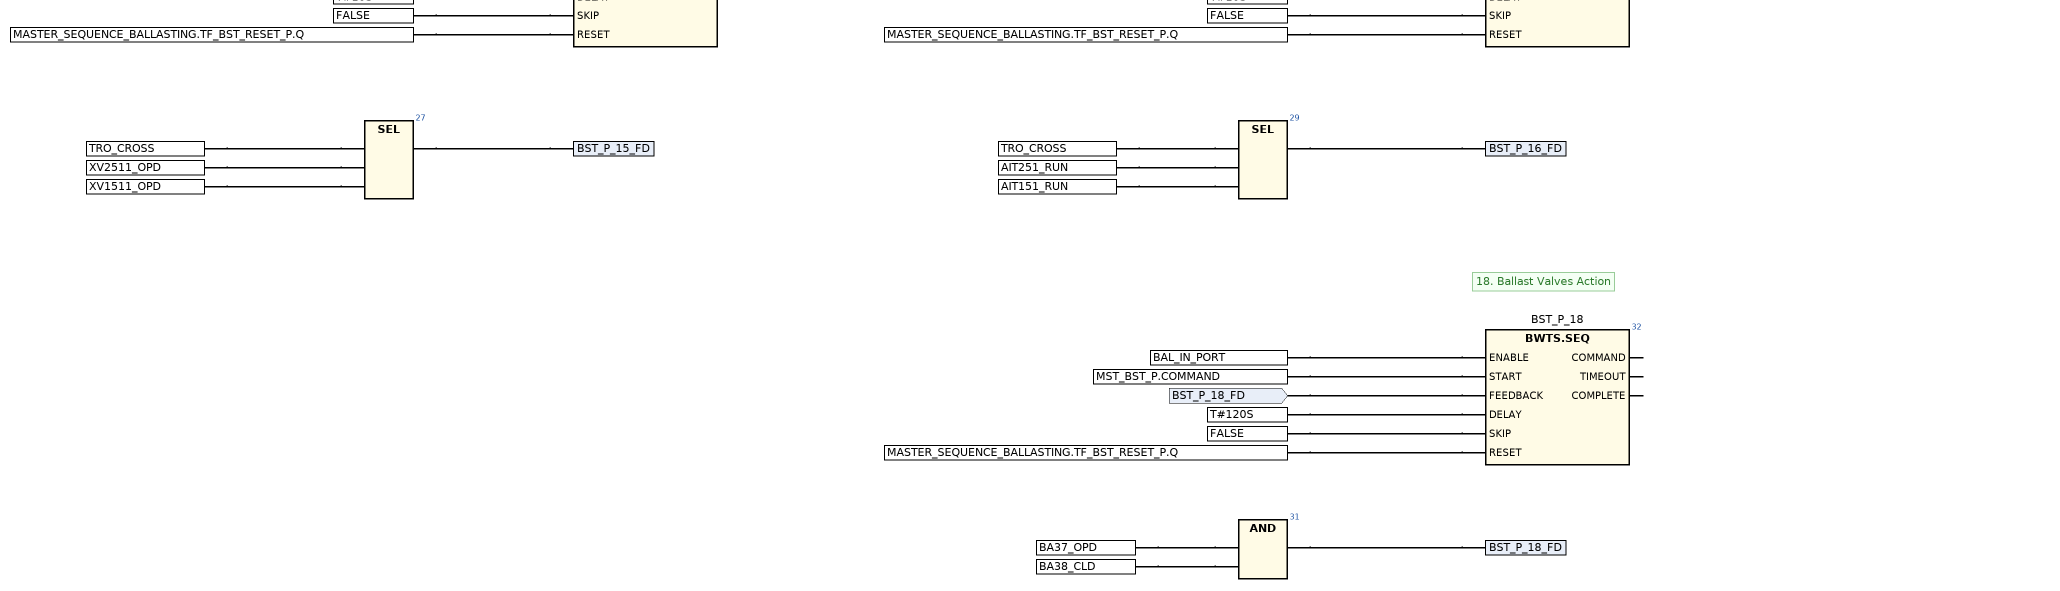
(* B117A_RUN AND XV1171A_OPD OR B117B_RUN AND XV1171B_OPD; result not used *)
// 01. Blower Start
BST_P_01(
    ENABLE := BAL_IN_PORT,
    START := MST_BST_P.COMMAND,
    FEEDBACK := _w1,
    DELAY := T#35s,
    SKIP := _w1,
    RESET := MASTER_SEQUENCE_BALLASTING.TF_BST_RESET_P.Q); // BWTS.SEQ
// BLOWER  PRE RUNNING TIME
TON_1(IN := BST_P_01.COMPLETE, PT := SEL(SEQ_BAL_ST_S.TON_1.Q, MS_BLR_PRE, T#0S)); // TON
// SWFP RUNNING WAITING TIME
TON_2(IN := BST_P_06.COMPLETE, PT := SEL(SEQ_BAL_ST_S.TON_2.Q, MS_SWP_ST, T#0S)); // TON
// 03. TRC Valve Init. Open
BST_P_03(
    ENABLE := BAL_IN_PORT,
    START := TON_1.Q,
    FEEDBACK := FCV2211_OPD,
    DELAY := T#120S,
    SKIP := FCV2211_OPD,
    RESET := MASTER_SEQUENCE_BALLASTING.TF_BST_RESET_P.Q); // BWTS.SEQ
// 04. Inj. Valve Init. Open
BST_P_04(
    ENABLE := BAL_IN_PORT,
    START := TON_1.Q,
    FEEDBACK := FCV2131_OPD,
    DELAY := T#30S,
    SKIP := FCV2131_OPD,
    RESET := MASTER_SEQUENCE_BALLASTING.TF_BST_RESET_P.Q); // BWTS.SEQ
// TRO RUNNING WATITNG TIME
TON_3(IN := BST_P_08.COMPLETE, PT := SEL(SEQ_BAL_ST_S.TON_3.Q, MS_TRO_WAIT, T#0S)); // TON
(* P171A_RUN OR P171B_RUN; result not used *)
// 06. S.W.F.P Start
BST_P_06(
    ENABLE := BAL_IN_PORT,
    START := TON_1.Q,
    FEEDBACK := _w2,
    DELAY := T#30S,
    SKIP := BST_S_06.COMPLETE,
    RESET := MASTER_SEQUENCE_BALLASTING.TF_BST_RESET_P.Q); // BWTS.SEQ
// 05. H/E Valve Init. Open
BST_P_05(
    ENABLE := BAL_IN_PORT,
    START := TON_1.Q,
    FEEDBACK := XV1731_OPD,
    DELAY := T#10S,
    SKIP := BST_S_05.COMPLETE,
    RESET := MASTER_SEQUENCE_BALLASTING.TF_BST_RESET_P.Q); // BWTS.SEQ
// 07. E/U Level Check
BST_P_07(
    ENABLE := BAL_IN_PORT,
    START := TON_2.Q,
    FEEDBACK := LS_1111,
    DELAY := T#30S,
    SKIP := LS_1111,
    RESET := MASTER_SEQUENCE_BALLASTING.TF_BST_RESET_P.Q); // BWTS.SEQ
// 08. WBP Start Request
BST_P_08(
    ENABLE := BAL_IN_PORT,
    START := BST_P_10.COMPLETE,
    FEEDBACK := _w3,
    DELAY := T#120S,
    SKIP := FALSE,
    RESET := MASTER_SEQUENCE_BALLASTING.TF_BST_RESET_P.Q); // BWTS.SEQ
(* CT_1111 > MS_CIT_NOR OR MF_CT1111; result not used *)
// 10. Salinity Check
BST_P_10(
    ENABLE := BAL_IN_PORT,
    START := BST_P_07.COMPLETE,
    FEEDBACK := _w4,
    DELAY := T#180S,
    RESET := MASTER_SEQUENCE_BALLASTING.TF_BST_RESET_P.Q); // BWTS.SEQ
// 12. Main Flow Control
BST_P_12(
    ENABLE := BAL_IN_PORT,
    START := BST_P_08.COMPLETE,
    FEEDBACK := BST_P_12.COMMAND,
    DELAY := T#5S,
    SKIP := FALSE,
    RESET := MASTER_SEQUENCE_BALLASTING.TF_BST_RESET_P.Q); // BWTS.SEQ
// 13. Inj. Flow Control
BST_P_13(
    ENABLE := BAL_IN_PORT,
    START := BST_P_08.COMPLETE,
    FEEDBACK := BST_P_13.COMMAND,
    DELAY := T#5S,
    SKIP := FALSE,
    RESET := MASTER_SEQUENCE_BALLASTING.TF_BST_RESET_P.Q); // BWTS.SEQ
(* SEL(RFA_DISABLE, RFA_RUN, TRUE) AND SEL(RFB_DISABLE, RFB_RUN, TRUE) AND SEL(RFC_DISABLE, RFC_RUN, TRUE); result not used *)
// 14. Rectifier Start
BST_P_14(
    ENABLE := BAL_IN_PORT,
    START := BST_P_08.COMPLETE,
    FEEDBACK := _w5,
    DELAY := T#20S,
    SKIP := FALSE,
    RESET := MASTER_SEQUENCE_BALLASTING.TF_BST_RESET_P.Q); // BWTS.SEQ
(* SEL(TRO_CROSS, XV2511_OPD, XV1511_OPD); result not used *)
// 15. TRO Valve Open
BST_P_15(
    ENABLE := BAL_IN_PORT,
    START := BST_P_08.COMPLETE,
    FEEDBACK := _w6,
    DELAY := T#10S,
    SKIP := FALSE,
    RESET := MASTER_SEQUENCE_BALLASTING.TF_BST_RESET_P.Q); // BWTS.SEQ
(* SEL(TRO_CROSS, AIT251_RUN, AIT151_RUN); result not used *)
// 16. TRO Sensing Start
BST_P_16(
    ENABLE := BAL_IN_PORT,
    START := TON_3.Q,
    FEEDBACK := _w7,
    DELAY := T#10S,
    SKIP := FALSE,
    RESET := MASTER_SEQUENCE_BALLASTING.TF_BST_RESET_P.Q); // BWTS.SEQ
(* BA37_OPD AND BA38_CLD; result not used *)
// 18. Ballast Valves Action
BST_P_18(
    ENABLE := BAL_IN_PORT,
    START := MST_BST_P.COMMAND,
    FEEDBACK := _w8,
    DELAY := T#120S,
    SKIP := FALSE,
    RESET := MASTER_SEQUENCE_BALLASTING.TF_BST_RESET_P.Q); // BWTS.SEQ

END_PROGRAM

// Device/Application/Logic/2.Sequence/SEQ_BAL_ST_S
PROGRAM SEQ_BAL_ST_S
VAR
	TON_1 : TON;		// BLOWER PRE RUNNING TIME
	TON_2 : TON;		// SWFP RUNNING WAITING TIME
	TON_3 : TON;		// TRO RUNNING WAITING TIME
END_VAR
VAR // added by the converter: edge detectors and wires of the graphical bodies
    _w1, _w2, _w3, _w4, _w5, _w6, _w7, _w8 : ANY;
END_VAR

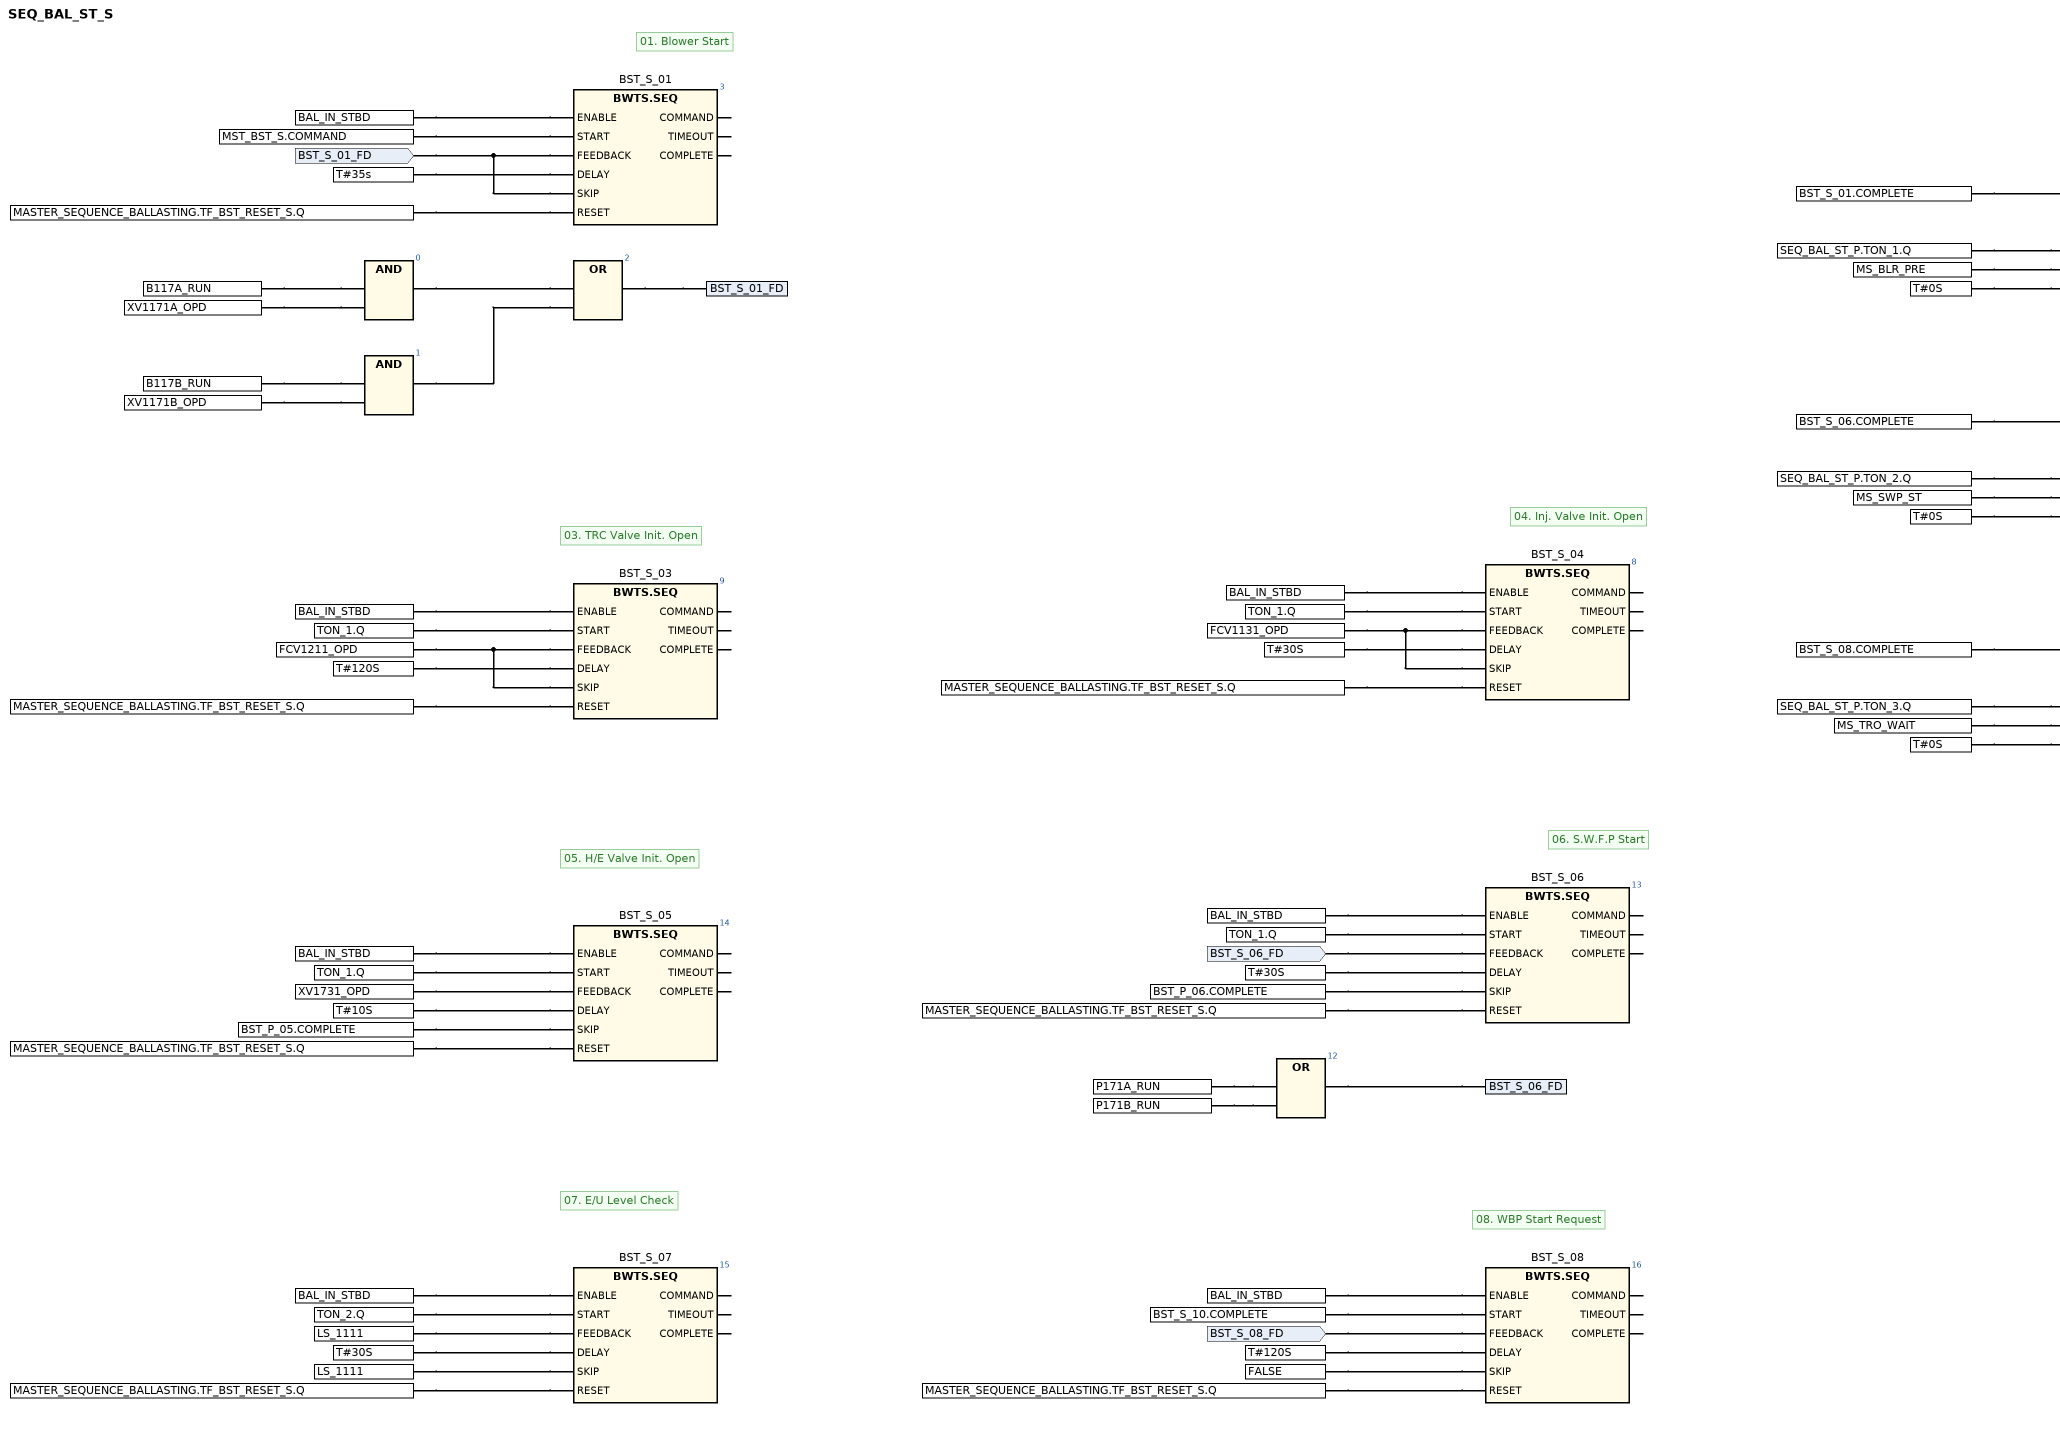
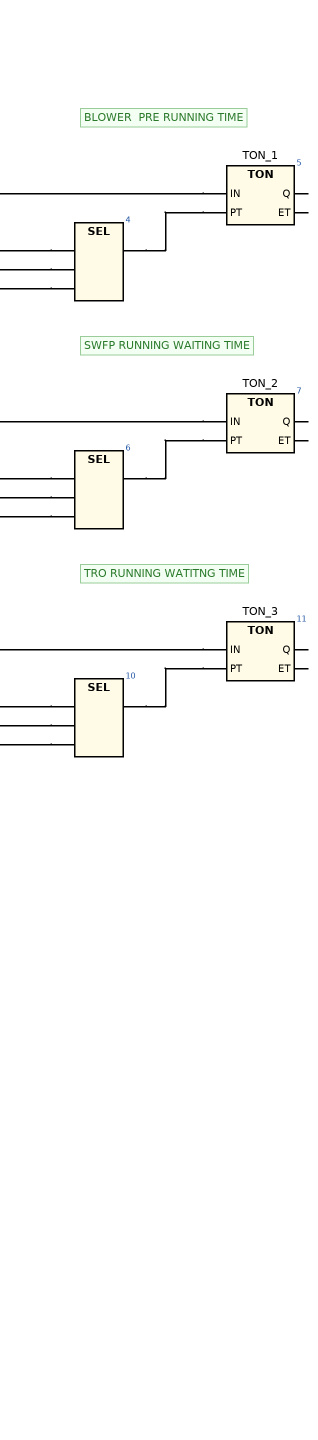
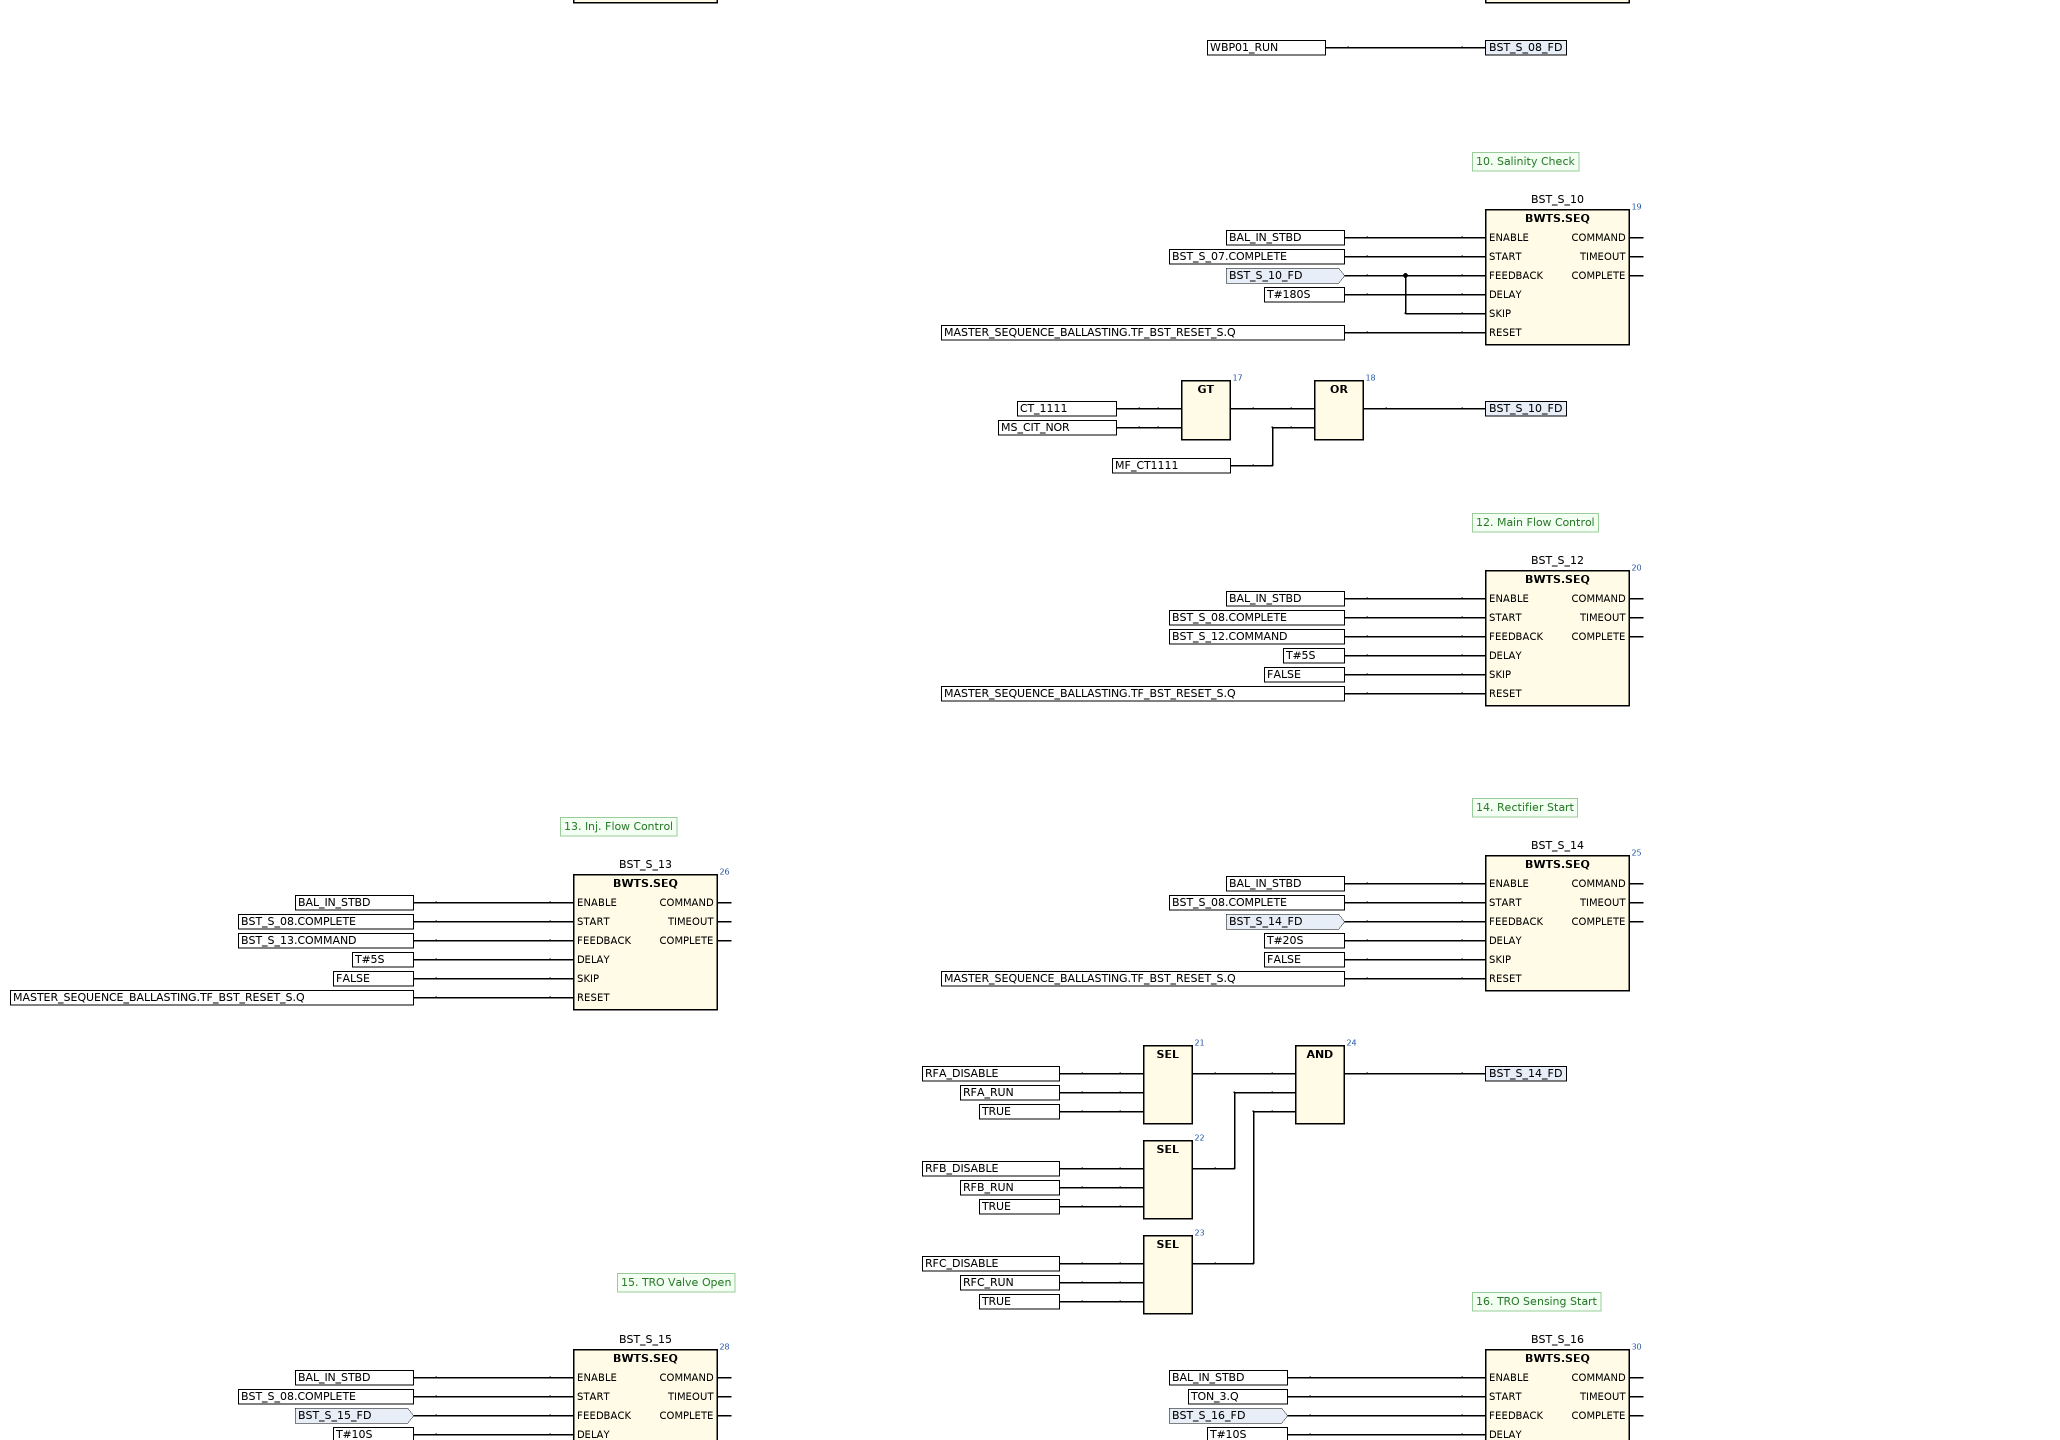
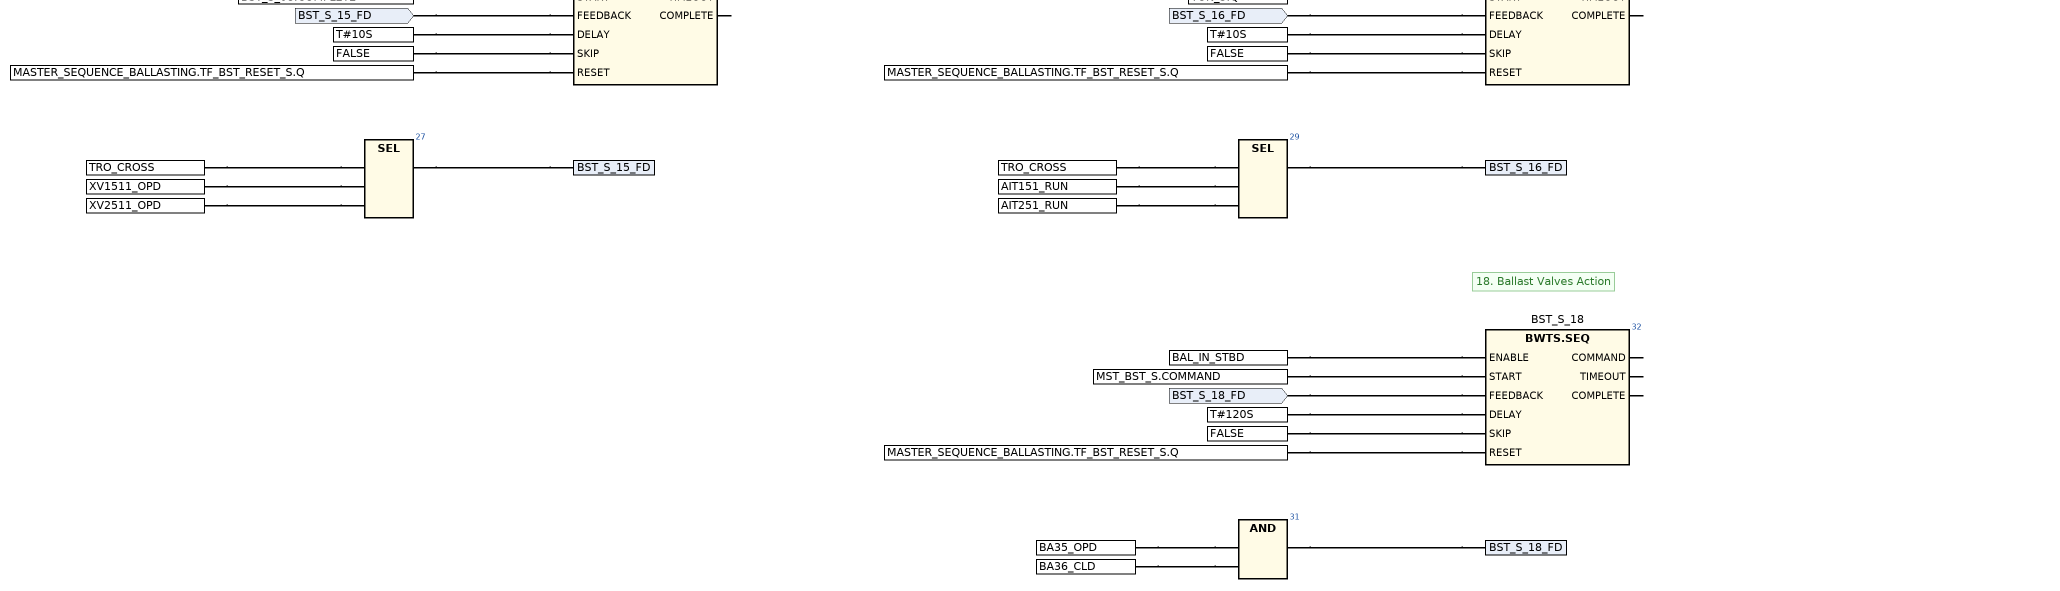
(* B117A_RUN AND XV1171A_OPD OR B117B_RUN AND XV1171B_OPD; result not used *)
// 01. Blower Start
BST_S_01(
    ENABLE := BAL_IN_STBD,
    START := MST_BST_S.COMMAND,
    FEEDBACK := _w1,
    DELAY := T#35s,
    SKIP := _w1,
    RESET := MASTER_SEQUENCE_BALLASTING.TF_BST_RESET_S.Q); // BWTS.SEQ
// BLOWER  PRE RUNNING TIME
TON_1(IN := BST_S_01.COMPLETE, PT := SEL(SEQ_BAL_ST_P.TON_1.Q, MS_BLR_PRE, T#0S)); // TON
// SWFP RUNNING WAITING TIME
TON_2(IN := BST_S_06.COMPLETE, PT := SEL(SEQ_BAL_ST_P.TON_2.Q, MS_SWP_ST, T#0S)); // TON
// 04. Inj. Valve Init. Open
BST_S_04(
    ENABLE := BAL_IN_STBD,
    START := TON_1.Q,
    FEEDBACK := FCV1131_OPD,
    DELAY := T#30S,
    SKIP := FCV1131_OPD,
    RESET := MASTER_SEQUENCE_BALLASTING.TF_BST_RESET_S.Q); // BWTS.SEQ
// 03. TRC Valve Init. Open
BST_S_03(
    ENABLE := BAL_IN_STBD,
    START := TON_1.Q,
    FEEDBACK := FCV1211_OPD,
    DELAY := T#120S,
    SKIP := FCV1211_OPD,
    RESET := MASTER_SEQUENCE_BALLASTING.TF_BST_RESET_S.Q); // BWTS.SEQ
// TRO RUNNING WATITNG TIME
TON_3(IN := BST_S_08.COMPLETE, PT := SEL(SEQ_BAL_ST_P.TON_3.Q, MS_TRO_WAIT, T#0S)); // TON
(* P171A_RUN OR P171B_RUN; result not used *)
// 06. S.W.F.P Start
BST_S_06(
    ENABLE := BAL_IN_STBD,
    START := TON_1.Q,
    FEEDBACK := _w2,
    DELAY := T#30S,
    SKIP := BST_P_06.COMPLETE,
    RESET := MASTER_SEQUENCE_BALLASTING.TF_BST_RESET_S.Q); // BWTS.SEQ
// 05. H/E Valve Init. Open
BST_S_05(
    ENABLE := BAL_IN_STBD,
    START := TON_1.Q,
    FEEDBACK := XV1731_OPD,
    DELAY := T#10S,
    SKIP := BST_P_05.COMPLETE,
    RESET := MASTER_SEQUENCE_BALLASTING.TF_BST_RESET_S.Q); // BWTS.SEQ
// 07. E/U Level Check
BST_S_07(
    ENABLE := BAL_IN_STBD,
    START := TON_2.Q,
    FEEDBACK := LS_1111,
    DELAY := T#30S,
    SKIP := LS_1111,
    RESET := MASTER_SEQUENCE_BALLASTING.TF_BST_RESET_S.Q); // BWTS.SEQ
// 08. WBP Start Request
BST_S_08(
    ENABLE := BAL_IN_STBD,
    START := BST_S_10.COMPLETE,
    FEEDBACK := _w3,
    DELAY := T#120S,
    SKIP := FALSE,
    RESET := MASTER_SEQUENCE_BALLASTING.TF_BST_RESET_S.Q); // BWTS.SEQ
(* CT_1111 > MS_CIT_NOR OR MF_CT1111; result not used *)
// 10. Salinity Check
BST_S_10(
    ENABLE := BAL_IN_STBD,
    START := BST_S_07.COMPLETE,
    FEEDBACK := _w4,
    DELAY := T#180S,
    SKIP := _w4,
    RESET := MASTER_SEQUENCE_BALLASTING.TF_BST_RESET_S.Q); // BWTS.SEQ
// 12. Main Flow Control
BST_S_12(
    ENABLE := BAL_IN_STBD,
    START := BST_S_08.COMPLETE,
    FEEDBACK := BST_S_12.COMMAND,
    DELAY := T#5S,
    SKIP := FALSE,
    RESET := MASTER_SEQUENCE_BALLASTING.TF_BST_RESET_S.Q); // BWTS.SEQ
(* SEL(RFA_DISABLE, RFA_RUN, TRUE) AND SEL(RFB_DISABLE, RFB_RUN, TRUE) AND SEL(RFC_DISABLE, RFC_RUN, TRUE); result not used *)
// 14. Rectifier Start
BST_S_14(
    ENABLE := BAL_IN_STBD,
    START := BST_S_08.COMPLETE,
    FEEDBACK := _w5,
    DELAY := T#20S,
    SKIP := FALSE,
    RESET := MASTER_SEQUENCE_BALLASTING.TF_BST_RESET_S.Q); // BWTS.SEQ
// 13. Inj. Flow Control
BST_S_13(
    ENABLE := BAL_IN_STBD,
    START := BST_S_08.COMPLETE,
    FEEDBACK := BST_S_13.COMMAND,
    DELAY := T#5S,
    SKIP := FALSE,
    RESET := MASTER_SEQUENCE_BALLASTING.TF_BST_RESET_S.Q); // BWTS.SEQ
(* SEL(TRO_CROSS, XV1511_OPD, XV2511_OPD); result not used *)
// 15. TRO Valve Open
BST_S_15(
    ENABLE := BAL_IN_STBD,
    START := BST_S_08.COMPLETE,
    FEEDBACK := _w6,
    DELAY := T#10S,
    SKIP := FALSE,
    RESET := MASTER_SEQUENCE_BALLASTING.TF_BST_RESET_S.Q); // BWTS.SEQ
(* SEL(TRO_CROSS, AIT151_RUN, AIT251_RUN); result not used *)
// 16. TRO Sensing Start
BST_S_16(
    ENABLE := BAL_IN_STBD,
    START := TON_3.Q,
    FEEDBACK := _w7,
    DELAY := T#10S,
    SKIP := FALSE,
    RESET := MASTER_SEQUENCE_BALLASTING.TF_BST_RESET_S.Q); // BWTS.SEQ
(* BA35_OPD AND BA36_CLD; result not used *)
// 18. Ballast Valves Action
BST_S_18(
    ENABLE := BAL_IN_STBD,
    START := MST_BST_S.COMMAND,
    FEEDBACK := _w8,
    DELAY := T#120S,
    SKIP := FALSE,
    RESET := MASTER_SEQUENCE_BALLASTING.TF_BST_RESET_S.Q); // BWTS.SEQ

END_PROGRAM

// Device/Application/Logic/2.Sequence/SEQ_DEBAL_SP_P
PROGRAM SEQ_DEBAL_SP_P
VAR
	TON_0: TON;
	DST_S_ON: BOOL;
END_VAR
VAR // added by the converter: edge detectors and wires of the graphical bodies
    _w1, _w2, _w3, _w4, _w5, _w6, _w7 : ANY;
END_VAR

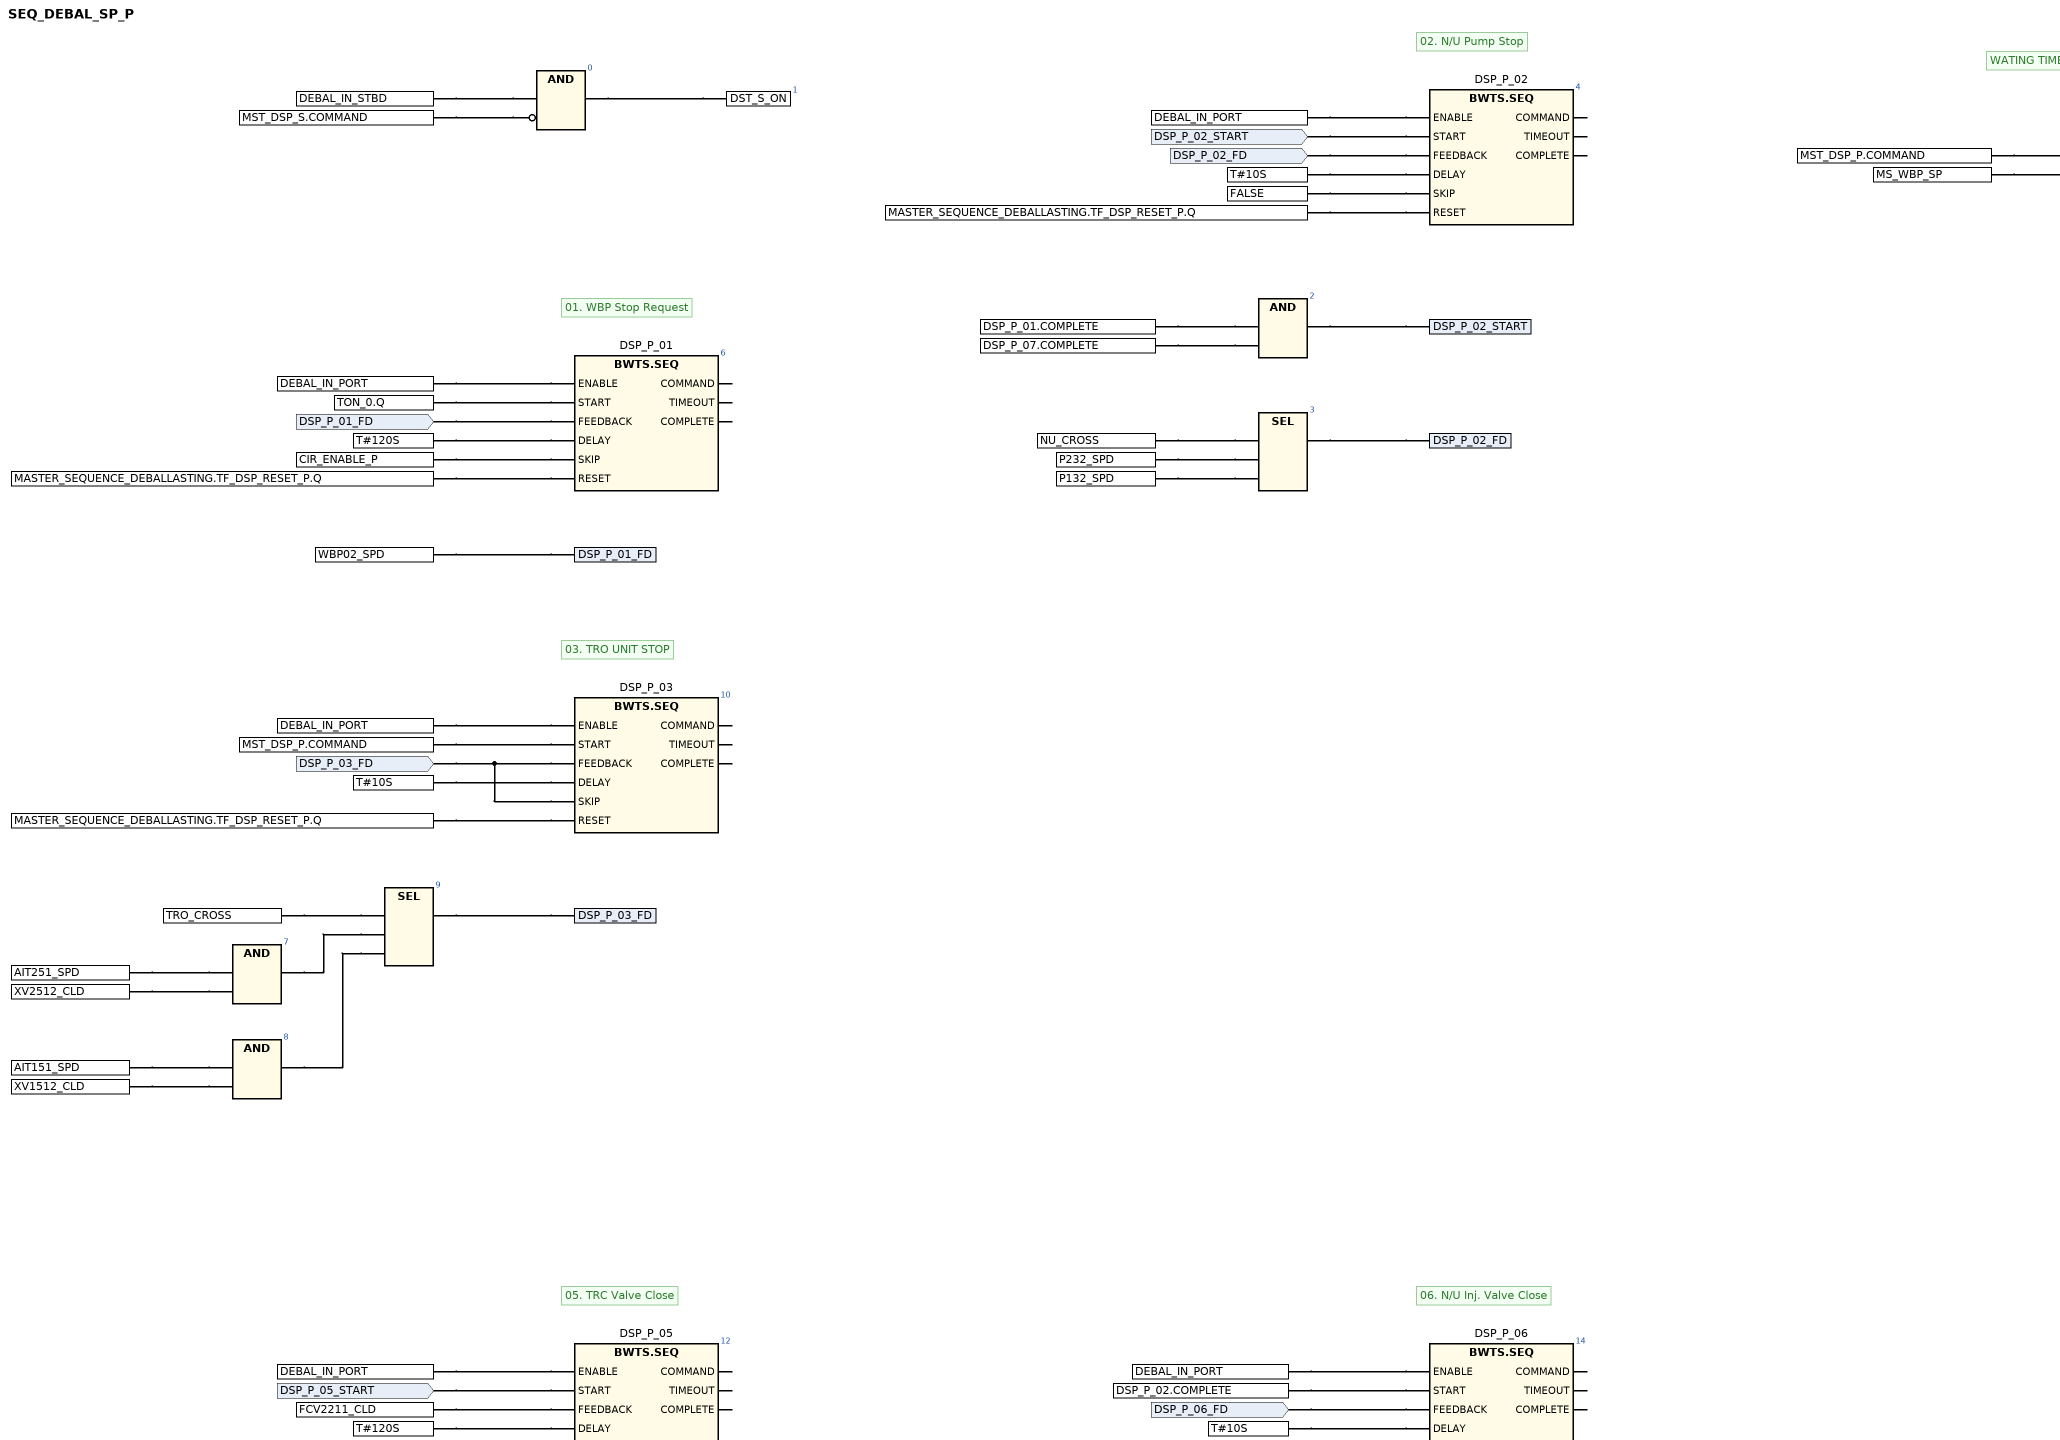
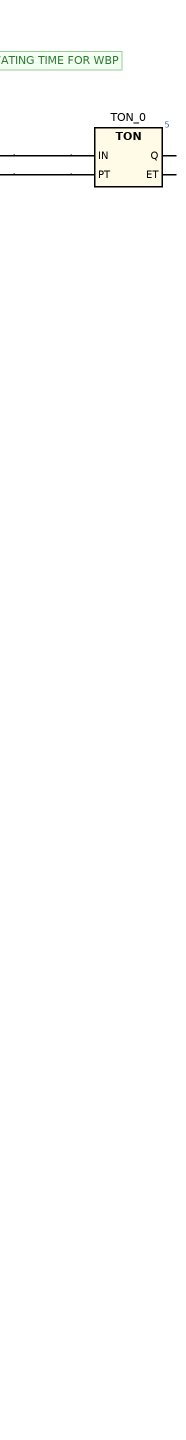
